// SIMATIC STEP 7 (V5.x) project Saldatura
// CPU: CPU 315-2 DP
// station: P_ADR_BUS
// station: Hardware
// station: SIMATIC 300(1)
// program: Programma S7(1)
// program: Originale

SYMBOL_TABLE
"Z10"	C 10	COUNTER	// Counter
"Z11"	C 11	COUNTER	// Counter
"Z12"	C 12	COUNTER	// Counter
"Z13"	C 13	COUNTER	// Counter
"DI_Balluff1"	DB 5	FB 20	// DB Instance of FB20
"DatiOP170B"	DB 7	DB 7	// PLC<->OP170B interface
"Timer"	DB 20	DB 20
"DBWork"	DB 21	DB 21
"coordinate"	DB 22	DB 22
"DB180"	DB 180	FB 24	// DB instance FB24 AsseY
"DB181"	DB 181	FB 24	// DB instance FB24 AsseX
"DBWork2"	DB 200	DB 200
"Asse_611U"	FB 16	FB 16	// Axis 611U management
"BALLUFF"	FB 20	FB 20	// BALLUFF Reader/Writer management
"FB24 - Gestione Mov Assi"	FB 24	FB 24	// GESTIONE ASSI STAZIONE
"NormalizzazioneAnalogico"	FC 7	FC 7	// Normalization of a analog value
"FC11 - STATUS"	FC 11	FC 11	// Sensors and proximity state
"FC12 - GENERAL"	FC 12	FC 12	// General management
"FC13 - MANUAL"	FC 13	FC 13	// Manual commands
"FC14 - AUTOMATIC"	FC 14	FC 14	// Automatic cycle management
"FC16 - ALARMS"	FC 16	FC 16	// Alarms management
"FC17 - OPERATOR PANNEL"	FC 17	FC 17	// Operator pannel management
"FC18 - OUTPUTS"	FC 18	FC 18	// Outputs management
"FC19 - REPOSITIONING"	FC 19	FC 19	// Repositioning management
"FC - AUTOMATIC"	FC 24	FC 24
"FC50 - TEACH-IN"	FC 50	FC 50
"FC51 - TYPE TOOL"	FC 51	FC 51
"FC52 - SYSTEM VISION"	FC 52	FC 52
"FC53 - REWORK"	FC 53	FC 53
"FC81 - GEST AXIS"	FC 81	FC 81	// Management axis
"FC117 - ERROR TOOL"	FC 117	FC 117
"TimeOut"	FC 800	FC 800	// Management TimeOut movimenti
"E0.0"	I 0.0	BOOL	// THERMAL SWTCH_ASPIRATOR_MTR
"E0.1"	I 0.1	BOOL	// 230 Vac power supply circuit braker
"E0.2"	I 0.2	BOOL	// 230 VAC PS CKT BRAKER
"E0.3"	I 0.3	BOOL	// Welding Machine OK
"E0.4"	I 0.4	BOOL	// Reserve
"E0.5"	I 0.5	BOOL	// AUXILIXARY ON
"DOOR CLOSE"	I 0.6	BOOL	// Reserve
"E0.7"	I 0.7	BOOL	// SAFETY BARRIER
"E1.0"	I 1.0	BOOL	// CYCLE_START
"E1.1"	I 1.1	BOOL	// AUTO_MANUAL
"E1.2"	I 1.2	BOOL	// COMPRESSED AIR
"E1.3"	I 1.3	BOOL	// AXIS RESET_POS
"E1.4"	I 1.4	BOOL	// Rotary table motor thermal switch
"E1.5"	I 1.5	BOOL	// LCK_UNLCK_DOORS_PB
"E1.6"	I 1.6	BOOL	// Reserve
"E1.7"	I 1.7	BOOL	// DRIVE TEMP
"E2.0"	I 2.0	BOOL	// STOP_CYCLE_PB
"E2.1"	I 2.1	BOOL	// Doors Closed & Locked
"E2.2"	I 2.2	BOOL	// Safety Barrier OK
"E2.3"	I 2.3	BOOL	// WELDING_TORCH_DWN
"E2.4"	I 2.4	BOOL	// WELDING_TORCH_UP
"E2.5"	I 2.5	BOOL	// ROTARY_TABLE_ZERO
"E2.6"	I 2.6	BOOL	// ROTARY_TABLE_ZERO1
"E2.7"	I 2.7	BOOL	// Reserve
"E3.0"	I 3.0	BOOL	// VEN DETECTOR_FWD
"E3.1"	I 3.1	BOOL	// VEN DETECTOR_REV
"E3.2"	I 3.2	BOOL	// VEN DETECTOR_DWN
"E3.3"	I 3.3	BOOL	// VEN DETECTOR_UP
"E3.4"	I 3.4	BOOL	// ROTARY_TABLE_CAM
"E3.5"	I 3.5	BOOL	// Reserve
"E3.6"	I 3.6	BOOL	// Reserve
"E3.7"	I 3.7	BOOL	// Reserve
"e5.0"	I 5.0	BOOL	// Lever Detector System - bit 0
"e5.1"	I 5.1	BOOL	// Lever Detector System - bit 1
"e5.2"	I 5.2	BOOL	// Lever Detector System - bit 2
"e5.3"	I 5.3	BOOL	// Lever Detector System - bit 3
"e5.4"	I 5.4	BOOL	// Lever Detector System - bit 4
"e5.5"	I 5.5	BOOL	// Lever Detector System - bit 5
"e5.6"	I 5.6	BOOL	// Lever Detector System - bit 6
"e5.7"	I 5.7	BOOL	// Lever Detector System - bit 7
"e6.0"	I 6.0	BOOL	// Lever Detector System - bit 8
"e6.1"	I 6.1	BOOL	// Lever Detector System - bit 9
"e6.2"	I 6.2	BOOL	// Lever Detector System - bit 10
"e6.3"	I 6.3	BOOL	// Lever Detector System - bit 11 - 12è13
"e6.4"	I 6.4	BOOL	// Lever Detector System - bit 12
"e6.5"	I 6.5	BOOL	// Lever Detector System - bit 13
"e6.6"	I 6.6	BOOL	// Lever Detector System - bit 14
"e6.7"	I 6.7	BOOL	// Lever Detector System - Vane Assy Total Number
"EXSTRACTOR_HIGH"	I 7.2	BOOL
"EXSTRACTOR_LOW"	I 7.3	BOOL
"TABLE_LCK_CYCLINDER_UP"	I 7.4	BOOL
"TABLE_LCK_CYCLINDER_DWN"	I 7.5	BOOL
"E32.0"	I 32.0	BOOL	// Push-button start cycle (on load position)
"E32.1"	I 32.1	BOOL	// Push button stop cycle
"E32.2"	I 32.2	BOOL	// Aut/Man Selector
"E32.3"	I 32.3	BOOL	// Reserve
"E32.4"	I 32.4	BOOL	// Reserve
"E32.5"	I 32.5	BOOL	// Lock/Unlock doors Push Button
"E32.6"	I 32.6	BOOL	// Reserve
"E32.7"	I 32.7	BOOL	// Air Presence
"E34.0"	I 34.0	BOOL	// Cam Table
"E34.1"	I 34.1	BOOL	// Reserve
"E34.2"	I 34.2	BOOL	// Reserve
"E34.3"	I 34.3	BOOL	// Reserve
"E34.4"	I 34.4	BOOL	// Table locker cylinder  up
"E34.5"	I 34.5	BOOL	// Table locker cylinder down
"E34.6"	I 34.6	BOOL	// Exstractor High
"E34.7"	I 34.7	BOOL	// Extractor Low
"E35.0"	I 35.0	BOOL	// Torch Welding low
"E35.1"	I 35.1	BOOL	// Torch Welding high
"E35.2"	I 35.2	BOOL	// Home Assy
"E35.3"	I 35.3	BOOL	// 1 --> PP1 on welding ; 0 --> PP2 on welding
"E35.4"	I 35.4	BOOL	// Detect components Control group High
"E35.5"	I 35.5	BOOL	// Detect components Control group Low
"E35.6"	I 35.6	BOOL	// Detect components Control group forward
"E35.7"	I 35.7	BOOL	// Detect components Control group backward
"E36.0"	I 36.0	BOOL	// Reserve not mounted
"E36.1"	I 36.1	BOOL	// Reserve not mounted
"E36.2"	I 36.2	BOOL	// Reserve not mounted
"E36.3"	I 36.3	BOOL	// Reserve not mounted
"E36.4"	I 36.4	BOOL	// Reserve not mounted
"E36.5"	I 36.5	BOOL	// Reserve not mounted
"E36.6"	I 36.6	BOOL	// Reserve not mounted
"E36.7"	I 36.7	BOOL	// Reserve not mounted
"E52.0"	I 52.0	BOOL	// Lever Detector System - bit 0
"E52.1"	I 52.1	BOOL	// Lever Detector System - bit 1
"E52.2"	I 52.2	BOOL	// Lever Detector System - bit 2
"E52.3"	I 52.3	BOOL	// Lever Detector System - bit 3
"E52.4"	I 52.4	BOOL	// Lever Detector System - bit 4
"E52.5"	I 52.5	BOOL	// Lever Detector System - bit 5
"E52.6"	I 52.6	BOOL	// Lever Detector System - bit 6
"E52.7"	I 52.7	BOOL	// Lever Detector System - bit 7
"E53.0"	I 53.0	BOOL	// Lever Detector System - bit 8
"E53.1"	I 53.1	BOOL	// Lever Detector System - bit 9
"E53.2"	I 53.2	BOOL	// Lever Detector System - bit 10
"E53.3"	I 53.3	BOOL	// Lever Detector System - bit 11 - 12è13
"E53.4"	I 53.4	BOOL	// Lever Detector System - bit 12
"E53.5"	I 53.5	BOOL	// Lever Detector System - bit 13
"E53.6"	I 53.6	BOOL	// Lever Detector System - bit 14
"E53.7"	I 53.7	BOOL	// Lever Detector System - Vane Assy Total Number
"E64.0"	I 64.0	BOOL	// VOSION SYSTEM OK
"E64.1"	I 64.1	BOOL	// Busy
"E64.2"	I 64.2	BOOL	// Or
"E64.3"	I 64.3	BOOL	// Error
"E64.4"	I 64.4	BOOL	// Gate
"E64.5"	I 64.5	BOOL	// Strobe trigger 0 out
"E64.6"	I 64.6	BOOL	// Strobe trigger 1 out
"E64.7"	I 64.7	BOOL	// DO0
"E65.0"	I 65.0	BOOL	// DO1
"E65.1"	I 65.1	BOOL	// DO2
"E65.2"	I 65.2	BOOL	// DO3
"E65.3"	I 65.3	BOOL	// DO4
"E65.4"	I 65.4	BOOL	// DO5
"E65.5"	I 65.5	BOOL	// DO6
"E65.6"	I 65.6	BOOL	// DO7
"E65.7"	I 65.7	BOOL	// DO8
"M0.0"	M 0.0	BOOL	// Clock 0,1 s
"M0.1"	M 0.1	BOOL	// Clock 0,2 s
"M0.2"	M 0.2	BOOL	// Clock 0,4 s
"M0.3"	M 0.3	BOOL	// Clock 0,5 s
"M0.4"	M 0.4	BOOL	// Clock 0,8 s
"M0.5"	M 0.5	BOOL	// Clock 1 s
"M0.6"	M 0.6	BOOL	// Clock 1,6 s
"M0.7"	M 0.7	BOOL	// Clock 2 s
"Off"	M 1.0	BOOL	// Merker always OFF
"On"	M 1.1	BOOL	// Merker always ON
"ToDo"	M 1.2	BOOL
"Bypass"	M 1.3	BOOL	// Merker that indicates a bypass forced of the code
"BypassPC"	M 1.4	BOOL	// Merker for bypass control handshake with PC supervision
"Clock_P"	M 1.5	BOOL	// Positiv pulse of clock
"Clock_N"	M 1.6	BOOL	// Negativ pulse of code
"Clock_10s"	M 1.7	BOOL	// 10 seconds clock
"M2.0"	M 2.0	BOOL	// Occhio
"BPSupervisor"	M 3.0	BOOL	// By Pass del supervisore
"Auxiliary_ON"	M 10.0	BOOL	// Auxiliary ON
"COMPRESSED_AIR"	M 10.1	BOOL	// Compressed Air
"SHIELDS_OK"	M 10.2	BOOL	// Schermi Chiusi e bloccati
"MACHINE_ON"	M 10.3	BOOL	// Machine OK
"Occhio"	M 10.7	BOOL
"START_POS"	M 11.0	BOOL	// Machine in initial positon
"START_POS_MEM"	M 11.1	BOOL	// mem initial position
"M11.2"	M 11.2	BOOL	// Manual Mode Selected
"SEMI"	M 11.3	BOOL	// Selezione modo semi automatico
"AUT"	M 11.4	BOOL	// Automatic Mode Selected
"START"	M 12.0	BOOL	// Start machine
"START_PULSE"	M 12.1	BOOL	// Pulse of start push-button
"SINGLE_CYCLE"	M 12.2	BOOL	// 1=ciclo singolo 0=ciclo continuo
"ALARM"	M 12.3	BOOL	// Alarm
"END_CYCLE"	M 12.4	BOOL	// Automatic cycle finished
"CmdMan_Av"	M 12.5	BOOL	// Forward manual command
"CmdMan_Ind"	M 12.6	BOOL	// Backward manual command
"STOP_BUTTON"	M 12.7	BOOL	// STATUS - stop button
"M13.0"	M 13.0	BOOL	// STATUS - Lock/Unlock doors Push Button
"M14.0"	M 14.0	BOOL	// Mem Lever Detector System - bit 0
"M14.1"	M 14.1	BOOL	// Mem Lever Detector System - bit 1
"M14.2"	M 14.2	BOOL	// Mem Lever Detector System - bit 2
"M14.3"	M 14.3	BOOL	// Mem Lever Detector System - bit 3
"M14.4"	M 14.4	BOOL	// Mem Lever Detector System - bit 4
"M14.5"	M 14.5	BOOL	// Mem Lever Detector System - bit 5
"M14.6"	M 14.6	BOOL	// Mem Lever Detector System - bit 6
"M14.7"	M 14.7	BOOL	// Mem Lever Detector System - bit 7
"M15.0"	M 15.0	BOOL	// Mem Lever Detector System - bit 8
"M15.1"	M 15.1	BOOL	// Mem Lever Detector System - bit 9
"M15.2"	M 15.2	BOOL	// Mem Lever Detector System - bit 10
"M15.3"	M 15.3	BOOL	// Mem Lever Detector System - bit 11
"M15.4"	M 15.4	BOOL	// Mem Lever Detector System - bit 12
"M15.5"	M 15.5	BOOL	// Mem Lever Detector System - bit 13
"M15.6"	M 15.6	BOOL	// Mem Lever Detector System - bit 14 (Roller)
"M15.7"	M 15.7	BOOL	// Mem Lever Detector System - bit 15
"M16.0"	M 16.0	BOOL	// mem Reworked Parts
"M16.1"	M 16.1	BOOL	// Disable Extractor if Rework
"M16.2"	M 16.2	BOOL	// Part on table 1 welding
"M16.3"	M 16.3	BOOL	// Part on Table 2 Welding
"M16.4"	M 16.4	BOOL	// Table can ROTATE
"M16.5"	M 16.5	BOOL	// Extractor can MOVE
"M16.6"	M 16.6	BOOL	// OK Extract
"M16.7"	M 16.7	BOOL	// Manual PAge Active
"M17.2"	M 17.2	BOOL	// Rework
"M17.3"	M 17.3	BOOL	// Vane no welding
"M17.4"	M 17.4	BOOL	// PP2 - OUT
"M17.5"	M 17.5	BOOL	// PP1 - OUT
"M17.6"	M 17.6	BOOL	// AUX - F R E E
"M17.7"	M 17.7	BOOL	// AUX - F R E E
"M18.0"	M 18.0	BOOL	// AUX - F R E E
"M18.1"	M 18.1	BOOL	// AUX - F R E E
"M18.2"	M 18.2	BOOL	// AUX - F R E E
"M18.3"	M 18.3	BOOL	// AUX - F R E E
"M18.4"	M 18.4	BOOL	// AUX - F R E E
"M18.5"	M 18.5	BOOL	// AUX - F R E E
"M18.6"	M 18.6	BOOL	// AUX - F R E E
"M18.7"	M 18.7	BOOL	// AUX - F R E E
"M19.0"	M 19.0	BOOL	// AUX - F R E E
"M19.1"	M 19.1	BOOL	// AUX - F R E E
"M19.2"	M 19.2	BOOL	// AUX - F R E E
"M19.3"	M 19.3	BOOL	// AUX - F R E E
"M19.4"	M 19.4	BOOL	// AUX - F R E E
"M19.5"	M 19.5	BOOL	// AUX - F R E E
"M19.6"	M 19.6	BOOL	// AUX - F R E E
"M19.7"	M 19.7	BOOL	// AUX - F R E E
"M20.0"	M 20.0	BOOL	// AUX - F R E E
"M20.1"	M 20.1	BOOL	// AUX - F R E E
"M20.2"	M 20.2	BOOL	// Presence of tool to assembly nozzle
"M20.3"	M 20.3	BOOL	// AUX - F R E E
"M20.4"	M 20.4	BOOL	// Tension OK
"M20.5"	M 20.5	BOOL	// AUX - F R E E
"M20.6"	M 20.6	BOOL	// AUX - F R E E
"M20.7"	M 20.7	BOOL	// AUX-Man
"M21.0"	M 21.0	BOOL	// STATUS - Mem Component pinched on Workrest - FC1
"Mem E34.5"	M 21.1	BOOL	// Mem Component pinched on Workrest - FC2
"M21.2"	M 21.2	BOOL	// AUX - F R E E
"M21.3"	M 21.3	BOOL	// AUX - F R E E
"M21.4"	M 21.4	BOOL	// Aux Alarm
"Warning"	M 21.5	BOOL	// Warning
"ResetAlarm"	M 21.6	BOOL	// Reset alarm
"Repos"	M 21.7	BOOL	// Repositioning
"M22.0"	M 22.0	BOOL	// STATUS - Table locker up
"M22.1"	M 22.1	BOOL	// STATUS - Table locker Down
"CmdMan_Av_Pulse"	M 22.2	BOOL	// Pulse of forward manual command
"CmdMan_Ind_Pulse"	M 22.3	BOOL	// Pulse of backward manual command
"M22.4"	M 22.4	BOOL	// Forward command
"M22.5"	M 22.5	BOOL	// Backward command
"CmdMan_Esg"	M 22.6	BOOL	// Memory of manual command executed
"CicloInCorso"	M 22.7	BOOL	// Automatic cycle in course
"M23.0"	M 23.0	BOOL	// Mem Start
"StopAEndCycle"	M 23.1	BOOL
"ChangeFunc"	M 23.2	BOOL	// Pulse change operation mode
"PresencePz"	M 23.3	BOOL
"SafetyBarrier_KO"	M 23.5	BOOL	// STATUS - Security bar KO
"M24.0"	M 24.0	BOOL	// STATUS - Torch Welding low
"M24.1"	M 24.1	BOOL	// STATUS - Torch Welding high
"M24.2"	M 24.2	BOOL	// STATUS -
"M24.3"	M 24.3	BOOL	// STATUS -
"M24.4"	M 24.4	BOOL	// STATUS - Cam table
"M24.5"	M 24.5	BOOL	// 1 --> PP1 on welding ;0 --> PP2 on welding
"M25.0"	M 25.0	BOOL	// Position Rotation 0°
"M25.1"	M 25.1	BOOL	// Position Rotation 180°
"M25.2"	M 25.2	BOOL	// Pos 0° e camma OK
"M25.3"	M 25.3	BOOL	// Pos 180° e camma OK
"M25.7"	M 25.7	BOOL	// Pulse Cam
"M26.1"	M 26.1	BOOL	// Table is FREE
"M26.2"	M 26.2	BOOL	// STATUS - System Detector Up
"M26.3"	M 26.3	BOOL	// STATUS - System Detector Lower
"M26.4"	M 26.4	BOOL	// STATUS - Detector work position
"M26.5"	M 26.5	BOOL	// STATUS - Detector park position
"M26.6"	M 26.6	BOOL	// STATUS - Exstractor High
"M26.7"	M 26.7	BOOL	// STATUS - Extractor low
"M28.0"	M 28.0	BOOL	// STATUS - DO1SYSTEM VISION
"M28.1"	M 28.1	BOOL	// STATUS - DO2 SYSTEM VISION
"M28.2"	M 28.2	BOOL	// STATUS - DO3 SYSTEM VISION
"M28.3"	M 28.3	BOOL	// STATUS - DO4 SYSTEM VISION
"M29.0"	M 29.0	BOOL	// STATUS - Run System Vision
"M29.1"	M 29.1	BOOL	// STATUS - Busy System Vision
"M29.2"	M 29.2	BOOL	// STATUS - OK System Vision
"M29.3"	M 29.3	BOOL	// STATUS - Error System Vision
"M29.4"	M 29.4	BOOL	// STATUS - Gate System Vision
"M29.6"	M 29.6	BOOL	// STATUS - DO1 SYSTEM VISION
"M29.7"	M 29.7	BOOL	// STATUS - DO0 SYSTEM VISION
"M30.0"	M 30.0	BOOL	// MAN - Table Rotation Forward
"M30.1"	M 30.1	BOOL	// MAN - Table Rotation Backward
"M30.2"	M 30.2	BOOL	// MAN - Jog + AsseY
"M30.3"	M 30.3	BOOL	// MAN - Jog - AsseY
"M30.4"	M 30.4	BOOL	// MAN - Jog + AsseX
"M30.5"	M 30.5	BOOL	// MAN - Jog - AsseX
"M30.6"	M 30.6	BOOL	// MAN - Forward SD
"M30.7"	M 30.7	BOOL	// MAN - Backward SD
"M31.0"	M 31.0	BOOL	// MAN - High SD
"M31.1"	M 31.1	BOOL	// MAN - Low SD
"M31.2"	M 31.2	BOOL	// MAN - High TW
"M31.3"	M 31.3	BOOL	// MAN - Low TW
"M31.4"	M 31.4	BOOL	// MAN - Extractor High
"M31.5"	M 31.5	BOOL	// MAN - Extractor down
"M31.6"	M 31.6	BOOL	// MAN - ON\OFF TW
"M31.7"	M 31.7	BOOL	// MAN - START/STOP WM
"M32.0"	M 32.0	BOOL	// Man  -  Start Torch W"elding
"M32.1"	M 32.1	BOOL	// MAN - Test Arco Gas Ok
"M32.2"	M 32.2	BOOL	// MAN - Test Arco Gas
"M32.3"	M 32.3	BOOL	// MAN - Torch Welding Temp Ok
"M32.4"	M 32.4	BOOL	// MAN - low table locker cylinder
"M32.5"	M 32.5	BOOL	// MAN - up table locker cylinder
"M32.6"	M 32.6	BOOL	// MAN - Welding
"M32.7"	M 32.7	BOOL	// MAN - Free
"M33.0"	M 33.0	BOOL	// MAN - Free
"M33.1"	M 33.1	BOOL	// MAN - Free
"M33.2"	M 33.2	BOOL	// MAN - Free
"M33.3"	M 33.3	BOOL	// MAN - Free
"M33.4"	M 33.4	BOOL	// MAN - Free
"M33.5"	M 33.5	BOOL	// MAN - Free
"M33.6"	M 33.6	BOOL	// MAN - Free
"M33.7"	M 33.7	BOOL	// MAN - Free
"M34.0"	M 34.0	BOOL	// MAN - Memory for rotation table
"M34.1"	M 34.1	BOOL	// MAN - Memory back rotation table
"M34.2"	M 34.2	BOOL	// MAN - Free
"M34.3"	M 34.3	BOOL	// MAN - Free
"M34.4"	M 34.4	BOOL	// MAN - Free
"M34.5"	M 34.5	BOOL	// MAN - Free
"M34.6"	M 34.6	BOOL	// MAN - Free
"M34.7"	M 34.7	BOOL	// MAN - Free
"M40.0"	M 40.0	BOOL	// RIP - Start repositioning
"M40.1"	M 40.1	BOOL	// RIP - Start reposit CamTable
"M40.2"	M 40.2	BOOL	// RIP - Cam Table
"M40.3"	M 40.3	BOOL	// RIP - System Detector vertical
"M40.4"	M 40.4	BOOL	// RIP - System Detector horizontal
"M40.5"	M 40.5	BOOL	// RIP - torch welding
"M40.6"	M 40.6	BOOL	// RIP - estractor
"M40.7"	M 40.7	BOOL	// RIP - Axis X and Y
"M41.0"	M 41.0	BOOL	// RIP - low table locker cylinder
"M41.1"	M 41.1	BOOL	// RIP - up table locker cylinder
"M41.2"	M 41.2	BOOL	// RIP - Free
"M41.3"	M 41.3	BOOL	// RIP - Free
"M41.4"	M 41.4	BOOL	// RIP - Free
"M41.5"	M 41.5	BOOL	// RIP - Free
"M41.6"	M 41.6	BOOL	// RIP - Free
"M41.7"	M 41.7	BOOL	// RIP - Free
"M42.0"	M 42.0	BOOL	// RIP - Free
"M42.1"	M 42.1	BOOL	// RIP - Table locker
"M42.2"	M 42.2	BOOL	// RIP - Free
"M42.3"	M 42.3	BOOL	// RIP - Free
"M42.4"	M 42.4	BOOL	// RIP - Free
"M42.5"	M 42.5	BOOL	// RIP - Free
"M42.6"	M 42.6	BOOL	// RIP - Free
"M42.7"	M 42.7	BOOL	// RIP - Free
"M50.0"	M 50.0	BOOL	// AUT - Table forward Side A
"M50.1"	M 50.1	BOOL	// AUT - Table backward Side B
"M50.2"	M 50.2	BOOL	// AUT - System Detector Forward
"M50.3"	M 50.3	BOOL	// AUT - System Detector Backward
"M50.4"	M 50.4	BOOL	// AUT - System Detector Low
"M50.5"	M 50.5	BOOL	// AUT - System Detector High
"M50.6"	M 50.6	BOOL	// AUT - welding down
"M50.7"	M 50.7	BOOL	// AUT - welding up
"M51.0"	M 51.0	BOOL	// AUT - Free
"M51.1"	M 51.1	BOOL	// AUT - Free
"M51.2"	M 51.2	BOOL	// AUT - Free
"M51.3"	M 51.3	BOOL	// AUT - Estractor High
"M51.4"	M 51.4	BOOL	// AUT - Estractor Low
"M51.5"	M 51.5	BOOL	// AUT - Free
"M51.6"	M 51.6	BOOL	// AUT - Free
"M51.7"	M 51.7	BOOL	// AUT - Free
"M52.0"	M 52.0	BOOL	// AUT -Temp  welding OK
"M52.1"	M 52.1	BOOL	// AUT - welding now
"M52.2"	M 52.2	BOOL	// AUT - Trigger System Vision
"M52.3"	M 52.3	BOOL	// AUT - ligth up
"M52.4"	M 52.4	BOOL	// AUT - Test Arc
"M52.5"	M 52.5	BOOL	// AUT - Test Arc Gas Ok
"M52.6"	M 52.6	BOOL	// AUT - low table locker cylinder
"M52.7"	M 52.7	BOOL	// AUT - up table locker cylinder
"M53.0"	M 53.0	BOOL	// AUT - Table locker Up
"M53.1"	M 53.1	BOOL	// AUT - Table locker Down
"M60.0"	M 60.0	BOOL	// STEP - 1:Table Forward
"M60.1"	M 60.1	BOOL	// STEP - 2:System Detector Forward
"M60.2"	M 60.2	BOOL	// STEP 3- System Detector Low
"M60.3"	M 60.3	BOOL	// STEP - 3 Check Nozzle Component
"M60.4"	M 60.4	BOOL	// STEP - 5 System detector High
"M60.5"	M 60.5	BOOL	// STEP 6 - System Detector Bacward
"M60.6"	M 60.6	BOOL	// STEP -7 welding down on point
"M60.7"	M 60.7	BOOL	// STEP - welding OK
"M61.0"	M 61.0	BOOL	// STEP - All welding is effectuated
"M61.1"	M 61.1	BOOL	// STEP - Photo Executed
"M61.2"	M 61.2	BOOL	// STEP - Axis in position 0
"M61.3"	M 61.3	BOOL	// STEP - point for welding receive
"M61.4"	M 61.4	BOOL	// STEP - welding up after work
"M61.5"	M 61.5	BOOL	// STEP - Welding in progress
"M61.6"	M 61.6	BOOL	// STEP - Start Rotation Table
"M61.7"	M 61.7	BOOL	// STEP - Photo without error
"M62.0"	M 62.0	BOOL	// STEP - Mem Reset Table
"M62.1"	M 62.1	BOOL	// STEP - Free
"M62.2"	M 62.2	BOOL	// STEP - Table cylinder up
"M62.3"	M 62.3	BOOL	// STEP - Free
"M62.4"	M 62.4	BOOL	// STEP - Free
"M62.5"	M 62.5	BOOL	// STEP - Free
"M62.6"	M 62.6	BOOL	// STEP - Free
"M62.7"	M 62.7	BOOL	// STEP - Photo Executed
"M63.0"	M 63.0	BOOL	// STEP - Nozzle Extracted
"M63.1"	M 63.1	BOOL	// STEP - Table Cylinder Low
"M63.6"	M 63.6	BOOL	// STEP - receive point photo
"M66.0"	M 66.0	BOOL	// STEP - photo 1 is NO good
"M66.1"	M 66.1	BOOL	// STEP - photo 2 is NO good
"M66.4"	M 66.4	BOOL	// STEP - Axis in position
"M66.6"	M 66.6	BOOL	// STEP - Execute 2th photo
"M66.7"	M 66.7	BOOL	// STEP - All photo is NO Good
"M67.0"	M 67.0	BOOL	// STEP - Axis Y in position
"M67.1"	M 67.1	BOOL	// STEP - Axis X in position
"M70.0"	M 70.0	BOOL	// Nozzle components Ok
"M70.1"	M 70.1	BOOL	// memNozzle-components Ok
"M70.2"	M 70.2	BOOL	// Component of Nozzle KO
"M70.3"	M 70.3	BOOL	// error assembling su PP1
"M70.4"	M 70.4	BOOL	// error assembling su PP2
"M71.0"	M 71.0	BOOL	// System Detector in Pos initial
"M72.0"	M 72.0	BOOL	// ready for welding
"M73.0"	M 73.0	BOOL	// Enable velocity for repositioning
"M74.0"	M 74.0	BOOL	// Output SV enable
"M74.1"	M 74.1	BOOL	// piece good
"M74.2"	M 74.2	BOOL	// piece reject
"M75.0"	M 75.0	BOOL	// Enable movement axis for teach in
"M75.1"	M 75.1	BOOL	// TeachIn OK
"M76.0"	M 76.0	BOOL	// position welding receive
"MEM Welding Machine OK"	M 80.0	BOOL
"Type_PP1_10_vane"	M 90.0	BOOL	// PP1-10 presence
"Type_PP2_9_vane"	M 90.1	BOOL	// presence PP2 -11 welding
"Type_PP3_9_vane"	M 90.2	BOOL	// presence PP3 - 9welding
"Type_PP4_13_vane"	M 90.3	BOOL	// presence PP4 - 13 Welding
"AUT STEP 1"	M 160.0	BOOL
"AUT STEP 2"	M 160.1	BOOL
"AUT STEP 3"	M 160.2	BOOL
"AUT STEP 4"	M 160.3	BOOL
"AUT STEP 5"	M 160.4	BOOL
"AUT STEP 6"	M 160.5	BOOL
"AUT STEP 7"	M 160.6	BOOL
"AUT STEP 8"	M 160.7	BOOL
"AUT STEP 9"	M 161.0	BOOL
"AUT STEP10"	M 161.1	BOOL
"AUT STEP11"	M 161.2	BOOL
"AUT STEP12"	M 161.3	BOOL
"AUT STEP13"	M 161.4	BOOL
"AUT STEP14"	M 161.5	BOOL
"AUT STEP15"	M 161.6	BOOL
"AUT STEP16"	M 161.7	BOOL
"AUT STEP17"	M 162.0	BOOL
"AUT STEP18"	M 162.1	BOOL
"AUT STEP19"	M 162.2	BOOL
"AUT STEP20"	M 162.3	BOOL
"AUT STEP21"	M 162.4	BOOL
"AUT STEP22"	M 162.5	BOOL
"AUT STEP23"	M 162.6	BOOL
"AUT STEP24"	M 162.7	BOOL
"AUT STEP25"	M 163.0	BOOL
"AUT STEP26"	M 163.1	BOOL
"AUT STEP27"	M 163.2	BOOL
"AUT STEP28"	M 163.3	BOOL
"AUT STEP29"	M 163.4	BOOL
"AUT STEP30"	M 163.5	BOOL
"Clock 0.5 S"	M 200.3	BOOL
"Clock 1s"	M 200.5	BOOL
"M254.0"	M 254.0	BOOL	// Front Command HOME
"M254.1"	M 254.1	BOOL	// Front Command END
"M256.0"	M 256.0	BOOL	// Pulse
"M256.2"	M 256.2	BOOL	// Pulse
"M256.6"	M 256.6	BOOL	// Pulse
"M256.7"	M 256.7	BOOL	// Pulse
"M340.0"	M 340.0	BOOL	// AXIS Y:STOP MOVE
"M340.1"	M 340.1	BOOL	// AXIS Y:START POSITIONING
"M340.2"	M 340.2	BOOL	// AXIS Y:START SEARCH HOME
"M340.3"	M 340.3	BOOL	// AXIS Y:START POSITIONING ON HOME
"M340.4"	M 340.4	BOOL	// AXIS X:COMMAND JOG PLUS
"M340.5"	M 340.5	BOOL	// AXIS X:COMANDO JOG LESS
"M341.0"	M 341.0	BOOL	// AXIS Y:ACHIEVED LOCATION
"M341.1"	M 341.1	BOOL	// AXIS Y:REFERED AXIS
"M341.2"	M 341.2	BOOL	// AXIS Y:AXIS LOCATION ON HOME
"M341.3"	M 341.3	BOOL	// AXIS Y:AXIS STOP NONE COMMAND PROGRESS
"M341.4"	M 341.4	BOOL	// AXIS Y:SETTING SETTING IN MOTION OK
"M341.5"	M 341.5	BOOL	// AXIS Y:ALLRM SETTING IN MOTION
"M342.0"	M 342.0	BOOL	// AXIS Y:AXIS ON CAM OF  REFERENCE
"M342.1"	M 342.1	BOOL	// AXIS Y:AXIS ON OVER RACE NEGATIVE HARDWARE
"M342.2"	M 342.2	BOOL	// AXIS Y:AXIS ON OVER RACE POSITIVE HARDWARE
"M342.3"	M 342.3	BOOL	// AXIS Y:COMMAND BRAKE PARKING
"M342.4"	M 342.4	BOOL	// AXIS Y:AXIS ON OVER RACE NEGATIVE SOFTWARE
"M342.5"	M 342.5	BOOL	// AXIS Y:AXIS ON OVER RACE POSITIVE SOFTWARE
"M342.6"	M 342.6	BOOL	// AXIS Y:POSSIBLE MOVE AXIS
"M342.7"	M 342.7	BOOL	// AXIS Y:INITIAL LOCATION AXIS
"M343.0"	M 343.0	BOOL	// AXIS Y:START POSITIONING INCREMENTAL
"M346.0"	M 346.0	BOOL	// AXIS X:STOP MOVE
"M346.1"	M 346.1	BOOL	// AXIS X:START POSITIONING
"M346.2"	M 346.2	BOOL	// AXIS X:START SEARCH HOME
"M346.3"	M 346.3	BOOL	// AXIS X:START POSITIONING ON HOME
"M346.4"	M 346.4	BOOL	// AXIS Y:COMMAND JOG PLUS
"M346.5"	M 346.5	BOOL	// AXIS Y:COMANDO JOG LESS
"M347.0"	M 347.0	BOOL	// AXIS X:ACHIEVED LOCATION
"M347.1"	M 347.1	BOOL	// AXIS X:REFERED AXIS
"M347.2"	M 347.2	BOOL	// AXIS X:AXIS LOCATION ON HOME
"M347.3"	M 347.3	BOOL	// AXIS X:AXIS STOP NONE COMMAND PROGRESS
"M347.4"	M 347.4	BOOL	// AXIS X:SETTING SETTING IN MOTION OK
"M347.5"	M 347.5	BOOL	// AXIS X:ALLRM SETTING IN MOTION
"M348.0"	M 348.0	BOOL	// AXIS X:AXIS ON CAM OF  REFERENCE
"M348.1"	M 348.1	BOOL	// AXIS X:AXIS ON OVER RACE NEGATIVE HARDWARE
"M348.2"	M 348.2	BOOL	// AXIS X:AXIS ON OVER RACE POSITIVE HARDWARE
"M348.3"	M 348.3	BOOL	// AXIS X:COMMAND BRAKE PARKING
"M348.4"	M 348.4	BOOL	// AXIS X:AXIS ON OVER RACE NEGATIVE SOFTWARE
"M348.5"	M 348.5	BOOL	// AXIS X:AXIS ON OVER RACE POSITIVE SOFTWARE
"M348.6"	M 348.6	BOOL	// AXIS X:POSSIBLE MOVE AXIS
"M348.7"	M 348.7	BOOL	// AXIS X:INITIAL LOCATION AXIS
"M349.0"	M 349.0	BOOL	// AXIS X:START POSITIONING INCREMENTAL
"Photo 2 executed"	M 500.0	BOOL	// m61.1
"TriggerVisSystem2"	M 500.1	BOOL
"ErroreCamera"	M 500.7	BOOL
"M1000.0"	M 1000.0	BOOL	// AUX
"M1000.1"	M 1000.1	BOOL	// AUX
"M1000.2"	M 1000.2	BOOL	// AUX
"M1000.3"	M 1000.3	BOOL	// AUX
"M1000.4"	M 1000.4	BOOL	// AUX
"M1000.5"	M 1000.5	BOOL	// AUX
"M1000.6"	M 1000.6	BOOL	// AUX
"M1000.7"	M 1000.7	BOOL	// AUX
"M1001.0"	M 1001.0	BOOL	// AUX
"M1001.1"	M 1001.1	BOOL	// AUX
"M1001.2"	M 1001.2	BOOL	// AUX
"M1001.3"	M 1001.3	BOOL	// AUX
"M1001.4"	M 1001.4	BOOL	// AUX
"M1001.5"	M 1001.5	BOOL	// AUX
"M1001.6"	M 1001.6	BOOL	// AUX
"M1001.7"	M 1001.7	BOOL	// AUX
"M1002.0"	M 1002.0	BOOL	// AUX
"M1002.1"	M 1002.1	BOOL	// AUX
"M1002.2"	M 1002.2	BOOL	// AUX
"M1002.3"	M 1002.3	BOOL	// AUX
"M1002.4"	M 1002.4	BOOL	// AUX
"M1002.5"	M 1002.5	BOOL	// AUX
"M1002.6"	M 1002.6	BOOL	// AUX
"M1002.7"	M 1002.7	BOOL	// AUX
"M1003.0"	M 1003.0	BOOL	// AUX
"M1003.1"	M 1003.1	BOOL	// AUX
"M1003.2"	M 1003.2	BOOL	// AUX
"M1003.3"	M 1003.3	BOOL	// AUX
"M1003.4"	M 1003.4	BOOL	// AUX
"M1003.5"	M 1003.5	BOOL	// AUX
"M1003.6"	M 1003.6	BOOL	// AUX
"M1003.7"	M 1003.7	BOOL	// AUX
"M1004.0"	M 1004.0	BOOL	// AUX
"M1004.1"	M 1004.1	BOOL	// AUX
"M1004.2"	M 1004.2	BOOL	// AUX
"M1004.3"	M 1004.3	BOOL	// AUX
"M1004.4"	M 1004.4	BOOL	// AUX
"M1004.5"	M 1004.5	BOOL	// AUX
"M1004.6"	M 1004.6	BOOL	// AUX
"M1004.7"	M 1004.7	BOOL	// AUX
"M1005.0"	M 1005.0	BOOL	// AUX
"M1005.1"	M 1005.1	BOOL	// AUX
"M1005.2"	M 1005.2	BOOL	// AUX
"M1005.3"	M 1005.3	BOOL	// AUX
"M1005.4"	M 1005.4	BOOL	// AUX
"M1005.5"	M 1005.5	BOOL	// AUX
"M1005.6"	M 1005.6	BOOL	// AUX
"M1005.7"	M 1005.7	BOOL	// AUX
"M1006.0"	M 1006.0	BOOL	// AUX
"M1006.1"	M 1006.1	BOOL	// AUX
"M1006.2"	M 1006.2	BOOL	// AUX
"M1006.3"	M 1006.3	BOOL	// AUX
"M1006.4"	M 1006.4	BOOL	// AUX
"M1006.5"	M 1006.5	BOOL	// AUX
"M1006.6"	M 1006.6	BOOL	// AUX
"M1006.7"	M 1006.7	BOOL	// AUX
"M1007.0"	M 1007.0	BOOL	// AUX
"M1007.1"	M 1007.1	BOOL	// AUX
"M1007.2"	M 1007.2	BOOL	// AUX
"M1007.3"	M 1007.3	BOOL	// AUX
"M1007.4"	M 1007.4	BOOL	// AUX
"M1007.5"	M 1007.5	BOOL	// AUX
"M1007.6"	M 1007.6	BOOL	// AUX
"M1007.7"	M 1007.7	BOOL	// AUX
"M1008.0"	M 1008.0	BOOL	// AUX
"M1008.1"	M 1008.1	BOOL	// AUX
"M1008.2"	M 1008.2	BOOL	// AUX
"M1008.3"	M 1008.3	BOOL	// AUX
"M1008.4"	M 1008.4	BOOL	// AUX
"M1008.5"	M 1008.5	BOOL	// AUX
"M1008.6"	M 1008.6	BOOL	// AUX
"M1008.7"	M 1008.7	BOOL	// AUX
"M1009.0"	M 1009.0	BOOL	// AUX
"M1009.1"	M 1009.1	BOOL	// AUX
"M1009.2"	M 1009.2	BOOL	// AUX
"M1009.3"	M 1009.3	BOOL	// AUX
"M1009.4"	M 1009.4	BOOL	// AUX
"M1009.5"	M 1009.5	BOOL	// AUX
"M1009.6"	M 1009.6	BOOL	// AUX
"M1009.7"	M 1009.7	BOOL	// AUX
"FPAuxON_force_Axis_reset"	M 1900.0	BOOL
"Luce telecamera"	M 1900.2	BOOL
"AppoFP_M1900.3"	M 1900.3	BOOL
"Soffio Camera"	M 1900.4	BOOL
"Manual_cameralight_on"	M 1900.5	BOOL
"M2034.0"	M 2034.0	BOOL	// Key Start from pannell
"M2034.1"	M 2034.1	BOOL	// Key Finish from pannell
"M2034.2"	M 2034.2	BOOL	// Key Teach In from Pannell
"M2034.5"	M 2034.5	BOOL	// Key Enter teach from pannel
"M2034.6"	M 2034.6	BOOL	// Key Exit teach from pannel
"M2034.7"	M 2034.7	BOOL	// Key Rite from pannell
"M2035.0"	M 2035.0	BOOL	// Key Start from Teach In page
"M2035.1"	M 2035.1	BOOL	// Key Welding Run from pannel
"M2035.2"	M 2035.2	BOOL	// Key ACK on page 21 from pannell
"MB2046"	MB 2046	BYTE	// white byte
"MD30"	MD 30	DWORD	// DWORD Manual Commands
"MD100"	MD 100	DWORD	// temp
"MD588"	MD 588	DINT	// temporary for X point
"MD592"	MD 592	DINT	// temporary for X point
"MD596"	MD 596	DINT	// target X
"MD600"	MD 600	DINT	// target Y
"MD620"	MD 620	DWORD	// InsertPointX
"MD624"	MD 624	DWORD	// InsertPointY
"MD650"	MD 650	DINT	// axis X actual position
"MD654"	MD 654	DINT	// axis Y actual posiion
"SaldEffet"	MW 110	WORD	// number welding make
"MW120"	MW 120	INT	// number welding make
"MW300"	MW 300	INT	// number point to want go
"MW2042"	MW 2042	INT	// temp for clock
"MAIN PROGRAM"	OB 1	OB 1	// Main Program
"I/O_FLT1"	OB 82	OB 82	// I/O Point Fault 1
"RACK_FLT"	OB 86	OB 86	// Loss of Rack Fault
"COMPLETE RESTART"	OB 100	OB 100	// Complete Restart
"MOD_ERR"	OB 122	OB 122	// Module Access Error
"A0.0"	Q 0.0	BOOL	// Red Lamp
"A0.1"	Q 0.1	BOOL	// Yellow Lamp
"A0.2"	Q 0.2	BOOL	// Green Lamp
"A0.3"	Q 0.3	BOOL	// Lock doors relay
"A0.4"	Q 0.4	BOOL	// Simodrive Reset realy
"A0.5"	Q 0.5	BOOL	// Reserve
"A0.6"	Q 0.6	BOOL	// Reserve
"A0.7"	Q 0.7	BOOL	// Reserve
"A1.0"	Q 1.0	BOOL	// Enable Coral Vacuum
"A1.1"	Q 1.1	BOOL	// Test Gas Arco Pilota
"A1.2"	Q 1.2	BOOL	// Forward table rotation
"A1.3"	Q 1.3	BOOL	// Backward table rotation
"A1.4"	Q 1.4	BOOL	// Enable Axis X
"A1.5"	Q 1.5	BOOL	// Enable Axis Y
"A1.6"	Q 1.6	BOOL	// Start Welding
"A1.7"	Q 1.7	BOOL	// Ignition torch
"A2.0"	Q 2.0	BOOL	// Reserve
"A2.1"	Q 2.1	BOOL	// Reserve
"A2.2"	Q 2.2	BOOL	// Reserve
"A2.3"	Q 2.3	BOOL	// Reserve
"A2.4"	Q 2.4	BOOL	// Reserve
"A2.5"	Q 2.5	BOOL	// Reserve
"A2.6"	Q 2.6	BOOL	// Reserve
"A2.7"	Q 2.7	BOOL	// Reserve
"A3.0"	Q 3.0	BOOL	// Reserve
"A3.1"	Q 3.1	BOOL	// Reserve
"A3.2"	Q 3.2	BOOL	// Reserve
"A3.3"	Q 3.3	BOOL	// Reserve
"A3.4"	Q 3.4	BOOL	// Reserve
"A3.5"	Q 3.5	BOOL	// Reserve
"A3.6"	Q 3.6	BOOL	// Reserve
"A3.7"	Q 3.7	BOOL	// Reserve
"SIMODRIVE_RESET"	Q 12.0	BOOL
"BUZZER"	Q 12.1	BOOL
"Torch Welding Machin"	Q 12.2	BOOL	// Down
"Torch Welding MachinE"	Q 12.3	BOOL	// UP
"TABLE_LCKER_DWN"	Q 12.4	BOOL
"Table locker cylinder up"	Q 12.5	BOOL
"FWD_LEVER_DETECT_SYS"	Q 12.6	BOOL
"REV_LEVER_DETECT_SYS"	Q 12.7	BOOL
"UP_lever detector system"	Q 13.0	BOOL
"DW_lever detector sys"	Q 13.1	BOOL
"UP_Down _Extractor"	Q 13.2	BOOL
"_soffio_telecamera"	Q 13.3	BOOL
"DRIVE_ENABLE"	Q 13.5	BOOL
"ENABLE_Y_AXIS"	Q 13.6	BOOL
"ENABLE_X_AXIS"	Q 13.7	BOOL
"STOP_CYCLE_LAMP"	Q 14.3	BOOL
"START_CYCLE_LAMP"	Q 14.4	BOOL
"a14.5"	Q 14.5	BOOL
"ACCESES_BARRIER_LAMP"	Q 14.6	BOOL
"Enable Coral Vacuum"	Q 17.0	BOOL
"FWD_TABLE_ROTATION"	Q 17.1	BOOL
"REVERSE_TABLE_ROTATION"	Q 17.2	BOOL
"IGNITION_TORCH"	Q 17.5	BOOL
"START_WELDING"	Q 17.6	BOOL
"Test Gas Arc Pilota"	Q 17.7	BOOL
"PLC READY"	Q 18.0	BOOL	// ADDITION
"_Illumin_telecamera"	Q 18.1	BOOL
"PIECE_REFUSE"	Q 18.3	BOOL
"RED_LAMP"	Q 18.4	BOOL
"PIECE_GOOD"	Q 18.5	BOOL
"Lamp_Door_Locked"	Q 18.6	BOOL
"LOCK_DOORS_RELAY"	Q 18.7	BOOL
"A32.0"	Q 32.0	BOOL	// Lamp Start cycle
"A32.1"	Q 32.1	BOOL	// Lamp Stop cycle
"A32.2"	Q 32.2	BOOL	// Piece Good
"A32.3"	Q 32.3	BOOL	// Piece Refuse
"A32.4"	Q 32.4	BOOL	// Unlocked doors
"A32.5"	Q 32.5	BOOL	// Emergency Lamp
"A32.6"	Q 32.6	BOOL	// Access barrier Lamp
"A32.7"	Q 32.7	BOOL	// Buzzer
"A33.0"	Q 33.0	BOOL	// Reserve
"A33.1"	Q 33.1	BOOL	// Reserve
"A33.2"	Q 33.2	BOOL	// Reserve
"A33.3"	Q 33.3	BOOL	// Reserve
"A33.4"	Q 33.4	BOOL	// Reserve not mounted
"A33.5"	Q 33.5	BOOL	// Reserve not mounted
"A33.6"	Q 33.6	BOOL	// Reserve not mounted
"A33.7"	Q 33.7	BOOL	// Reserve not mounted
"A34.0"	Q 34.0	BOOL	// Forward lever detector System
"A34.1"	Q 34.1	BOOL	// Backward lever detector System
"A34.2"	Q 34.2	BOOL	// Down lever detector system
"A34.3"	Q 34.3	BOOL	// Up lever detector system
"A34.4"	Q 34.4	BOOL	// Down Torch Welding Machine
"A34.5"	Q 34.5	BOOL	// Up Torch Welding Machine
"A34.6"	Q 34.6	BOOL	// Down Extractor
"A34.7"	Q 34.7	BOOL	// Up Extractor
"A35.0"	Q 35.0	BOOL	// Table locker down
"A35.1"	Q 35.1	BOOL	// Table locker up
"A35.2"	Q 35.2	BOOL	// Reserve
"A35.3"	Q 35.3	BOOL	// Reserve
"A35.4"	Q 35.4	BOOL	// Reserve
"A35.5"	Q 35.5	BOOL	// Reserve
"A35.6"	Q 35.6	BOOL	// Reserve
"A35.7"	Q 35.7	BOOL	// Reserve
"A64.0"	Q 64.0	BOOL	// Reset
"A64.1"	Q 64.1	BOOL	// Trigger
"A64.2"	Q 64.2	BOOL	// Data Send Request
"A64.3"	Q 64.3	BOOL	// DI0
"A64.4"	Q 64.4	BOOL	// DI1
"A64.5"	Q 64.5	BOOL	// DI2
"A64.6"	Q 64.6	BOOL	// DI3
"A64.7"	Q 64.7	BOOL	// DI4
"A65.0"	Q 65.0	BOOL	// DI5
"A65.1"	Q 65.1	BOOL	// DI6
"A65.2"	Q 65.2	BOOL	// DI7
"A65.3"	Q 65.3	BOOL	// DI8
"A65.4"	Q 65.4	BOOL	// DI9
"A65.5"	Q 65.5	BOOL	// Reserve
"A65.6"	Q 65.6	BOOL	// Reserve
"A65.7"	Q 65.7	BOOL	// Reserve
"TON"	SFB 4	SFB 4	// Generate an On Delay
"READ_CLK"	SFC 1	SFC 1	// Read System Clock
"DPRD_DAT"	SFC 14	SFC 14	// Read Consistent Data of a Standard DP Slave
"DPWR_DAT"	SFC 15	SFC 15	// Write Consistent Data to a Standard DP Slave
"BLKMOV"	SFC 20	SFC 20	// Copy Variables
"FILL"	SFC 21	SFC 21	// Initialize a Memory Area
"CREAT_DB"	SFC 22	SFC 22	// Create Data Block
"DIS_AIRT"	SFC 41	SFC 41	// Delay the Higher Priority Interrupts and Asynchronous Errors
"EN_AIRT"	SFC 42	SFC 42	// Enable Higher Priority Interrupts and Asynchronous Errors
"STP"	SFC 46	SFC 46	// Change the CPU to STOP
"LGC_GADR"	SFC 49	SFC 49	// Query the Module Slot Belonging to a Logical Address
"RDSYSST"	SFC 51	SFC 51	// Read a System Status List or Partial List
"WR_REC"	SFC 58	SFC 58	// Write Data Record
"RD_REC"	SFC 59	SFC 59	// Read a Data Record
"T2"	T 2	TIMER
"T3"	T 3	TIMER	// Time for Component Start UP
"T10"	T 10	TIMER	// Delay
"T11"	T 11	TIMER
"T12"	T 12	TIMER	// delay next step
"T13"	T 13	TIMER	// Delay
"T14"	T 14	TIMER	// timer for delay KO
"T15"	T 15	TIMER	// Delay
"T16"	T 16	TIMER	// Delay
"T17"	T 17	TIMER	// timer delay
"T18"	T 18	TIMER	// Delay
"T19"	T 19	TIMER	// delay
"T20"	T 20	TIMER	// timer delay
"T21"	T 21	TIMER	// Time Test Arc
"T22"	T 22	TIMER	// Delay
"T23"	T 23	TIMER	// Timer for repositioning
"T24"	T 24	TIMER	// Delay make 2th photo
"T25"	T 25	TIMER	// delay
"T26"	T 26	TIMER	// time for reset output rotation table
"T27"	T 27	TIMER	// Timer for Executed Photo
"T28"	T 28	TIMER	// Delay for entry in teach in mode
"T29"	T 29	TIMER	// delay for reset both axis
"T30"	T 30	TIMER	// timer dealy
"T31"	T 31	TIMER	// MAN - time for welding
"T32"	T 32	TIMER	// MAN - time for welding UP
"T33"	T 33	TIMER	// Delay
"T34"	T 34	TIMER	// Time Test Arco
"T35"	T 35	TIMER	// Delay
"T36"	T 36	TIMER	// delay for cam not present
"T37"	T 37	TIMER	// Time Torch Welding Ok
"T38"	T 38	TIMER	// timer reset alarms axis X
"T39"	T 39	TIMER	// timer reset alarms axis Y
"T40"	T 40	TIMER	// Time Torch Welding Ok
"T41"	T 41	TIMER	// delay alarm air pressure
"T42"	T 42	TIMER	// Timer stop welding
"T43"	T 43	TIMER	// Timer welding Manual
"T44"	T 44	TIMER	// Delay
"T45"	T 45	TIMER	// timer for upgrade value
"T46"	T 46	TIMER	// delay enable axis Ytimer reset alarms axis X
"T47"	T 47	TIMER	// delay
"T48"	T 48	TIMER	// delay enable axis Ytimer reset alarms axis Y
"T50"	T 50	TIMER	// Delay
"T51"	T 51	TIMER
"T52"	T 52	TIMER	// wait after rotation table
"T53"	T 53	TIMER	// delay for chek camera point
"T54"	T 54	TIMER	// delay turn OFF Buzzer
"T60"	T 60	TIMER	// Delay for entry in teach in mode
"T61"	T 61	TIMER	// delay go in position for 2th photo
"T62"	T 62	TIMER	// delay for axis in position
"T63"	T 63	TIMER	// Delay
"T_SystemDetectorDW"	T 70	TIMER
"T_SystemDetector_UP"	T 71	TIMER
"T90"	T 90	TIMER	// delay allarm for Simodrive
"VAT_1"	VAT 1	
"Coordinate_saldatura"	VAT 2	
"I/O System Vision"	VAT 3	
"Saldatrice"	VAT 4	
"VAT_12"	VAT 5	
"VAT_PUNTI_AVV"	VAT 6	
"VAT_PUNTI_AVV_2"	VAT 7	
"DB22_SaldaturaSilv"	VAT 8	
"DB22_Sald_PP1"	VAT 9	
"VAT_tool check"	VAT 10	
"VAT_Balluff"	VAT 11	
"ASSE_P"	VAT 12	
"DB22_Sald_PP3"	VAT 13	
"VAT_Point"	VAT 14	
"VAT_Point 16"	VAT 15	
"DB22_Sald_PP16"	VAT 16	
"VAT_17"	VAT 17	
"Tipo portapezzo"	VAT 18	
"VAT_Daniele"	VAT 19	
END_SYMBOL_TABLE

FUNCTION_BLOCK "Asse_611U"	// FB 16
AUTHOR : Cellini
VERSION : 0.1
BEGIN
// (block stored without names or comments; labels and parameter names are numbered)
NETWORK
TITLE =
      L     DIW [AR2,P#0.0];
      SLD   3;
      T     LD 28;
      L     P#DIX 2.0;
      T     LD 36;
      L     11;
M001: T     LW 34;
      L     PIW [LD 28];
      T     DIW [LD 36];
      L     LD 28;
      L     P#2.0;
      +D;
      T     LD 28;
      L     LD 36;
      L     P#2.0;
      +D;
      T     LD 36;
      L     LW 34;
      LOOP  M001;
NETWORK
TITLE =
      A     DIX [AR2,P#10.5];
      AN    DIX [AR2,P#10.4];
      =     DIX [AR2,P#45.1];
      A     DIX [AR2,P#11.0];
      A     DIX [AR2,P#11.1];
      A     DIX [AR2,P#11.2];
      AN    DIX [AR2,P#11.3];
      A     DIX [AR2,P#11.4];
      A     DIX [AR2,P#11.5];
      A     DIX [AR2,P#10.0];
      =     DIX [AR2,P#45.2];
      A     DIX [AR2,P#17.5];
      =     DIX [AR2,P#45.3];
      A     DIX [AR2,P#23.0];
      =     DIX [AR2,P#45.4];
      A     DIX [AR2,P#23.1];
      =     DIX [AR2,P#45.5];
      A     DIX [AR2,P#23.2];
      =     DIX [AR2,P#45.6];
      A     DIX [AR2,P#15.6];
      =     DIX [AR2,P#45.7];
      A     DIX [AR2,P#15.7];
      =     DIX [AR2,P#46.0];
      L     DID [AR2,P#18.0];
      T     DID [AR2,P#62.0];
NETWORK
TITLE =
      A     DIX [AR2,P#42.0];
      =     DIX [AR2,P#33.0];
      =     DIX [AR2,P#33.1];
      =     DIX [AR2,P#33.2];
      A     "On";
      =     DIX [AR2,P#33.3];
      O     DIX [AR2,P#42.2];
      O     DIX [AR2,P#11.3];
      ON    DIX [AR2,P#10.0];
      R     DIX [AR2,P#42.3];
      R     DIX [AR2,P#44.0];
      R     DIX [AR2,P#44.1];
      R     DIX [AR2,P#42.4];
      R     DIX [AR2,P#44.2];
      R     DIX [AR2,P#44.3];
      R     DIX [AR2,P#42.5];
      R     DIX [AR2,P#42.6];
      R     DIX [AR2,P#32.3];
      R     DIX [AR2,P#33.6];
      AN    DIX [AR2,P#42.2];
      =     DIX [AR2,P#33.4];
      AN    DIX [AR2,P#42.7];
      =     DIX [AR2,P#33.5];
      A     DIX [AR2,P#42.1];
      =     DIX [AR2,P#33.7];
      A     DIX [AR2,P#10.1];
      =     DIX [AR2,P#32.2];
      L     DIW [AR2,P#60.0];
      T     DIW [AR2,P#40.0];
NETWORK
TITLE =
      A     DIX [AR2,P#42.3];
      A(;
      L     DID [AR2,P#48.0];
      L     50;
      <D;
      );
      A(;
      L     DID [AR2,P#48.0];
      L     -50;
      >D;
      );
      R     DIX [AR2,P#42.3];
      A     DIX [AR2,P#42.3];
      R     DIX [AR2,P#35.0];
      S     DIX [AR2,P#35.1];
      R     DIX [AR2,P#35.2];
      R     DIX [AR2,P#35.3];
      R     DIX [AR2,P#35.4];
      R     DIX [AR2,P#35.5];
      A     DIX [AR2,P#42.3];
      AN    DIX [AR2,P#44.0];
      AN    DIX [AR2,P#44.1];
      S     DIX [AR2,P#44.0];
      JCN   M002;
      L     DID [AR2,P#48.0];
      T     DID [AR2,P#28.0];
      L     W#16#8051;
      T     DIW [AR2,P#24.0];
      L     2;
      T     DIW [AR2,P#26.0];
M002: NOP   0;
      A     DIX [AR2,P#42.3];
      A     DIX [AR2,P#44.0];
      AN    DIX [AR2,P#44.1];
      A(;
      L     DID [AR2,P#28.0];
      L     DID [AR2,P#6.0];
      ==D;
      );
      A(;
      L     W#16#5051;
      L     DIW [AR2,P#2.0];
      ==I;
      );
      A(;
      L     DIW [AR2,P#26.0];
      L     DIW [AR2,P#4.0];
      ==I;
      );
      S     DIX [AR2,P#44.1];
      A     DIX [AR2,P#42.3];
      A     DIX [AR2,P#44.0];
      A     DIX [AR2,P#44.1];
      A(;
      L     DID [AR2,P#48.0];
      L     DID [AR2,P#6.0];
      ==D;
      );
      AN    DIX [AR2,P#33.6];
      S     DIX [AR2,P#33.6];
      JCN   M003;
      L     0;
      T     DIW [AR2,P#24.0];
      T     DIW [AR2,P#26.0];
      T     DID [AR2,P#28.0];
M003: NOP   0;
      A     DIX [AR2,P#10.2];
      FP    DIX [AR2,P#47.0];
      A     DIX [AR2,P#42.3];
      A     DIX [AR2,P#44.0];
      A     DIX [AR2,P#44.1];
      A     DIX [AR2,P#33.6];
      R     DIX [AR2,P#33.6];
      R     DIX [AR2,P#42.3];
      R     DIX [AR2,P#44.0];
      R     DIX [AR2,P#44.1];
NETWORK
TITLE =
      A     DIX [AR2,P#42.4];
      AN    DIX [AR2,P#44.2];
      AN    DIX [AR2,P#44.3];
      JCN   M005;
      L     DID [AR2,P#52.0];
      L     DID [AR2,P#18.0];
      -D;
      T     DID [AR2,P#56.0];
      L     0;
      <D;
      JCN   M004;
      L     DID [AR2,P#56.0];
      NEGD;
      T     DID [AR2,P#56.0];
M004: NOP   0;
      A(;
      L     DID [AR2,P#56.0];
      L     99;
      <=D;
      );
      R     DIX [AR2,P#42.4];
M005: NOP   0;
      A     DIX [AR2,P#42.4];
      R     DIX [AR2,P#35.0];
      R     DIX [AR2,P#35.1];
      R     DIX [AR2,P#35.2];
      R     DIX [AR2,P#35.3];
      R     DIX [AR2,P#35.4];
      R     DIX [AR2,P#35.5];
      A     DIX [AR2,P#42.4];
      AN    DIX [AR2,P#44.2];
      AN    DIX [AR2,P#44.3];
      S     DIX [AR2,P#44.2];
      JCN   M006;
      L     DID [AR2,P#52.0];
      T     DID [AR2,P#28.0];
      L     W#16#8051;
      T     DIW [AR2,P#24.0];
      L     0;
      T     DIW [AR2,P#26.0];
M006: NOP   0;
      A     DIX [AR2,P#42.4];
      A     DIX [AR2,P#44.2];
      AN    DIX [AR2,P#44.3];
      A(;
      L     DID [AR2,P#28.0];
      L     DID [AR2,P#6.0];
      ==D;
      );
      A(;
      L     W#16#5051;
      L     DIW [AR2,P#2.0];
      ==I;
      );
      A(;
      L     DIW [AR2,P#26.0];
      L     DIW [AR2,P#4.0];
      ==I;
      );
      S     DIX [AR2,P#44.3];
      A     DIX [AR2,P#42.4];
      A     DIX [AR2,P#44.2];
      A     DIX [AR2,P#44.3];
      A(;
      L     DID [AR2,P#52.0];
      L     DID [AR2,P#6.0];
      ==D;
      );
      AN    DIX [AR2,P#13.0];
      AN    DIX [AR2,P#13.1];
      AN    DIX [AR2,P#13.2];
      AN    DIX [AR2,P#13.3];
      AN    DIX [AR2,P#13.4];
      AN    DIX [AR2,P#13.5];
      AN    DIX [AR2,P#33.6];
      S     DIX [AR2,P#33.6];
      JCN   M007;
      L     0;
      T     DIW [AR2,P#24.0];
      T     DIW [AR2,P#26.0];
      T     DID [AR2,P#28.0];
M007: NOP   0;
      A     DIX [AR2,P#10.2];
      FP    DIX [AR2,P#47.1];
      A     DIX [AR2,P#42.4];
      A     DIX [AR2,P#44.2];
      A     DIX [AR2,P#44.3];
      A     DIX [AR2,P#33.6];
      R     DIX [AR2,P#33.6];
      R     DIX [AR2,P#42.4];
      R     DIX [AR2,P#44.2];
      R     DIX [AR2,P#44.3];
NETWORK
TITLE =
      A     DIX [AR2,P#42.5];
      FP    DIX [AR2,P#47.2];
      A     DIX [AR2,P#45.0];
      R     DIX [AR2,P#42.5];
      A     DIX [AR2,P#42.5];
      S     DIX [AR2,P#35.0];
      R     DIX [AR2,P#35.1];
      R     DIX [AR2,P#35.2];
      R     DIX [AR2,P#35.3];
      R     DIX [AR2,P#35.4];
      R     DIX [AR2,P#35.5];
      A     DIX [AR2,P#42.5];
      A     DIX [AR2,P#13.0];
      AN    DIX [AR2,P#13.1];
      AN    DIX [AR2,P#13.2];
      AN    DIX [AR2,P#13.3];
      AN    DIX [AR2,P#13.4];
      AN    DIX [AR2,P#13.5];
      AN    DIX [AR2,P#33.6];
      S     DIX [AR2,P#33.6];
      A     DIX [AR2,P#10.2];
      FP    DIX [AR2,P#47.3];
      A     DIX [AR2,P#42.5];
      A     DIX [AR2,P#33.6];
      R     DIX [AR2,P#33.6];
      R     DIX [AR2,P#42.5];
NETWORK
TITLE =
      A     DIX [AR2,P#43.0];
      A     DIX [AR2,P#10.3];
      AN    DIX [AR2,P#15.7];
      =     DIX [AR2,P#32.1];
      A     DIX [AR2,P#43.1];
      A     DIX [AR2,P#10.3];
      AN    DIX [AR2,P#15.6];
      =     DIX [AR2,P#32.0];
NETWORK
TITLE =
      A     DIX [AR2,P#42.6];
      FP    DIX [AR2,P#47.4];
      S     DIX [AR2,P#32.3];
      A     DIX [AR2,P#10.3];
      FP    DIX [AR2,P#47.5];
      R     DIX [AR2,P#32.3];
      R     DIX [AR2,P#42.6];
NETWORK
TITLE =
      L     DIW [AR2,P#0.0];
      SLD   3;
      T     LD 28;
      L     P#DIX 24.0;
      T     LD 36;
      L     9;
M008: T     LW 34;
      L     DIW [LD 36];
      T     PQW [LD 28];
      L     LD 28;
      L     P#2.0;
      +D;
      T     LD 28;
      L     LD 36;
      L     P#2.0;
      +D;
      T     LD 36;
      L     LW 34;
      LOOP  M008;
END_FUNCTION_BLOCK

FUNCTION_BLOCK "BALLUFF"	// FB 20
AUTHOR : Salvati
VERSION : 0.1
BEGIN
// (block stored without names or comments; labels and parameter names are numbered)
NETWORK
TITLE =
      TAR1  LD 0;
      TAR2  LD 4;
      LAR1  P#L 8.0;
      L     B#16#10;
      T     LB [AR1,P#0.0];
      L     B#16#2;
      T     LB [AR1,P#1.0];
      L     6;
      T     LW [AR1,P#2.0];
      L     0;
      T     LW [AR1,P#4.0];
      L     DIW 0;
      SLD   3;
      L     P#I 0.0;
      +D;
      T     LD [AR1,P#6.0];
      LAR1  P#L 18.0;
      L     B#16#10;
      T     LB [AR1,P#0.0];
      L     B#16#2;
      T     LB [AR1,P#1.0];
      L     6;
      T     LW [AR1,P#2.0];
      L     0;
      T     LW [AR1,P#4.0];
      L     P#DIX 2.0;
      T     LD [AR1,P#6.0];
      BLD   7;
      UC    "BLKMOV";
      {     P#L 8.0, P#L 34.0, P#L 18.0 };
      BLD   8;
      LAR1  LD 0;
      LAR2  LD 4;
NETWORK
TITLE =
      TAR1  LD 0;
      TAR2  LD 4;
      LAR1  P#L 8.0;
      L     B#16#10;
      T     LB [AR1,P#0.0];
      L     B#16#2;
      T     LB [AR1,P#1.0];
      L     6;
      T     LW [AR1,P#2.0];
      L     0;
      T     LW [AR1,P#4.0];
      L     DIW 0;
      SLD   3;
      L     P#Q 0.0;
      +D;
      T     LD [AR1,P#6.0];
      LAR1  P#L 18.0;
      L     B#16#10;
      T     LB [AR1,P#0.0];
      L     B#16#2;
      T     LB [AR1,P#1.0];
      L     6;
      T     LW [AR1,P#2.0];
      L     0;
      T     LW [AR1,P#4.0];
      L     P#DIX 8.0;
      T     LD [AR1,P#6.0];
      BLD   7;
      UC    "BLKMOV";
      {     P#L 8.0, P#L 34.0, P#L 18.0 };
      BLD   8;
      LAR1  LD 0;
      LAR2  LD 4;
NETWORK
TITLE =
      A     DIX 14.3;
      A     "Clock_P";
      JCN   M001;
      L     DIB 18;
      L     1;
      +I;
      T     DIB 18;
M001: NOP   0;
      A     DIX 14.0;
      AN    DIX 15.0;
      AN    DIX 14.3;
      S     DIX 14.3;
      R     DIX 8.4;
      JCN   M002;
      L     0;
      T     DIB 18;
M002: NOP   0;
      A     DIX 14.0;
      A     DIX 14.3;
      AN    DIX 2.4;
      AN    DIX 14.4;
      S     DIX 14.4;
      A     DIX 14.0;
      A     DIX 14.4;
      A     DIX 2.7;
      A     DIX 2.0;
      AN    DIX 14.5;
      S     DIX 14.5;
      R     DIX 14.1;
      R     DIX 14.2;
      S     DIX 8.0;
      R     DIX 8.7;
      JC    M003;
      JU    M004;
M003: NOP   0;
      L     0;
      T     DIB 10;
      T     DIB 11;
      T     DIB 13;
      L     1;
      T     DIB 12;
      L     1;
      T     DIB 9;
M004: NOP   0;
      A     DIX 14.0;
      A     DIX 14.5;
      A     DIX 2.1;
      A     DIX 2.3;
      O;
      A(;
      L     DIB 18;
      L     10;
      >=I;
      );
      R     DIX 14.3;
      R     DIX 14.4;
      R     DIX 14.5;
      R     DIX 8.0;
      R     DIX 14.0;
      S     DIX 14.2;
      JCN   M005;
      L     0;
      T     DIB 18;
M005: NOP   0;
      A     DIX 14.0;
      A     DIX 14.5;
      A     DIX 2.1;
      A     DIX 2.2;
      R     DIX 14.3;
      R     DIX 14.4;
      R     DIX 14.5;
      R     DIX 8.0;
      R     DIX 14.0;
      S     DIX 14.1;
      JC    M006;
      JU    M007;
M006: L     DIB 3;
      T     DIB 16;
M007: NOP   0;
NETWORK
TITLE =
      A     DIX 15.3;
      A     "Clock_P";
      JCN   M008;
      L     DIB 18;
      L     1;
      +I;
      T     DIB 18;
M008: NOP   0;
      A     DIX 15.0;
      AN    DIX 14.0;
      AN    DIX 15.3;
      S     DIX 15.3;
      R     DIX 8.4;
      JCN   M009;
      L     0;
      T     DIB 18;
M009: NOP   0;
      A     DIX 15.0;
      A     DIX 15.3;
      AN    DIX 2.4;
      AN    DIX 15.4;
      S     DIX 15.4;
      A     DIX 15.0;
      A     DIX 15.4;
      A     DIX 2.7;
      A     DIX 2.0;
      AN    DIX 15.5;
      S     DIX 15.5;
      R     DIX 15.1;
      R     DIX 15.2;
      S     DIX 8.0;
      R     DIX 8.7;
      JC    M010;
      JU    M011;
M010: NOP   0;
      L     0;
      T     DIB 10;
      T     DIB 11;
      T     DIB 13;
      L     1;
      T     DIB 12;
      L     2;
      T     DIB 9;
M011: NOP   0;
      A     DIX 15.0;
      A     DIX 15.5;
      A     DIX 2.1;
      A     DIX 2.5;
      AN    DIX 15.6;
      S     DIX 15.6;
      S     DIX 8.6;
      JC    M012;
      JU    M013;
M012: NOP   0;
      L     DIB 17;
      T     DIB 9;
M013: NOP   0;
      A     DIX 15.0;
      A     DIX 15.6;
      A     DIX 2.1;
      A     DIX 2.3;
      O;
      A(;
      L     DIB 18;
      L     10;
      >=I;
      );
      R     DIX 15.3;
      R     DIX 15.4;
      R     DIX 15.5;
      R     DIX 15.6;
      R     DIX 8.0;
      R     DIX 8.6;
      R     DIX 15.0;
      S     DIX 15.2;
      JCN   M014;
      L     0;
      T     DIB 18;
M014: NOP   0;
      A     DIX 15.0;
      A     DIX 15.6;
      A     DIX 2.1;
      A     DIX 2.2;
      R     DIX 15.3;
      R     DIX 15.4;
      R     DIX 15.5;
      R     DIX 15.6;
      R     DIX 8.0;
      R     DIX 8.6;
      R     DIX 15.0;
      S     DIX 15.1;
NETWORK
TITLE =
      A     DIX 20.3;
      A     "Clock_P";
      JCN   M015;
      L     DIB 24;
      L     1;
      +I;
      T     DIB 24;
M015: NOP   0;
      A     DIX 20.0;
      AN    DIX 21.0;
      AN    DIX 14.0;
      AN    DIX 15.0;
      AN    DIX 20.3;
      S     DIX 20.3;
      S     DIX 8.4;
      JCN   M016;
      L     0;
      T     DIB 24;
M016: NOP   0;
      A     DIX 20.0;
      A     DIX 20.3;
      A     DIX 2.4;
      AN    DIX 20.4;
      S     DIX 20.4;
      A     DIX 20.0;
      A     DIX 20.4;
      A     DIX 2.7;
      A     DIX 2.0;
      AN    DIX 20.5;
      S     DIX 20.5;
      R     DIX 20.1;
      R     DIX 20.2;
      S     DIX 8.0;
      R     DIX 8.7;
      JC    M017;
      JU    M018;
M017: NOP   0;
      L     0;
      T     DIB 10;
      T     DIB 11;
      T     DIB 13;
      L     1;
      T     DIB 12;
      L     1;
      T     DIB 9;
M018: NOP   0;
      A     DIX 20.0;
      A     DIX 20.5;
      A     DIX 2.1;
      A     DIX 2.3;
      O;
      A(;
      L     DIB 24;
      L     10;
      >=I;
      );
      R     DIX 20.3;
      R     DIX 20.4;
      R     DIX 20.5;
      R     DIX 8.0;
      R     DIX 20.0;
      S     DIX 20.2;
      JCN   M019;
      L     0;
      T     DIB 24;
M019: NOP   0;
      A     DIX 20.0;
      A     DIX 20.5;
      A     DIX 2.1;
      A     DIX 2.2;
      R     DIX 20.3;
      R     DIX 20.4;
      R     DIX 20.5;
      R     DIX 8.0;
      R     DIX 20.0;
      S     DIX 20.1;
      JC    M020;
      JU    M021;
M020: L     DIB 3;
      T     DIB 22;
M021: NOP   0;
NETWORK
TITLE =
      A     DIX 21.3;
      A     "Clock_P";
      JCN   M022;
      L     DIB 24;
      L     1;
      +I;
      T     DIB 24;
M022: NOP   0;
      A     DIX 21.0;
      AN    DIX 20.0;
      AN    DIX 14.0;
      AN    DIX 15.0;
      AN    DIX 21.3;
      S     DIX 21.3;
      S     DIX 8.4;
      JCN   M023;
      L     0;
      T     DIB 24;
M023: NOP   0;
      A     DIX 21.0;
      A     DIX 21.3;
      A     DIX 2.4;
      AN    DIX 21.4;
      S     DIX 21.4;
      A     DIX 21.0;
      A     DIX 21.4;
      A     DIX 2.7;
      A     DIX 2.0;
      AN    DIX 21.5;
      S     DIX 21.5;
      R     DIX 21.1;
      R     DIX 21.2;
      S     DIX 8.0;
      R     DIX 8.7;
      JC    M024;
      JU    M025;
M024: NOP   0;
      L     0;
      T     DIB 10;
      T     DIB 11;
      T     DIB 13;
      L     1;
      T     DIB 12;
      L     2;
      T     DIB 9;
M025: NOP   0;
      A     DIX 21.0;
      A     DIX 21.5;
      A     DIX 2.1;
      A     DIX 2.5;
      AN    DIX 21.6;
      S     DIX 21.6;
      S     DIX 8.6;
      JC    M026;
      JU    M027;
M026: NOP   0;
      L     DIB 23;
      T     DIB 9;
M027: NOP   0;
      A     DIX 21.0;
      A     DIX 21.6;
      A     DIX 2.1;
      A     DIX 2.3;
      O;
      A(;
      L     DIB 24;
      L     10;
      >=I;
      );
      R     DIX 21.3;
      R     DIX 21.4;
      R     DIX 21.5;
      R     DIX 21.6;
      R     DIX 8.0;
      R     DIX 8.6;
      R     DIX 21.0;
      S     DIX 21.2;
      JCN   M028;
      L     0;
      T     DIB 24;
M028: NOP   0;
      A     DIX 21.0;
      A     DIX 21.6;
      A     DIX 2.1;
      A     DIX 2.2;
      R     DIX 21.3;
      R     DIX 21.4;
      R     DIX 21.5;
      R     DIX 21.6;
      R     DIX 8.0;
      R     DIX 8.6;
      R     DIX 21.0;
      S     DIX 21.1;
NETWORK
TITLE =
      TAR1  LD 0;
      TAR2  LD 4;
      LAR1  P#L 8.0;
      L     B#16#10;
      T     LB [AR1,P#0.0];
      L     B#16#2;
      T     LB [AR1,P#1.0];
      L     6;
      T     LW [AR1,P#2.0];
      L     0;
      T     LW [AR1,P#4.0];
      L     P#DIX 8.0;
      T     LD [AR1,P#6.0];
      LAR1  P#L 18.0;
      L     B#16#10;
      T     LB [AR1,P#0.0];
      L     B#16#2;
      T     LB [AR1,P#1.0];
      L     6;
      T     LW [AR1,P#2.0];
      L     0;
      T     LW [AR1,P#4.0];
      L     DIW 0;
      SLD   3;
      L     P#Q 0.0;
      +D;
      T     LD [AR1,P#6.0];
      BLD   7;
      UC    "BLKMOV";
      {     P#L 8.0, P#L 34.0, P#L 18.0 };
      BLD   8;
      LAR1  LD 0;
      LAR2  LD 4;
END_FUNCTION_BLOCK

FUNCTION_BLOCK "FB24 - Gestione Mov Assi"	// FB 24
VERSION : 0.1
VAR_INPUT
  INDIRIZZO_INIZIALE_E_A : DINT ;
  OK_FOR_COMMANDS : BOOL ;
  RESET_ALLARMI : BOOL ;
  STOP : BOOL ;
  TARGET_POSIZIONE : DINT ;
  TARGET_INCREMENTALE : DINT ;
  OVERRIDE : INT ;
  JOG_PIU : BOOL ;
  JOG_MENO : BOOL ;
  IN_PKE : WORD ;
  IN_IND : WORD ;
  IN_PWE : DINT ;
  ASSE_SU_HOME : BOOL ;
END_VAR
VAR_OUTPUT
  OUT_PKE : WORD ;
  OUT_IND : WORD ;
  OUT_PWE : DINT ;
  POSIZIONE_ATTUALE : DINT ;
  POSIZIONE_RAGGIUNTA : BOOL ;
  HOME_OK : BOOL ;
  RIPOSIZIONAMENTO_OK : BOOL ;
  ASSE_FERMO_NO_JOB : BOOL ;
  AZIONAMENTO_OK : BOOL ;
  AZIONAMENTO_FAULT : BOOL ;
  CAMMA_DI_RIFERIMENTO : BOOL ;
  OLTRECORSA_NEGATIVO : BOOL ;
  OLTRECORSA_POSITIVO : BOOL ;
  FINECORSA_SOFTWARE_NEG : BOOL ;
  FINECORSA_SOFTWARE_POS : BOOL ;
  FRENO : BOOL ;
END_VAR
VAR_IN_OUT
  START_ASSOLUTO : BOOL ;
  START_INCREMENTALE : BOOL ;
  START_HOME : BOOL ;
  START_RIPOSIZIONAMENTO : BOOL ;
END_VAR
VAR
  SCELTA_BLOCCO : WORD ;
  BLOCCO_ATTUALE : WORD ;
  INVIA_JOB1 : BOOL ;
  JOB1_ULTIMATO : BOOL ;
  INVIA_JOB2 : BOOL ;
  JOB2_ULTIMATO : BOOL ;
  GIA_IN_POSIZIONE : BOOL ;
  PACO1 : STRUCT
   STAT41 : BOOL ;
   STAT42 : BOOL ;
   STAT43 : BOOL ;
   STAT44 : BOOL ;
   STAT45 : BOOL ;
   STAT46 : BOOL ;
   STAT47 : BOOL ;
   STAT48 : BOOL ;
   STAT49 : BOOL ;
   STAT50 : BOOL ;
   STAT51 : BOOL ;
   STAT52 : BOOL ;
   STAT53 : BOOL ;
   STAT54 : BOOL ;
   STAT55 : BOOL ;
   STAT56 : BOOL ;
  END_STRUCT ;
  PAST1 : STRUCT
   STAT58 : BOOL ;
   STAT59 : BOOL ;
   STAT60 : BOOL ;
   STAT61 : BOOL ;
   STAT62 : BOOL ;
   STAT63 : BOOL ;
   STAT64 : BOOL ;
   STAT65 : BOOL ;
   STAT66 : BOOL ;
   STAT67 : BOOL ;
   STAT68 : BOOL ;
   STAT69 : BOOL ;
   STAT70 : BOOL ;
   STAT71 : BOOL ;
   STAT72 : BOOL ;
   STAT73 : BOOL ;
  END_STRUCT ;
  DIGin : STRUCT
   STAT75 : BOOL ;
   STAT76 : BOOL ;
   STAT77 : BOOL ;
   STAT78 : BOOL ;
   STAT79 : BOOL ;
   STAT80 : BOOL ;
   STAT81 : BOOL ;
   STAT82 : BOOL ;
   STAT83 : BOOL ;
   STAT84 : BOOL ;
   STAT85 : BOOL ;
   STAT86 : BOOL ;
   STAT87 : BOOL ;
   STAT88 : BOOL ;
   STAT89 : BOOL ;
   STAT90 : BOOL ;
  END_STRUCT ;
  AUX1 : BOOL ;
  AUX2 : BOOL ;
  AUX3 : BOOL ;
  AUX4 : BOOL ;
  AUX5 : BOOL ;
  AUX6 : BOOL ;
  AUX7 : BOOL ;
  VERIFICA_SPOSTAMENTO : DINT ;
  PAST2 : STRUCT
   STAT100 : BOOL ;
   STAT101 : BOOL ;
   STAT102 : BOOL ;
   STAT103 : BOOL ;
   STAT104 : BOOL ;
   STAT105 : BOOL ;
   STAT106 : BOOL ;
   STAT107 : BOOL ;
   STAT108 : BOOL ;
   STAT109 : BOOL ;
   STAT110 : BOOL ;
   STAT111 : BOOL ;
   STAT112 : BOOL ;
   STAT113 : BOOL ;
   STAT114 : BOOL ;
   STAT115 : BOOL ;
  END_STRUCT ;
  POS_PAST : STRUCT
   STAT117 : BOOL ;
   STAT118 : BOOL ;
   STAT119 : BOOL ;
   STAT120 : BOOL ;
   STAT121 : BOOL ;
   STAT122 : BOOL ;
   STAT123 : BOOL ;
   STAT124 : BOOL ;
   STAT125 : BOOL ;
   STAT126 : BOOL ;
   STAT127 : BOOL ;
   STAT128 : BOOL ;
   STAT129 : BOOL ;
   STAT130 : BOOL ;
   STAT131 : BOOL ;
   STAT132 : BOOL ;
  END_STRUCT ;
END_VAR
BEGIN
NETWORK
TITLE =
      L     #INDIRIZZO_INIZIALE_E_A;
      L     8;
      +I;
      SLD   3;
      T     "MD100";
      L     PIW ["MD100"];
      T     DIW 52;
      L     "MD100";
      SRW   3;
      L     2;
      +D;
      SLW   3;
      T     "MD100";
      L     PIW ["MD100"];
      T     #BLOCCO_ATTUALE;
      L     "MD100";
      SRW   3;
      L     2;
      +D;
      SLW   3;
      T     "MD100";
      L     PIW ["MD100"];
      T     DIW 64;
      L     "MD100";
      SRW   3;
      L     2;
      +D;
      SLW   3;
      T     "MD100";
      L     PIW ["MD100"];
      T     DIW 62;
      L     "MD100";
      SRW   3;
      L     2;
      +D;
      SLW   3;
      T     "MD100";
      L     PID ["MD100"];
      T     #POSIZIONE_ATTUALE;
      L     "MD100";
      SRW   3;
      L     4;
      +D;
      SLW   3;
      T     "MD100";
      L     PIW ["MD100"];
      T     DIW 54;
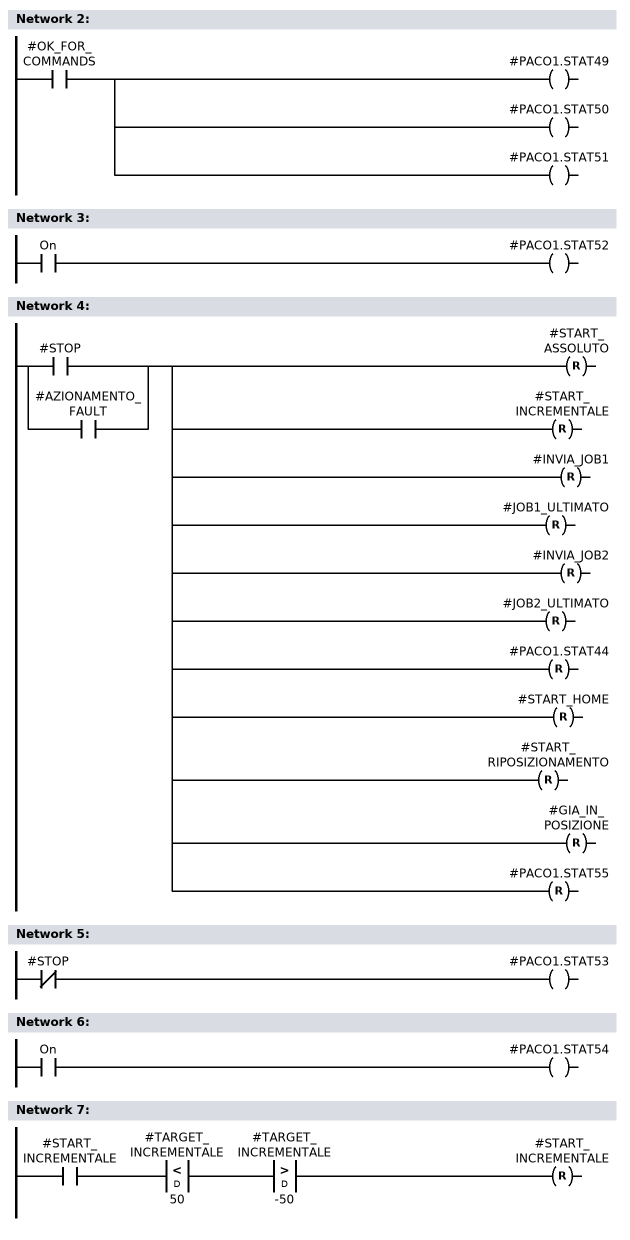
NETWORK
TITLE =
      A     #OK_FOR_COMMANDS;
      =     #PACO1.STAT49;
      =     #PACO1.STAT50;
      =     #PACO1.STAT51;
NETWORK
TITLE =
      A     "On";
      =     #PACO1.STAT52;
NETWORK
TITLE =
      O     #STOP;
      O     #AZIONAMENTO_FAULT;
      R     #START_ASSOLUTO;
      R     #START_INCREMENTALE;
      R     #INVIA_JOB1;
      R     #JOB1_ULTIMATO;
      R     #INVIA_JOB2;
      R     #JOB2_ULTIMATO;
      R     #PACO1.STAT44;
      R     #START_HOME;
      R     #START_RIPOSIZIONAMENTO;
      R     #GIA_IN_POSIZIONE;
      R     #PACO1.STAT55;
NETWORK
TITLE =
      AN    #STOP;
      =     #PACO1.STAT53;
NETWORK
TITLE =
      A     "On";
      =     #PACO1.STAT54;
NETWORK
TITLE =
      A     #START_INCREMENTALE;
      A(;
      L     #TARGET_INCREMENTALE;
      L     50;
      <D;
      );
      A(;
      L     #TARGET_INCREMENTALE;
      L     -50;
      >D;
      );
      R     #START_INCREMENTALE;
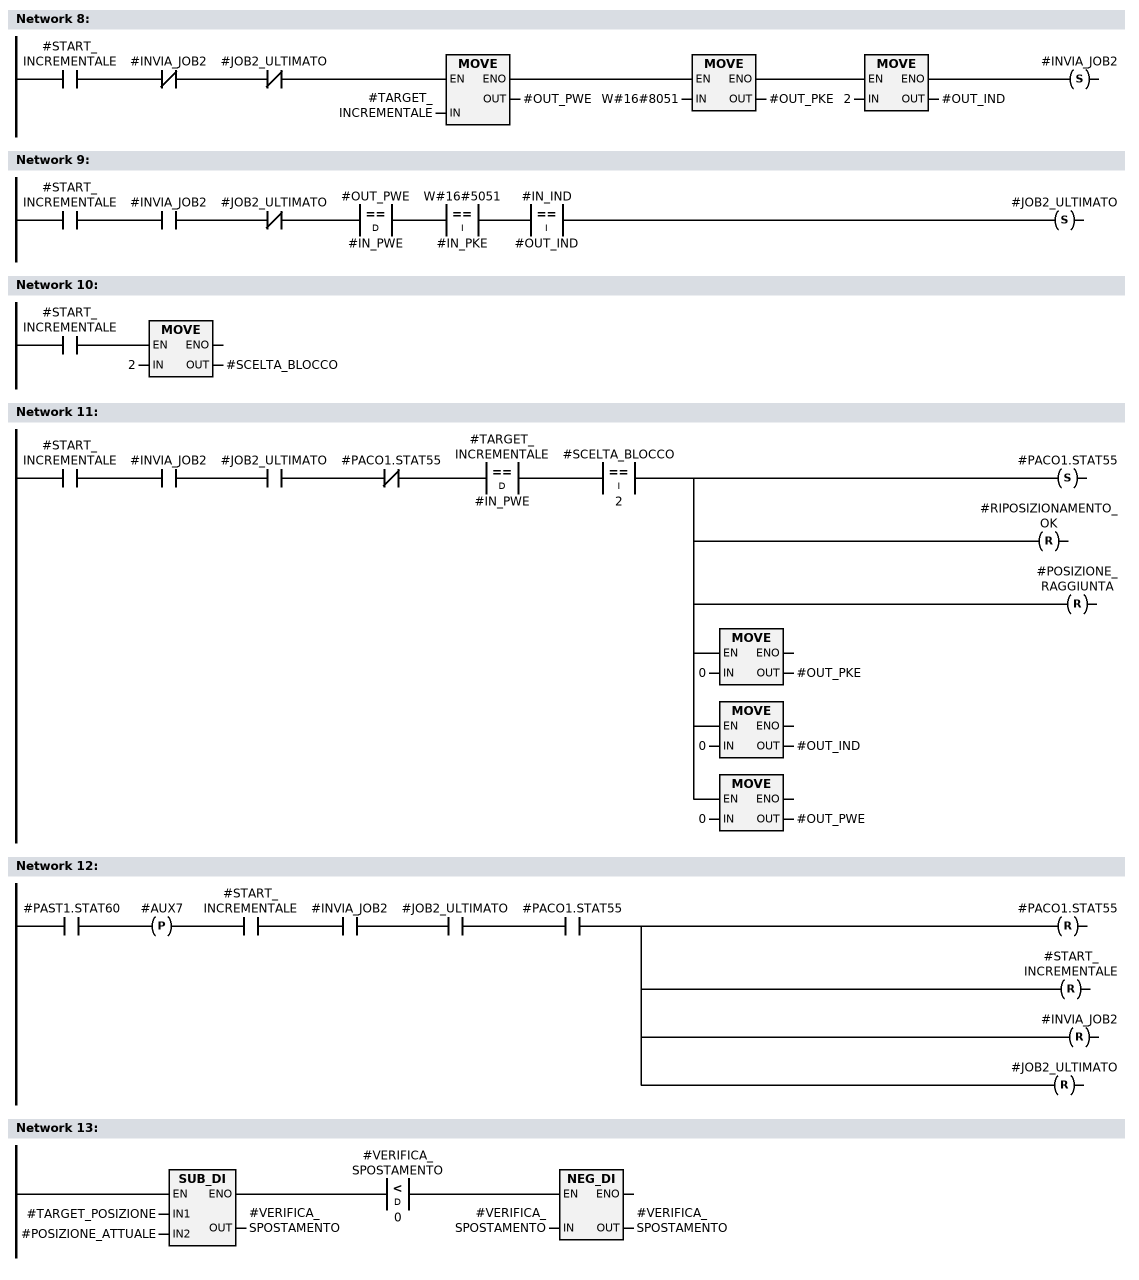
NETWORK
TITLE =
      A(;
      A(;
      A     #START_INCREMENTALE;
      AN    #INVIA_JOB2;
      AN    #JOB2_ULTIMATO;
      JNB   _001;
      L     #TARGET_INCREMENTALE;
      T     #OUT_PWE;
      SET;
      SAVE;
      CLR;
_001: A     BR;
      );
      JNB   _002;
      L     W#16#8051;
      T     #OUT_PKE;
      SET;
      SAVE;
      CLR;
_002: A     BR;
      );
      JNB   _003;
      L     2;
      T     #OUT_IND;
      SET;
      SAVE;
      CLR;
_003: A     BR;
      S     #INVIA_JOB2;
NETWORK
TITLE =
      A     #START_INCREMENTALE;
      A     #INVIA_JOB2;
      AN    #JOB2_ULTIMATO;
      A(;
      L     #OUT_PWE;
      L     #IN_PWE;
      ==D;
      );
      A(;
      L     W#16#5051;
      L     #IN_PKE;
      ==I;
      );
      A(;
      L     #IN_IND;
      L     #OUT_IND;
      ==I;
      );
      S     #JOB2_ULTIMATO;
NETWORK
TITLE =
      A     #START_INCREMENTALE;
      JNB   _004;
      L     2;
      T     #SCELTA_BLOCCO;
_004: NOP   0;
NETWORK
TITLE =
      A     #START_INCREMENTALE;
      A     #INVIA_JOB2;
      A     #JOB2_ULTIMATO;
      AN    #PACO1.STAT55;
      A(;
      L     #TARGET_INCREMENTALE;
      L     #IN_PWE;
      ==D;
      );
      A(;
      L     #SCELTA_BLOCCO;
      L     2;
      ==I;
      );
      =     L 0.0;
      A     L 0.0;
      BLD   102;
      S     #PACO1.STAT55;
      A     L 0.0;
      BLD   102;
      R     #RIPOSIZIONAMENTO_OK;
      A     L 0.0;
      BLD   102;
      R     #POSIZIONE_RAGGIUNTA;
      A     L 0.0;
      JNB   _005;
      L     0;
      T     #OUT_PKE;
_005: NOP   0;
      A     L 0.0;
      JNB   _006;
      L     0;
      T     #OUT_IND;
_006: NOP   0;
      A     L 0.0;
      JNB   _007;
      L     0;
      T     #OUT_PWE;
_007: NOP   0;
NETWORK
TITLE =
      A     #PAST1.STAT60;
      FP    #AUX7;
      A     #START_INCREMENTALE;
      A     #INVIA_JOB2;
      A     #JOB2_ULTIMATO;
      A     #PACO1.STAT55;
      R     #PACO1.STAT55;
      R     #START_INCREMENTALE;
      R     #INVIA_JOB2;
      R     #JOB2_ULTIMATO;
NETWORK
TITLE =
      A(;
      L     #TARGET_POSIZIONE;
      L     #POSIZIONE_ATTUALE;
      -D;
      T     #VERIFICA_SPOSTAMENTO;
      AN    OV;
      SAVE;
      CLR;
      A     BR;
      );
      A(;
      L     #VERIFICA_SPOSTAMENTO;
      L     0;
      <D;
      );
      JNB   _008;
      L     #VERIFICA_SPOSTAMENTO;
      NEGD;
      T     #VERIFICA_SPOSTAMENTO;
_008: NOP   0;
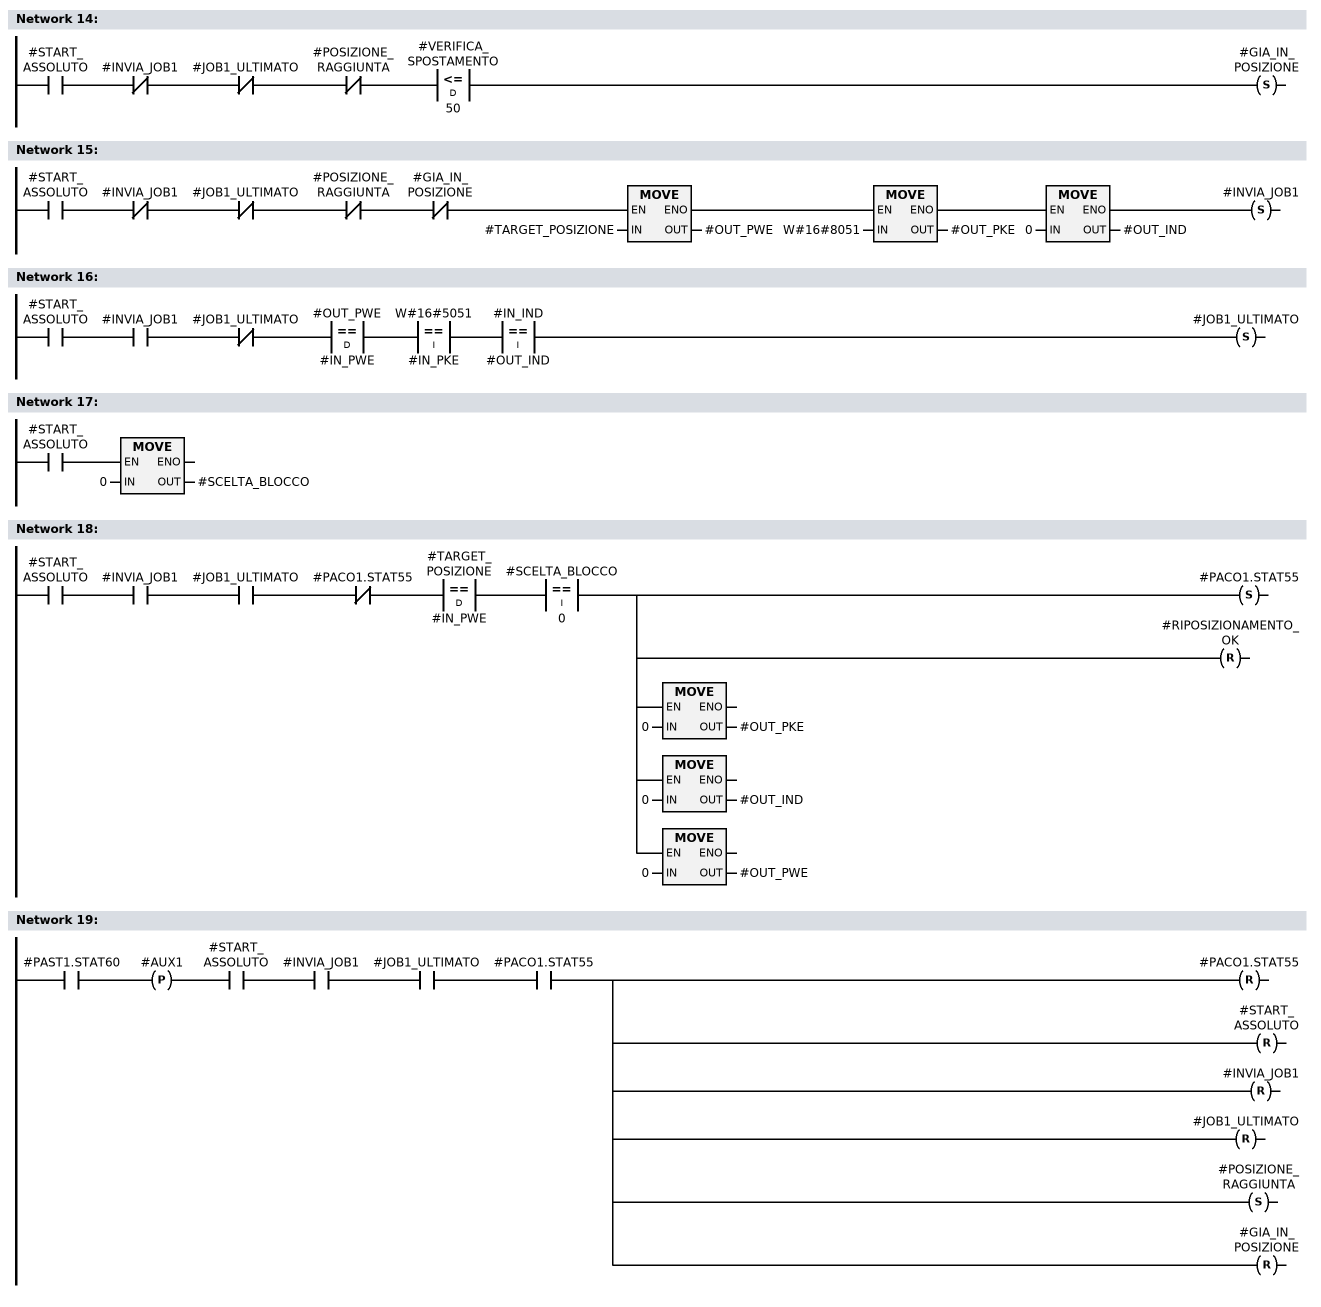
NETWORK
TITLE =
      A     #START_ASSOLUTO;
      AN    #INVIA_JOB1;
      AN    #JOB1_ULTIMATO;
      AN    #POSIZIONE_RAGGIUNTA;
      A(;
      L     #VERIFICA_SPOSTAMENTO;
      L     50;
      <=D;
      );
      S     #GIA_IN_POSIZIONE;
NETWORK
TITLE =
      A(;
      A(;
      A     #START_ASSOLUTO;
      AN    #INVIA_JOB1;
      AN    #JOB1_ULTIMATO;
      AN    #POSIZIONE_RAGGIUNTA;
      AN    #GIA_IN_POSIZIONE;
      JNB   _009;
      L     #TARGET_POSIZIONE;
      T     #OUT_PWE;
      SET;
      SAVE;
      CLR;
_009: A     BR;
      );
      JNB   _00a;
      L     W#16#8051;
      T     #OUT_PKE;
      SET;
      SAVE;
      CLR;
_00a: A     BR;
      );
      JNB   _00b;
      L     0;
      T     #OUT_IND;
      SET;
      SAVE;
      CLR;
_00b: A     BR;
      S     #INVIA_JOB1;
NETWORK
TITLE =
      A     #START_ASSOLUTO;
      A     #INVIA_JOB1;
      AN    #JOB1_ULTIMATO;
      A(;
      L     #OUT_PWE;
      L     #IN_PWE;
      ==D;
      );
      A(;
      L     W#16#5051;
      L     #IN_PKE;
      ==I;
      );
      A(;
      L     #IN_IND;
      L     #OUT_IND;
      ==I;
      );
      S     #JOB1_ULTIMATO;
NETWORK
TITLE =
      A     #START_ASSOLUTO;
      JNB   _00c;
      L     0;
      T     #SCELTA_BLOCCO;
_00c: NOP   0;
NETWORK
TITLE =
      A     #START_ASSOLUTO;
      A     #INVIA_JOB1;
      A     #JOB1_ULTIMATO;
      AN    #PACO1.STAT55;
      A(;
      L     #TARGET_POSIZIONE;
      L     #IN_PWE;
      ==D;
      );
      A(;
      L     #SCELTA_BLOCCO;
      L     0;
      ==I;
      );
      =     L 0.0;
      A     L 0.0;
      BLD   102;
      S     #PACO1.STAT55;
      A     L 0.0;
      BLD   102;
      R     #RIPOSIZIONAMENTO_OK;
      A     L 0.0;
      JNB   _00d;
      L     0;
      T     #OUT_PKE;
_00d: NOP   0;
      A     L 0.0;
      JNB   _00e;
      L     0;
      T     #OUT_IND;
_00e: NOP   0;
      A     L 0.0;
      JNB   _00f;
      L     0;
      T     #OUT_PWE;
_00f: NOP   0;
NETWORK
TITLE =
      A     #PAST1.STAT60;
      FP    #AUX1;
      A     #START_ASSOLUTO;
      A     #INVIA_JOB1;
      A     #JOB1_ULTIMATO;
      A     #PACO1.STAT55;
      R     #PACO1.STAT55;
      R     #START_ASSOLUTO;
      R     #INVIA_JOB1;
      R     #JOB1_ULTIMATO;
      S     #POSIZIONE_RAGGIUNTA;
      R     #GIA_IN_POSIZIONE;
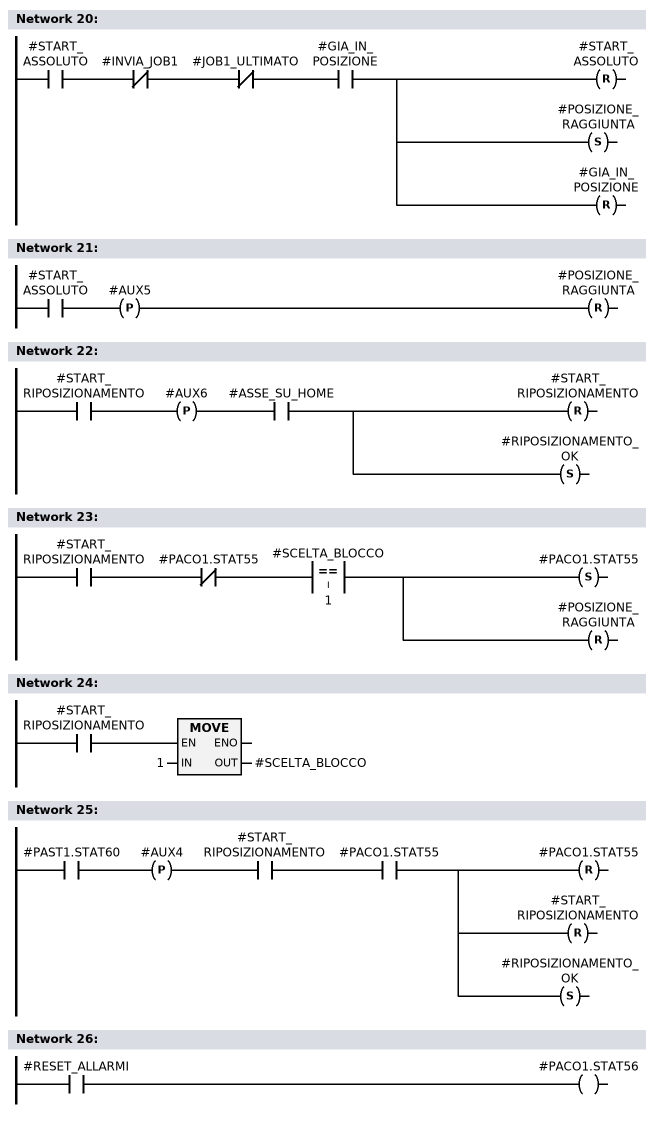
NETWORK
TITLE =
      A     #START_ASSOLUTO;
      AN    #INVIA_JOB1;
      AN    #JOB1_ULTIMATO;
      A     #GIA_IN_POSIZIONE;
      R     #START_ASSOLUTO;
      S     #POSIZIONE_RAGGIUNTA;
      R     #GIA_IN_POSIZIONE;
NETWORK
TITLE =
      A     #START_ASSOLUTO;
      FP    #AUX5;
      R     #POSIZIONE_RAGGIUNTA;
NETWORK
TITLE =
      A     #START_RIPOSIZIONAMENTO;
      FP    #AUX6;
      A     #ASSE_SU_HOME;
      R     #START_RIPOSIZIONAMENTO;
      S     #RIPOSIZIONAMENTO_OK;
NETWORK
TITLE =
      A     #START_RIPOSIZIONAMENTO;
      AN    #PACO1.STAT55;
      A(;
      L     #SCELTA_BLOCCO;
      L     1;
      ==I;
      );
      S     #PACO1.STAT55;
      R     #POSIZIONE_RAGGIUNTA;
NETWORK
TITLE =
      A     #START_RIPOSIZIONAMENTO;
      JNB   _010;
      L     1;
      T     #SCELTA_BLOCCO;
_010: NOP   0;
NETWORK
TITLE =
      A     #PAST1.STAT60;
      FP    #AUX4;
      A     #START_RIPOSIZIONAMENTO;
      A     #PACO1.STAT55;
      R     #PACO1.STAT55;
      R     #START_RIPOSIZIONAMENTO;
      S     #RIPOSIZIONAMENTO_OK;
NETWORK
TITLE =
      A     #RESET_ALLARMI;
      =     #PACO1.STAT56;
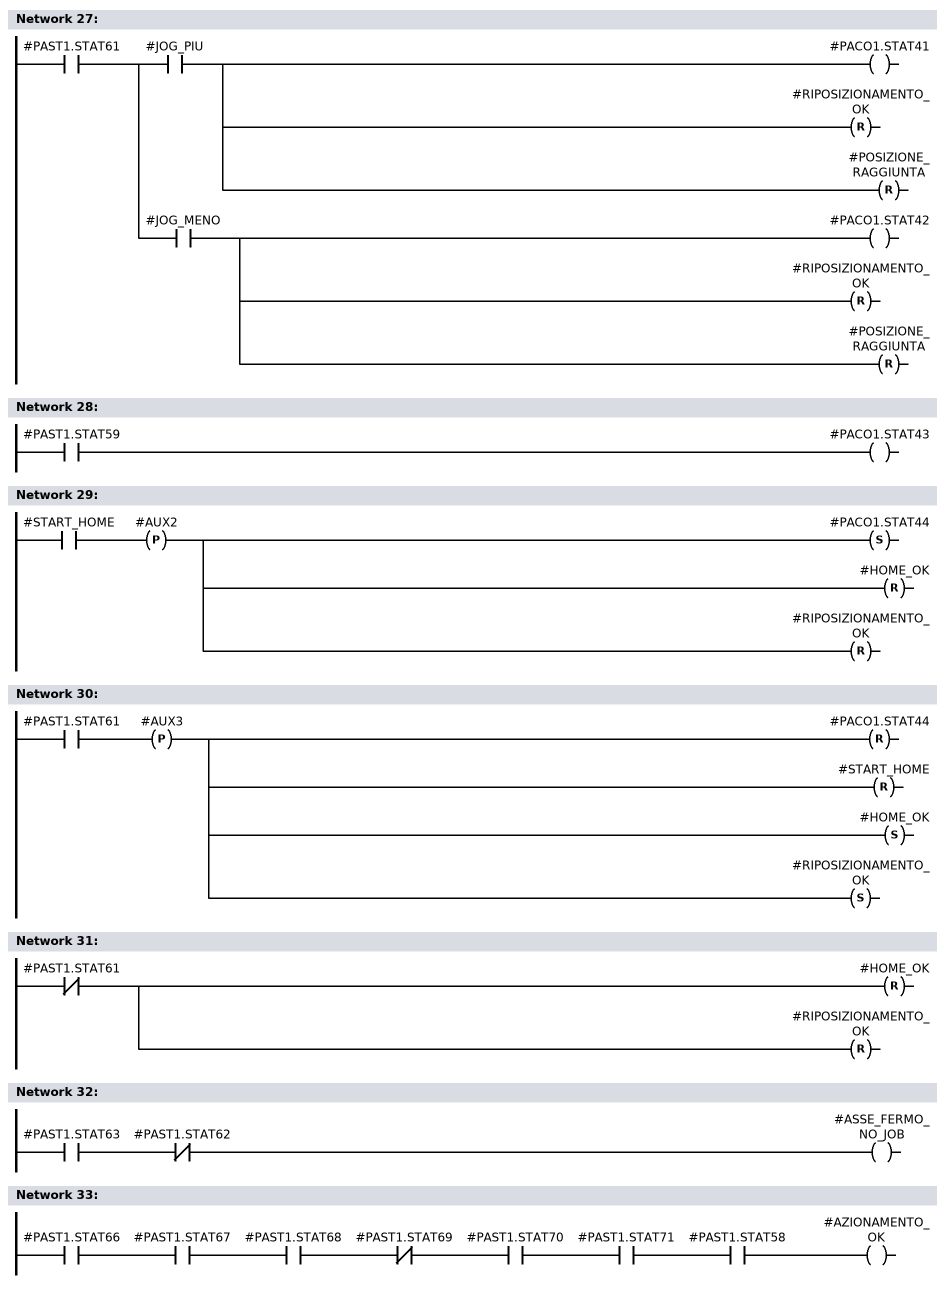
NETWORK
TITLE =
      A     #PAST1.STAT61;
      =     L 0.0;
      A     L 0.0;
      A     #JOG_PIU;
      =     #PACO1.STAT41;
      R     #RIPOSIZIONAMENTO_OK;
      R     #POSIZIONE_RAGGIUNTA;
      A     L 0.0;
      A     #JOG_MENO;
      =     #PACO1.STAT42;
      R     #RIPOSIZIONAMENTO_OK;
      R     #POSIZIONE_RAGGIUNTA;
NETWORK
TITLE =
      A     #PAST1.STAT59;
      =     #PACO1.STAT43;
NETWORK
TITLE =
      A     #START_HOME;
      FP    #AUX2;
      S     #PACO1.STAT44;
      R     #HOME_OK;
      R     #RIPOSIZIONAMENTO_OK;
NETWORK
TITLE =
      A     #PAST1.STAT61;
      FP    #AUX3;
      R     #PACO1.STAT44;
      R     #START_HOME;
      S     #HOME_OK;
      S     #RIPOSIZIONAMENTO_OK;
NETWORK
TITLE =
      AN    #PAST1.STAT61;
      R     #HOME_OK;
      R     #RIPOSIZIONAMENTO_OK;
NETWORK
TITLE =
      A     #PAST1.STAT63;
      AN    #PAST1.STAT62;
      =     #ASSE_FERMO_NO_JOB;
NETWORK
TITLE =
      A     #PAST1.STAT66;
      A     #PAST1.STAT67;
      A     #PAST1.STAT68;
      AN    #PAST1.STAT69;
      A     #PAST1.STAT70;
      A     #PAST1.STAT71;
      A     #PAST1.STAT58;
      =     #AZIONAMENTO_OK;
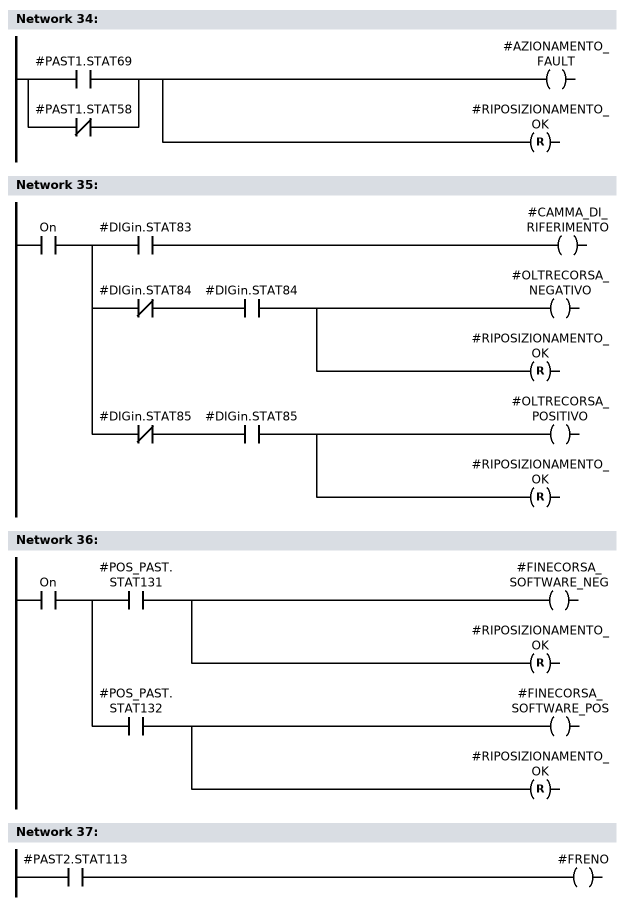
NETWORK
TITLE =
      O     #PAST1.STAT69;
      ON    #PAST1.STAT58;
      =     #AZIONAMENTO_FAULT;
      R     #RIPOSIZIONAMENTO_OK;
NETWORK
TITLE =
      A     "On";
      =     L 0.0;
      A     L 0.0;
      A     #DIGin.STAT83;
      =     #CAMMA_DI_RIFERIMENTO;
      A     L 0.0;
      AN    #DIGin.STAT84;
      A     #DIGin.STAT84;
      =     #OLTRECORSA_NEGATIVO;
      R     #RIPOSIZIONAMENTO_OK;
      A     L 0.0;
      AN    #DIGin.STAT85;
      A     #DIGin.STAT85;
      =     #OLTRECORSA_POSITIVO;
      R     #RIPOSIZIONAMENTO_OK;
NETWORK
TITLE =
      A     "On";
      =     L 0.0;
      A     L 0.0;
      A     #POS_PAST.STAT131;
      =     #FINECORSA_SOFTWARE_NEG;
      R     #RIPOSIZIONAMENTO_OK;
      A     L 0.0;
      A     #POS_PAST.STAT132;
      =     #FINECORSA_SOFTWARE_POS;
      R     #RIPOSIZIONAMENTO_OK;
NETWORK
TITLE =
      A     #PAST2.STAT113;
      =     #FRENO;
NETWORK
TITLE =
      L     #INDIRIZZO_INIZIALE_E_A;
      L     8;
      +I;
      SLD   3;
      T     "MD100";
      L     DIW 50;
      T     PQW ["MD100"];
      L     "MD100";
      SRW   3;
      L     2;
      +D;
      SLW   3;
      T     "MD100";
      L     #SCELTA_BLOCCO;
      T     PQW ["MD100"];
      L     "MD100";
      SRW   3;
      L     6;
      +D;
      SLW   3;
      T     "MD100";
      L     #OVERRIDE;
      T     PQW ["MD100"];
END_FUNCTION_BLOCK

// FC 7: know-how protected block, not included

FUNCTION "FC11 - STATUS" : VOID	// FC 11
VERSION : 0.1
VAR_TEMP
  TEMP0 : INT ;
END_VAR
BEGIN
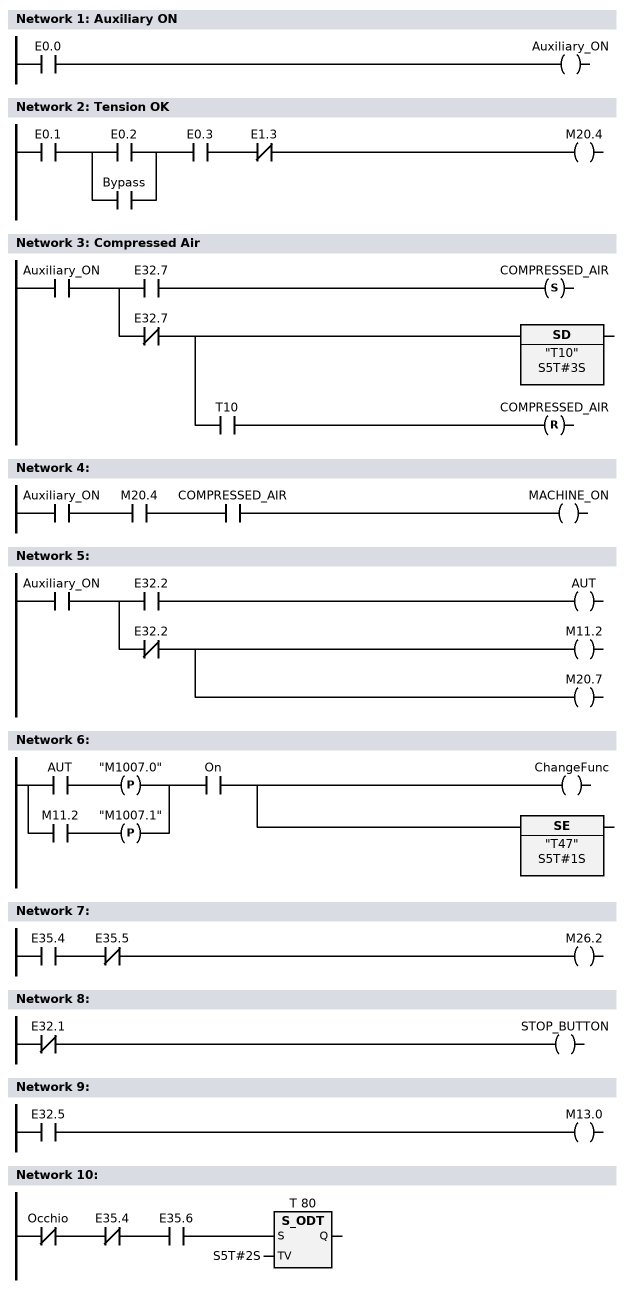
NETWORK
TITLE = Auxiliary ON
      A     "E0.0";
      =     "Auxiliary_ON";
NETWORK
TITLE = Tension OK
      A     "E0.1";
      A(;
      O     "E0.2";
      O     "Bypass";
      );
      A     "E0.3";
      AN    "E1.3";
      =     "M20.4";
NETWORK
TITLE = Compressed Air
      A     "Auxiliary_ON";
      =     L 2.0;
      A     L 2.0;
      A     "E32.7";
      S     "COMPRESSED_AIR";
      A     L 2.0;
      AN    "E32.7";
      =     L 2.1;
      A     L 2.1;
      BLD   102;
      L     S5T#3S;
      SD    "T10";
      A     L 2.1;
      A     "T10";
      R     "COMPRESSED_AIR";
NETWORK
TITLE =
      A     "Auxiliary_ON";
      A     "M20.4";
      A     "COMPRESSED_AIR";
      =     "MACHINE_ON";
NETWORK
TITLE =
      A     "Auxiliary_ON";
      =     L 2.0;
      A     L 2.0;
      A     "E32.2";
      =     "AUT";
      A     L 2.0;
      AN    "E32.2";
      =     "M11.2";
      =     "M20.7";
NETWORK
TITLE =
      A(;
      A     "AUT";
      FP    "M1007.0";
      O(;
      A     "M11.2";
      FP    "M1007.1";
      );
      );
      A     "On";
      =     "ChangeFunc";
      L     S5T#1S;
      SE    "T47";
NETWORK
TITLE =
      A     "E35.4";
      AN    "E35.5";
      =     "M26.2";
NETWORK
TITLE =
      AN    "E32.1";
      =     "STOP_BUTTON";
NETWORK
TITLE =
      A     "E32.5";
      =     "M13.0";
NETWORK
TITLE =
      AN    "Occhio";
      AN    "E35.4";
      A     "E35.6";
      L     S5T#2S;
      SD    T 80;
      NOP   0;
      NOP   0;
      NOP   0;
      NOP   0;
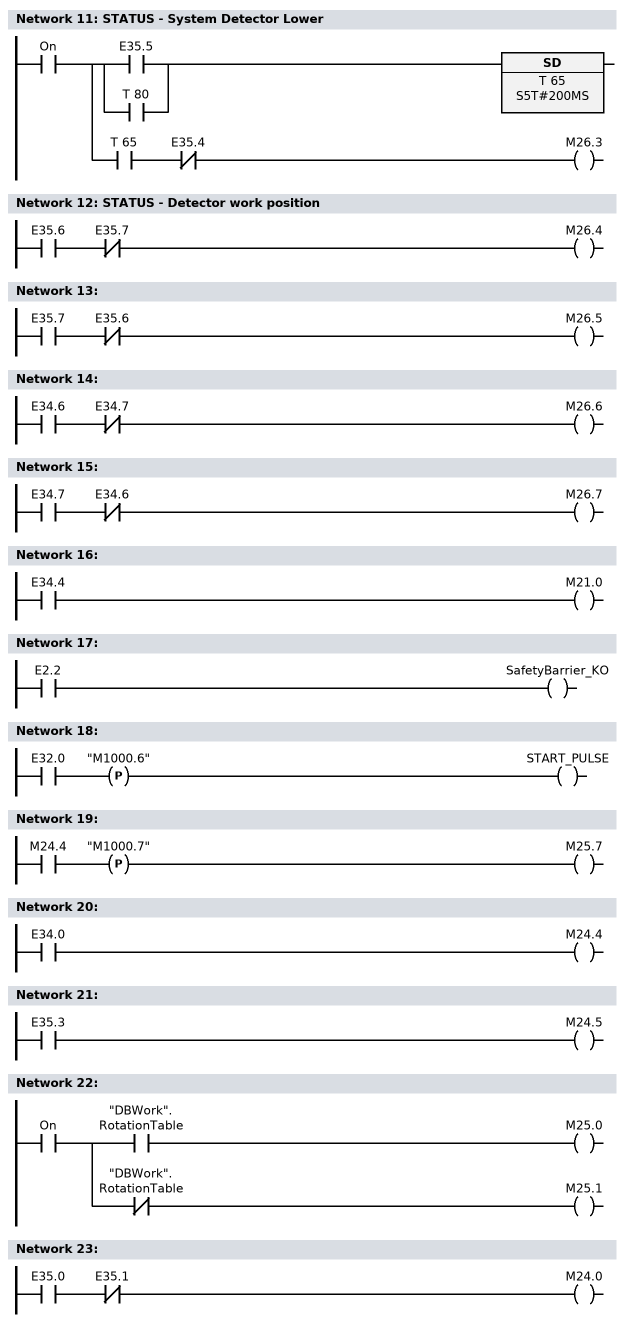
NETWORK
TITLE = STATUS - System Detector Lower
      A     "On";
      =     L 2.0;
      A     L 2.0;
      A(;
      O     "E35.5";
      O     T 80;
      );
      L     S5T#200MS;
      SD    T 65;
      A     L 2.0;
      A     T 65;
      AN    "E35.4";
      =     "M26.3";
NETWORK
TITLE = STATUS - Detector work position
      A     "E35.6";
      AN    "E35.7";
      =     "M26.4";
NETWORK
TITLE =
      A     "E35.7";
      AN    "E35.6";
      =     "M26.5";
NETWORK
TITLE =
      A     "E34.6";
      AN    "E34.7";
      =     "M26.6";
NETWORK
TITLE =
      A     "E34.7";
      AN    "E34.6";
      =     "M26.7";
NETWORK
TITLE =
      A     "E34.4";
      =     "M21.0";
NETWORK
TITLE =
      A     "E2.2";
      =     "SafetyBarrier_KO";
NETWORK
TITLE =
      A     "E32.0";
      FP    "M1000.6";
      =     "START_PULSE";
NETWORK
TITLE =
      A     "M24.4";
      FP    "M1000.7";
      =     "M25.7";
NETWORK
TITLE =
      A     "E34.0";
      =     "M24.4";
NETWORK
TITLE =
      A     "E35.3";
      =     "M24.5";
NETWORK
TITLE =
      A     "On";
      =     L 2.0;
      A     L 2.0;
      A     "DBWork".RotationTable;
      =     "M25.0";
      A     L 2.0;
      AN    "DBWork".RotationTable;
      =     "M25.1";
NETWORK
TITLE =
      A     "E35.0";
      AN    "E35.1";
      =     "M24.0";
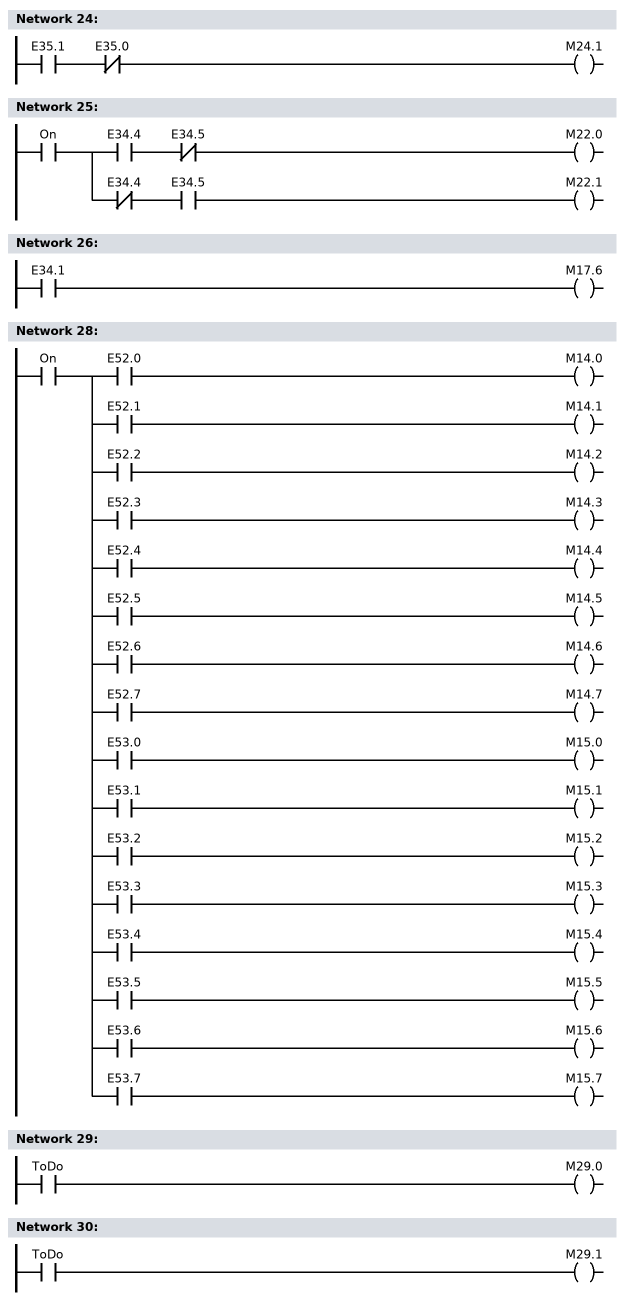
NETWORK
TITLE =
      A     "E35.1";
      AN    "E35.0";
      =     "M24.1";
NETWORK
TITLE =
      A     "On";
      =     L 2.0;
      A     L 2.0;
      A     "E34.4";
      AN    "E34.5";
      =     "M22.0";
      A     L 2.0;
      AN    "E34.4";
      A     "E34.5";
      =     "M22.1";
NETWORK
TITLE =
      A     "E34.1";
      =     "M17.6";
NETWORK
TITLE =
NETWORK
TITLE =
      A     "On";
      =     L 2.0;
      A     L 2.0;
      A     "E52.0";
      =     "M14.0";
      A     L 2.0;
      A     "E52.1";
      =     "M14.1";
      A     L 2.0;
      A     "E52.2";
      =     "M14.2";
      A     L 2.0;
      A     "E52.3";
      =     "M14.3";
      A     L 2.0;
      A     "E52.4";
      =     "M14.4";
      A     L 2.0;
      A     "E52.5";
      =     "M14.5";
      A     L 2.0;
      A     "E52.6";
      =     "M14.6";
      A     L 2.0;
      A     "E52.7";
      =     "M14.7";
      A     L 2.0;
      A     "E53.0";
      =     "M15.0";
      A     L 2.0;
      A     "E53.1";
      =     "M15.1";
      A     L 2.0;
      A     "E53.2";
      =     "M15.2";
      A     L 2.0;
      A     "E53.3";
      =     "M15.3";
      A     L 2.0;
      A     "E53.4";
      =     "M15.4";
      A     L 2.0;
      A     "E53.5";
      =     "M15.5";
      A     L 2.0;
      A     "E53.6";
      =     "M15.6";
      A     L 2.0;
      A     "E53.7";
      =     "M15.7";
NETWORK
TITLE =
      A     "ToDo";
      =     "M29.0";
NETWORK
TITLE =
      A     "ToDo";
      =     "M29.1";
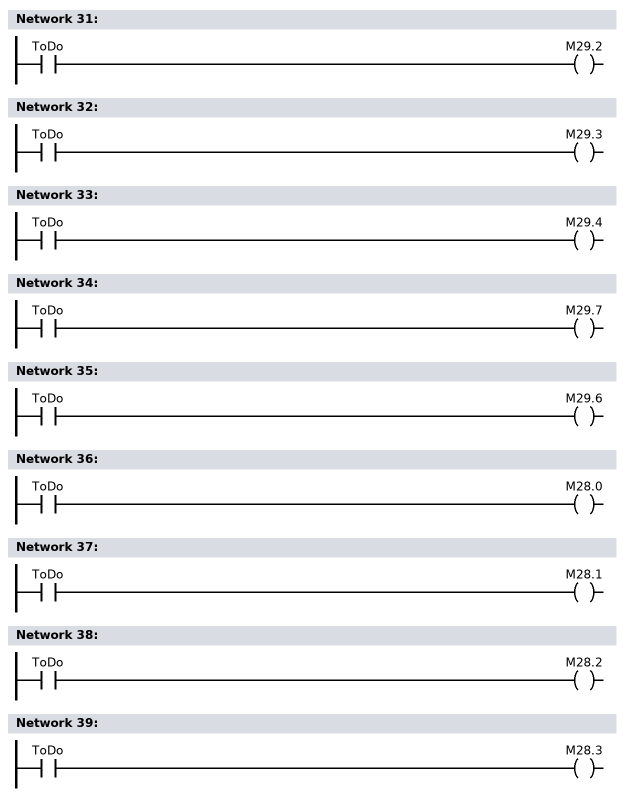
NETWORK
TITLE =
      A     "ToDo";
      =     "M29.2";
NETWORK
TITLE =
      A     "ToDo";
      =     "M29.3";
NETWORK
TITLE =
      A     "ToDo";
      =     "M29.4";
NETWORK
TITLE =
      A     "ToDo";
      =     "M29.7";
NETWORK
TITLE =
      A     "ToDo";
      =     "M29.6";
NETWORK
TITLE =
      A     "ToDo";
      =     "M28.0";
NETWORK
TITLE =
      A     "ToDo";
      =     "M28.1";
NETWORK
TITLE =
      A     "ToDo";
      =     "M28.2";
NETWORK
TITLE =
      A     "ToDo";
      =     "M28.3";
END_FUNCTION

FUNCTION "FC12 - GENERAL" : VOID	// FC 12
VERSION : 0.1
BEGIN
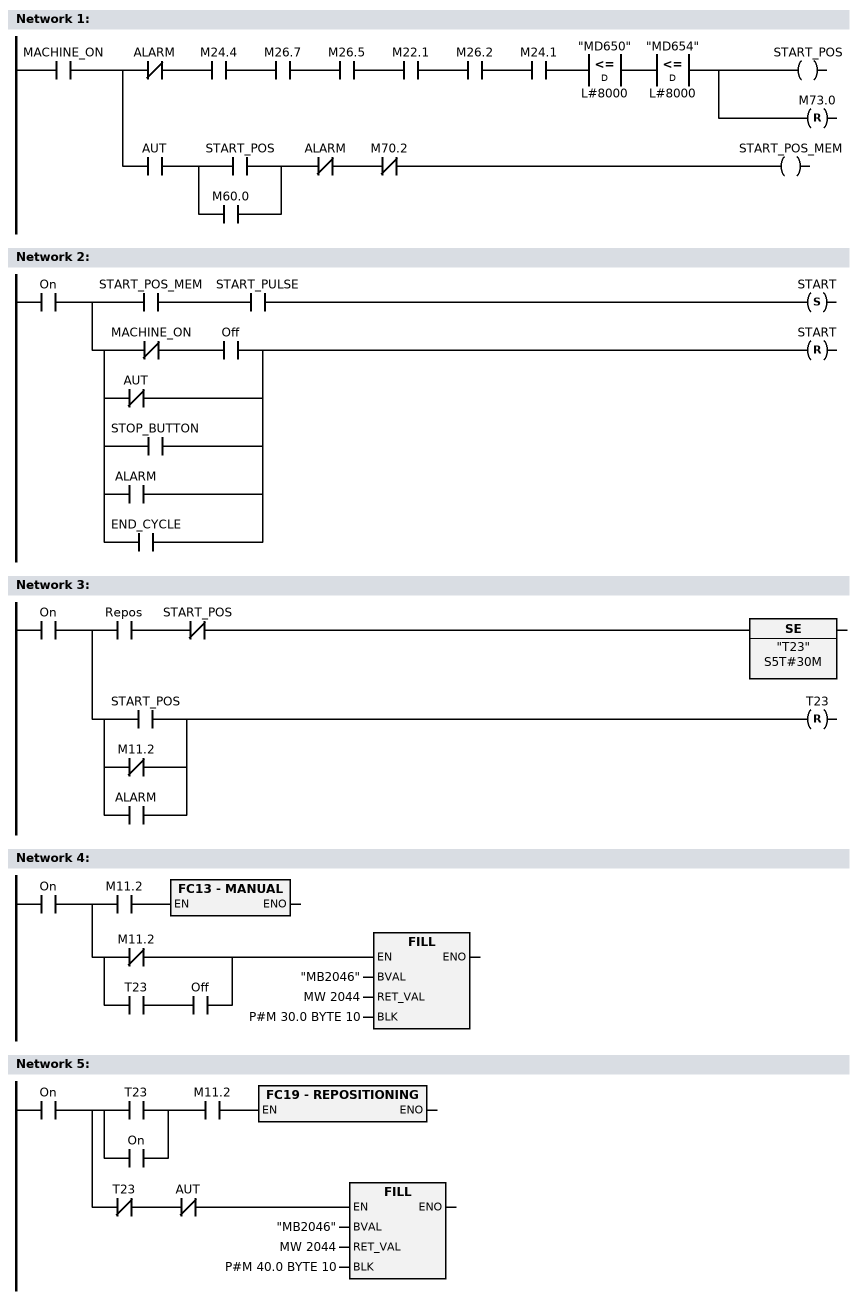
NETWORK
TITLE =
      A     "MACHINE_ON";
      =     L 0.0;
      A     L 0.0;
      AN    "ALARM";
      A     "M24.4";
      A     "M26.7";
      A     "M26.5";
      A     "M22.1";
      A     "M26.2";
      A     "M24.1";
      A(;
      L     "MD650";
      L     L#8000;
      <=D;
      );
      A(;
      L     "MD654";
      L     L#8000;
      <=D;
      );
      =     "START_POS";
      R     "M73.0";
      A     L 0.0;
      A     "AUT";
      A(;
      O     "START_POS";
      O     "M60.0";
      );
      AN    "ALARM";
      AN    "M70.2";
      =     "START_POS_MEM";
NETWORK
TITLE =
      A     "On";
      =     L 0.0;
      A     L 0.0;
      A     "START_POS_MEM";
      A     "START_PULSE";
      S     "START";
      A     L 0.0;
      A(;
      AN    "MACHINE_ON";
      A     "Off";
      ON    "AUT";
      O     "STOP_BUTTON";
      O     "ALARM";
      O     "END_CYCLE";
      );
      R     "START";
NETWORK
TITLE =
      A     "On";
      =     L 0.0;
      A     L 0.0;
      A     "Repos";
      AN    "START_POS";
      L     S5T#30M;
      SE    "T23";
      A     L 0.0;
      A(;
      O     "START_POS";
      ON    "M11.2";
      O     "ALARM";
      );
      R     "T23";
NETWORK
TITLE =
      A     "On";
      =     L 0.0;
      A     L 0.0;
      A     "M11.2";
      JNB   _001;
      CALL  "FC13 - MANUAL";
_001: NOP   0;
      A     L 0.0;
      A(;
      ON    "M11.2";
      O;
      A     "T23";
      A     "Off";
      );
      JNB   _002;
      CALL  "FILL" (
           BVAL                     := "MB2046",
           RET_VAL                  := MW 2044,
           BLK                      := P#M 30.0 BYTE 10);
_002: NOP   0;
NETWORK
TITLE =
      A     "On";
      =     L 0.0;
      A     L 0.0;
      A(;
      O     "T23";
      O     "On";
      );
      A     "M11.2";
      JNB   _003;
      CALL  "FC19 - REPOSITIONING";
_003: NOP   0;
      A     L 0.0;
      AN    "T23";
      AN    "AUT";
      JNB   _004;
      CALL  "FILL" (
           BVAL                     := "MB2046",
           RET_VAL                  := MW 2044,
           BLK                      := P#M 40.0 BYTE 10);
_004: NOP   0;
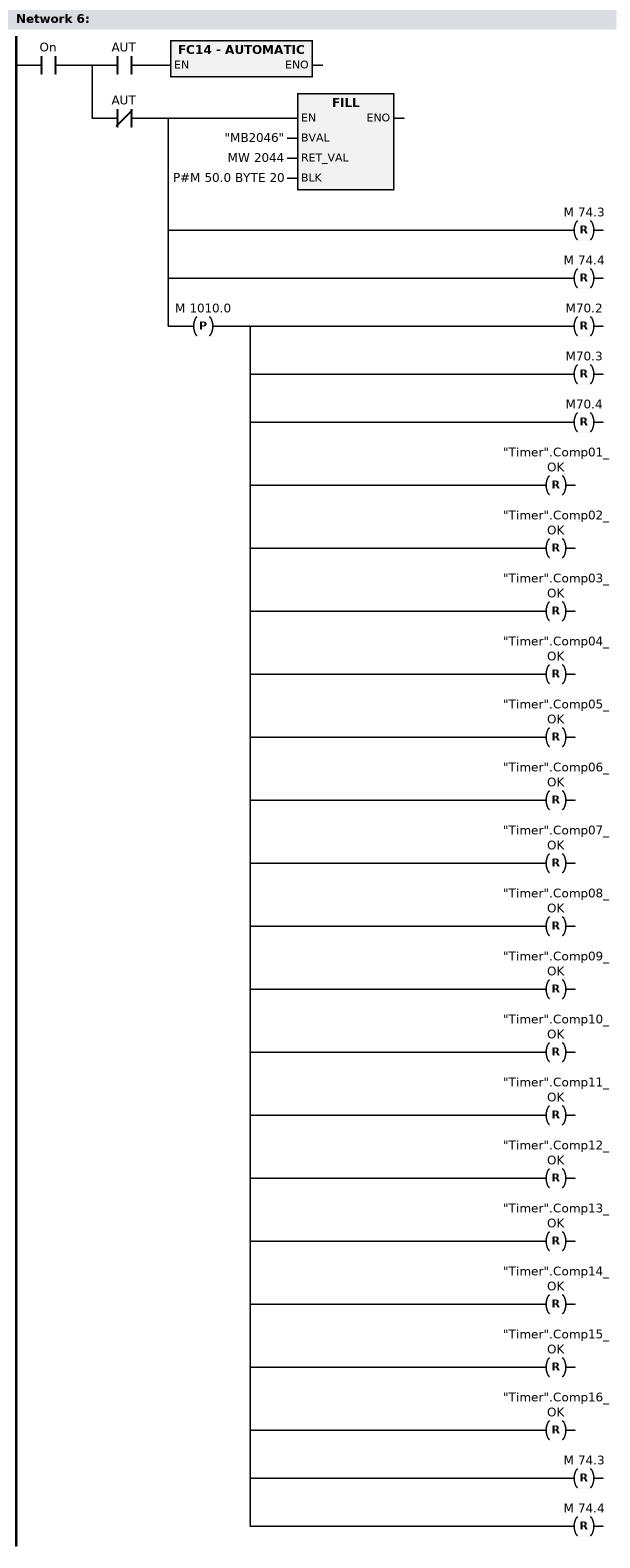
NETWORK
TITLE =
      A     "On";
      =     L 0.0;
      A     L 0.0;
      A     "AUT";
      JNB   _005;
      CALL  "FC14 - AUTOMATIC";
_005: NOP   0;
      A     L 0.0;
      AN    "AUT";
      =     L 0.1;
      A     L 0.1;
      JNB   _006;
      CALL  "FILL" (
           BVAL                     := "MB2046",
           RET_VAL                  := MW 2044,
           BLK                      := P#M 50.0 BYTE 20);
_006: NOP   0;
      A     L 0.1;
      BLD   102;
      R     M 74.3;
      A     L 0.1;
      BLD   102;
      R     M 74.4;
      A     L 0.1;
      FP    M 1010.0;
      R     "M70.2";
      R     "M70.3";
      R     "M70.4";
      R     "Timer".Comp01_OK;
      R     "Timer".Comp02_OK;
      R     "Timer".Comp03_OK;
      R     "Timer".Comp04_OK;
      R     "Timer".Comp05_OK;
      R     "Timer".Comp06_OK;
      R     "Timer".Comp07_OK;
      R     "Timer".Comp08_OK;
      R     "Timer".Comp09_OK;
      R     "Timer".Comp10_OK;
      R     "Timer".Comp11_OK;
      R     "Timer".Comp12_OK;
      R     "Timer".Comp13_OK;
      R     "Timer".Comp14_OK;
      R     "Timer".Comp15_OK;
      R     "Timer".Comp16_OK;
      R     M 74.3;
      R     M 74.4;
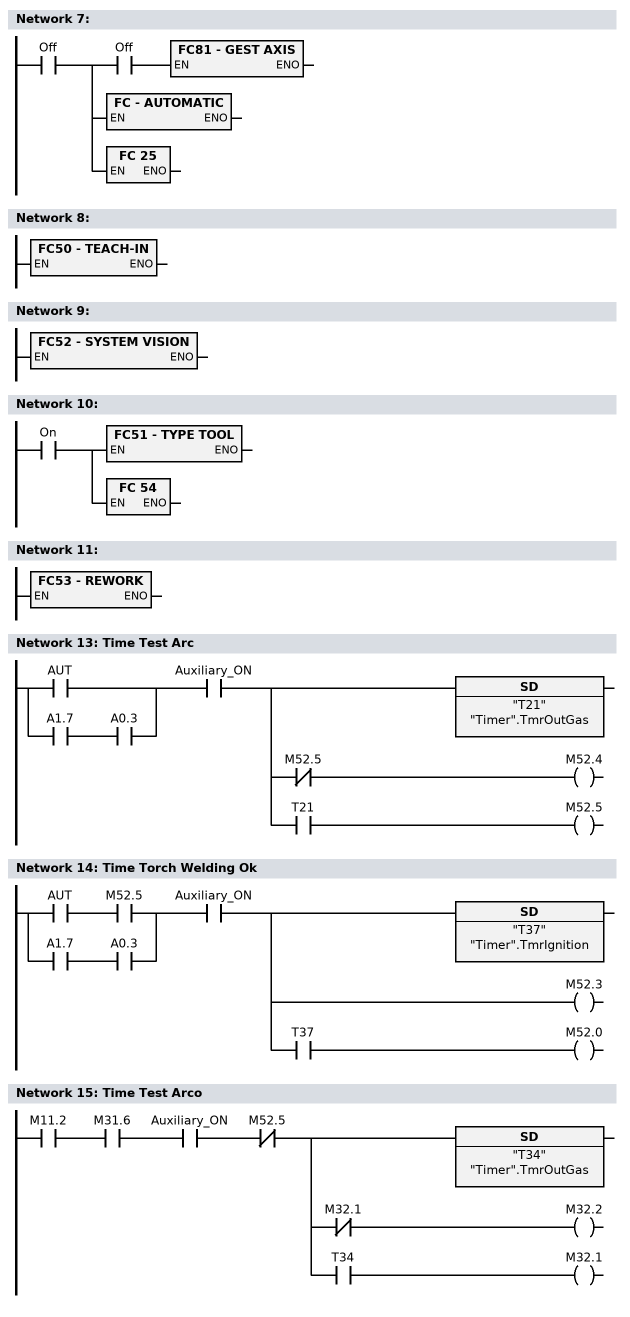
NETWORK
TITLE =
      A     "Off";
      =     L 0.0;
      A     L 0.0;
      A     "Off";
      JNB   _007;
      CALL  "FC81 - GEST AXIS";
_007: NOP   0;
      A     L 0.0;
      JNB   _008;
      CALL  "FC - AUTOMATIC";
_008: NOP   0;
      A     L 0.0;
      JNB   _009;
      CALL  FC 25;
_009: NOP   0;
NETWORK
TITLE =
      CALL  "FC50 - TEACH-IN";
      NOP   0;
NETWORK
TITLE =
      CALL  "FC52 - SYSTEM VISION";
      NOP   0;
NETWORK
TITLE =
      A     "On";
      =     L 0.0;
      A     L 0.0;
      JNB   _00a;
      CALL  "FC51 - TYPE TOOL";
_00a: NOP   0;
      A     L 0.0;
      JNB   _00b;
      CALL  FC 54;
_00b: NOP   0;
NETWORK
TITLE =
      CALL  "FC53 - REWORK";
      NOP   0;
NETWORK
TITLE =
NETWORK
TITLE = Time Test Arc
      A(;
      O     "AUT";
      O;
      A     "A1.7";
      A     "A0.3";
      );
      A     "Auxiliary_ON";
      =     L 0.0;
      A     L 0.0;
      BLD   102;
      L     "Timer".TmrOutGas;
      SD    "T21";
      A     L 0.0;
      AN    "M52.5";
      =     "M52.4";
      A     L 0.0;
      A     "T21";
      =     "M52.5";
NETWORK
TITLE = Time Torch Welding Ok
      A(;
      A     "AUT";
      A     "M52.5";
      O;
      A     "A1.7";
      A     "A0.3";
      );
      A     "Auxiliary_ON";
      =     L 0.0;
      A     L 0.0;
      BLD   102;
      L     "Timer".TmrIgnition;
      SD    "T37";
      A     L 0.0;
      BLD   102;
      =     "M52.3";
      A     L 0.0;
      A     "T37";
      =     "M52.0";
NETWORK
TITLE = Time Test Arco
      A     "M11.2";
      A     "M31.6";
      A     "Auxiliary_ON";
      AN    "M52.5";
      =     L 0.0;
      A     L 0.0;
      BLD   102;
      L     "Timer".TmrOutGas;
      SD    "T34";
      A     L 0.0;
      AN    "M32.1";
      =     "M32.2";
      A     L 0.0;
      A     "T34";
      =     "M32.1";
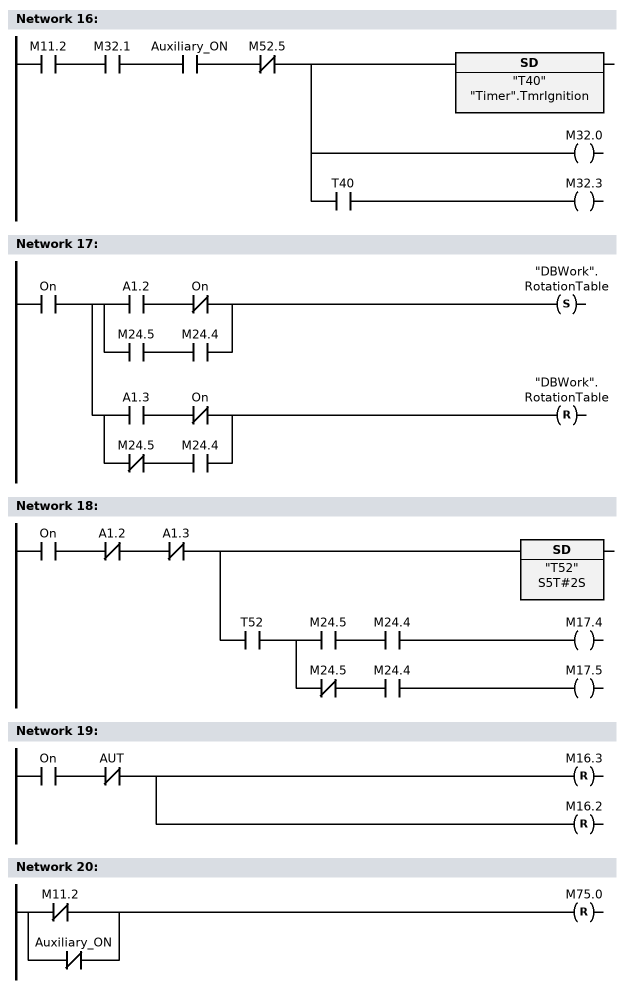
NETWORK
TITLE =
      A     "M11.2";
      A     "M32.1";
      A     "Auxiliary_ON";
      AN    "M52.5";
      =     L 0.0;
      A     L 0.0;
      BLD   102;
      L     "Timer".TmrIgnition;
      SD    "T40";
      A     L 0.0;
      BLD   102;
      =     "M32.0";
      A     L 0.0;
      A     "T40";
      =     "M32.3";
NETWORK
TITLE =
      A     "On";
      =     L 0.0;
      A     L 0.0;
      A(;
      A     "A1.2";
      AN    "On";
      O;
      A     "M24.5";
      A     "M24.4";
      );
      S     "DBWork".RotationTable;
      A     L 0.0;
      A(;
      A     "A1.3";
      AN    "On";
      O;
      AN    "M24.5";
      A     "M24.4";
      );
      R     "DBWork".RotationTable;
NETWORK
TITLE =
      A     "On";
      AN    "A1.2";
      AN    "A1.3";
      =     L 0.0;
      A     L 0.0;
      BLD   102;
      L     S5T#2S;
      SD    "T52";
      A     L 0.0;
      A     "T52";
      =     L 0.1;
      A     L 0.1;
      A     "M24.5";
      A     "M24.4";
      =     "M17.4";
      A     L 0.1;
      AN    "M24.5";
      A     "M24.4";
      =     "M17.5";
NETWORK
TITLE =
      A     "On";
      AN    "AUT";
      R     "M16.3";
      R     "M16.2";
NETWORK
TITLE =
      ON    "M11.2";
      ON    "Auxiliary_ON";
      R     "M75.0";
END_FUNCTION

FUNCTION "FC13 - MANUAL" : VOID	// FC 13
VERSION : 0.1
BEGIN
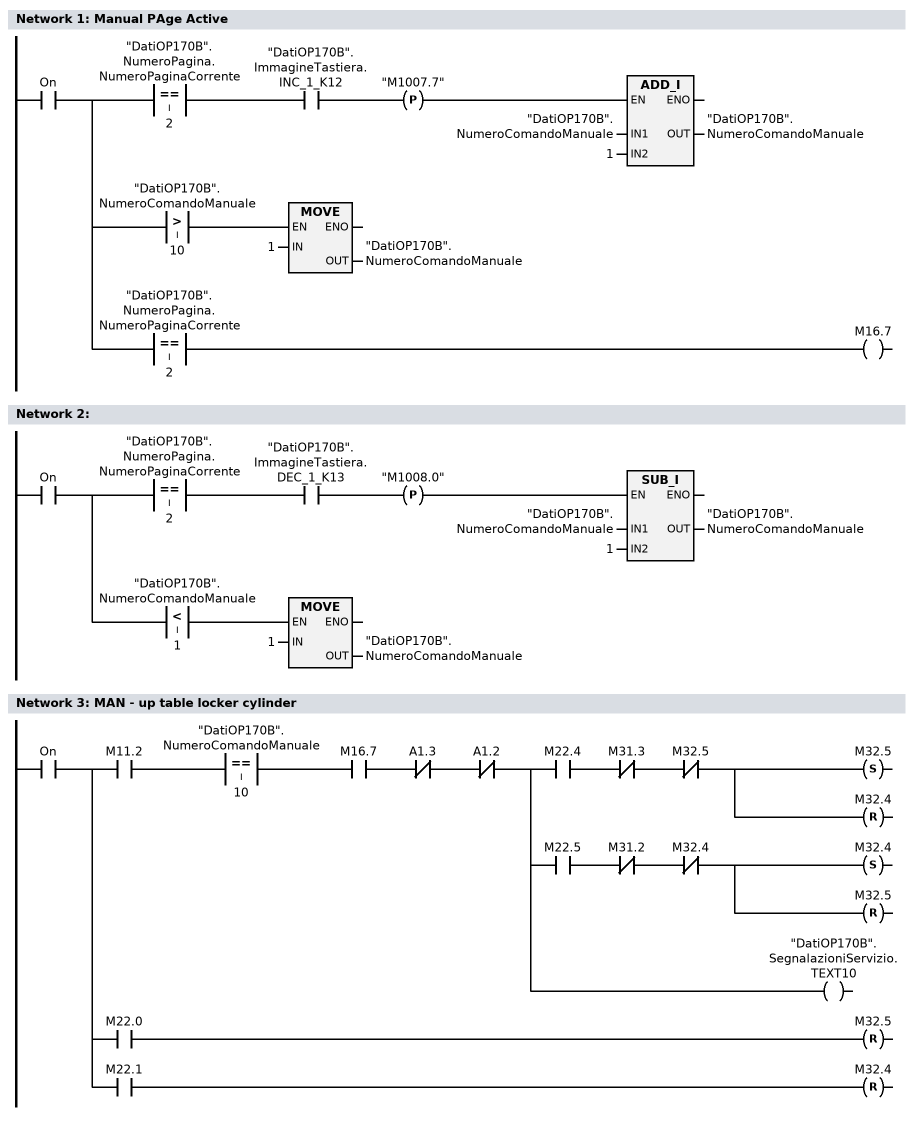
NETWORK
TITLE = Manual PAge Active
      A     "On";
      =     L 0.0;
      A     L 0.0;
      A(;
      L     "DatiOP170B".NumeroPagina.NumeroPaginaCorrente;
      L     2;
      ==I;
      );
      A     "DatiOP170B".ImmagineTastiera.INC_1_K12;
      FP    "M1007.7";
      JNB   _001;
      L     "DatiOP170B".NumeroComandoManuale;
      L     1;
      +I;
      T     "DatiOP170B".NumeroComandoManuale;
_001: NOP   0;
      A     L 0.0;
      A(;
      L     "DatiOP170B".NumeroComandoManuale;
      L     10;
      >I;
      );
      JNB   _002;
      L     1;
      T     "DatiOP170B".NumeroComandoManuale;
_002: NOP   0;
      A     L 0.0;
      A(;
      L     "DatiOP170B".NumeroPagina.NumeroPaginaCorrente;
      L     2;
      ==I;
      );
      =     "M16.7";
NETWORK
TITLE =
      A     "On";
      =     L 0.0;
      A     L 0.0;
      A(;
      L     "DatiOP170B".NumeroPagina.NumeroPaginaCorrente;
      L     2;
      ==I;
      );
      A     "DatiOP170B".ImmagineTastiera.DEC_1_K13;
      FP    "M1008.0";
      JNB   _003;
      L     "DatiOP170B".NumeroComandoManuale;
      L     1;
      -I;
      T     "DatiOP170B".NumeroComandoManuale;
_003: NOP   0;
      A     L 0.0;
      A(;
      L     "DatiOP170B".NumeroComandoManuale;
      L     1;
      <I;
      );
      JNB   _004;
      L     1;
      T     "DatiOP170B".NumeroComandoManuale;
_004: NOP   0;
NETWORK
TITLE = MAN - up table locker cylinder
      A     "On";
      =     L 0.0;
      A     L 0.0;
      A     "M11.2";
      A(;
      L     "DatiOP170B".NumeroComandoManuale;
      L     10;
      ==I;
      );
      A     "M16.7";
      AN    "A1.3";
      AN    "A1.2";
      =     L 0.1;
      A     L 0.1;
      A     "M22.4";
      AN    "M31.3";
      AN    "M32.5";
      S     "M32.5";
      R     "M32.4";
      A     L 0.1;
      A     "M22.5";
      AN    "M31.2";
      AN    "M32.4";
      S     "M32.4";
      R     "M32.5";
      A     L 0.1;
      BLD   102;
      =     "DatiOP170B".SegnalazioniServizio.TEXT10;
      A     L 0.0;
      A     "M22.0";
      R     "M32.5";
      A     L 0.0;
      A     "M22.1";
      R     "M32.4";
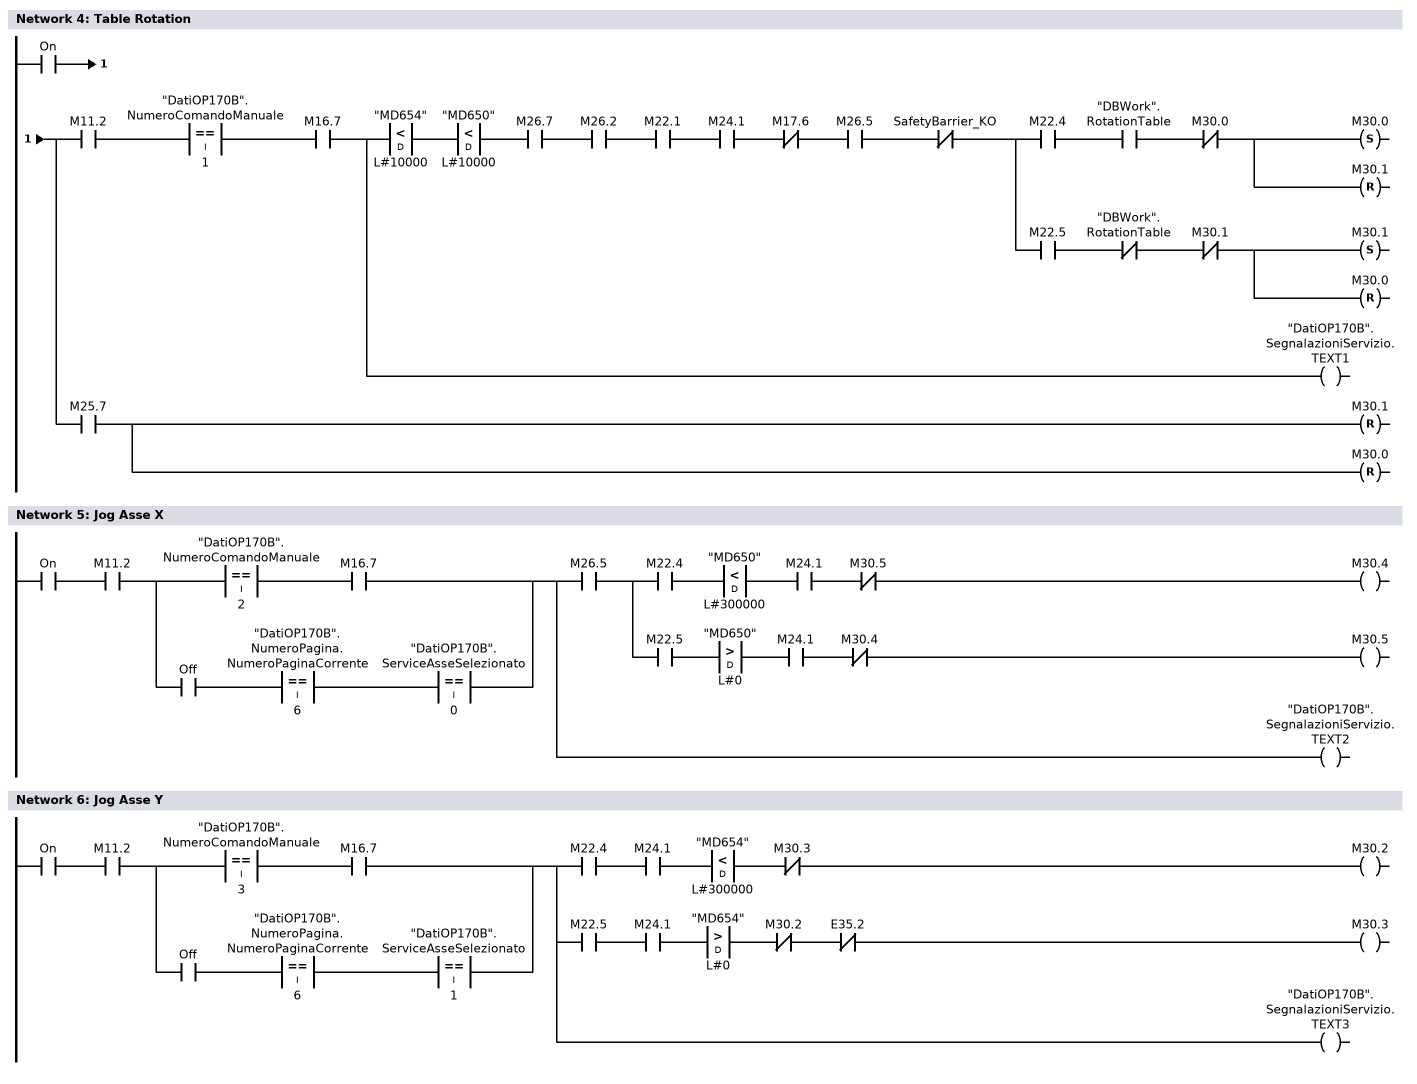
NETWORK
TITLE = Table Rotation
      A     "On";
      =     L 0.0;
      A     L 0.0;
      A     "M11.2";
      A(;
      L     "DatiOP170B".NumeroComandoManuale;
      L     1;
      ==I;
      );
      A     "M16.7";
      =     L 0.1;
      A     L 0.1;
      A(;
      L     "MD654";
      L     L#10000;
      <D;
      );
      A(;
      L     "MD650";
      L     L#10000;
      <D;
      );
      A     "M26.7";
      A     "M26.2";
      A     "M22.1";
      A     "M24.1";
      AN    "M17.6";
      A     "M26.5";
      AN    "SafetyBarrier_KO";
      =     L 0.2;
      A     L 0.2;
      A     "M22.4";
      A     "DBWork".RotationTable;
      AN    "M30.0";
      S     "M30.0";
      R     "M30.1";
      A     L 0.2;
      A     "M22.5";
      AN    "DBWork".RotationTable;
      AN    "M30.1";
      S     "M30.1";
      R     "M30.0";
      A     L 0.1;
      BLD   102;
      =     "DatiOP170B".SegnalazioniServizio.TEXT1;
      A     L 0.0;
      A     "M25.7";
      R     "M30.1";
      R     "M30.0";
NETWORK
TITLE = Jog Asse X
      A     "On";
      A     "M11.2";
      A(;
      A(;
      L     "DatiOP170B".NumeroComandoManuale;
      L     2;
      ==I;
      );
      A     "M16.7";
      O;
      A     "Off";
      A(;
      L     "DatiOP170B".NumeroPagina.NumeroPaginaCorrente;
      L     6;
      ==I;
      );
      A(;
      L     "DatiOP170B".ServiceAsseSelezionato;
      L     0;
      ==I;
      );
      );
      =     L 0.0;
      A     L 0.0;
      A     "M26.5";
      =     L 0.1;
      A     L 0.1;
      A     "M22.4";
      A(;
      L     "MD650";
      L     L#300000;
      <D;
      );
      A     "M24.1";
      AN    "M30.5";
      =     "M30.4";
      A     L 0.1;
      A     "M22.5";
      A(;
      L     "MD650";
      L     L#0;
      >D;
      );
      A     "M24.1";
      AN    "M30.4";
      =     "M30.5";
      A     L 0.0;
      BLD   102;
      =     "DatiOP170B".SegnalazioniServizio.TEXT2;
NETWORK
TITLE = Jog Asse Y
      A     "On";
      A     "M11.2";
      A(;
      A(;
      L     "DatiOP170B".NumeroComandoManuale;
      L     3;
      ==I;
      );
      A     "M16.7";
      O;
      A     "Off";
      A(;
      L     "DatiOP170B".NumeroPagina.NumeroPaginaCorrente;
      L     6;
      ==I;
      );
      A(;
      L     "DatiOP170B".ServiceAsseSelezionato;
      L     1;
      ==I;
      );
      );
      =     L 0.0;
      A     L 0.0;
      A     "M22.4";
      A     "M24.1";
      A(;
      L     "MD654";
      L     L#300000;
      <D;
      );
      AN    "M30.3";
      =     "M30.2";
      A     L 0.0;
      A     "M22.5";
      A     "M24.1";
      A(;
      L     "MD654";
      L     L#0;
      >D;
      );
      AN    "M30.2";
      AN    "E35.2";
      =     "M30.3";
      A     L 0.0;
      BLD   102;
      =     "DatiOP170B".SegnalazioniServizio.TEXT3;
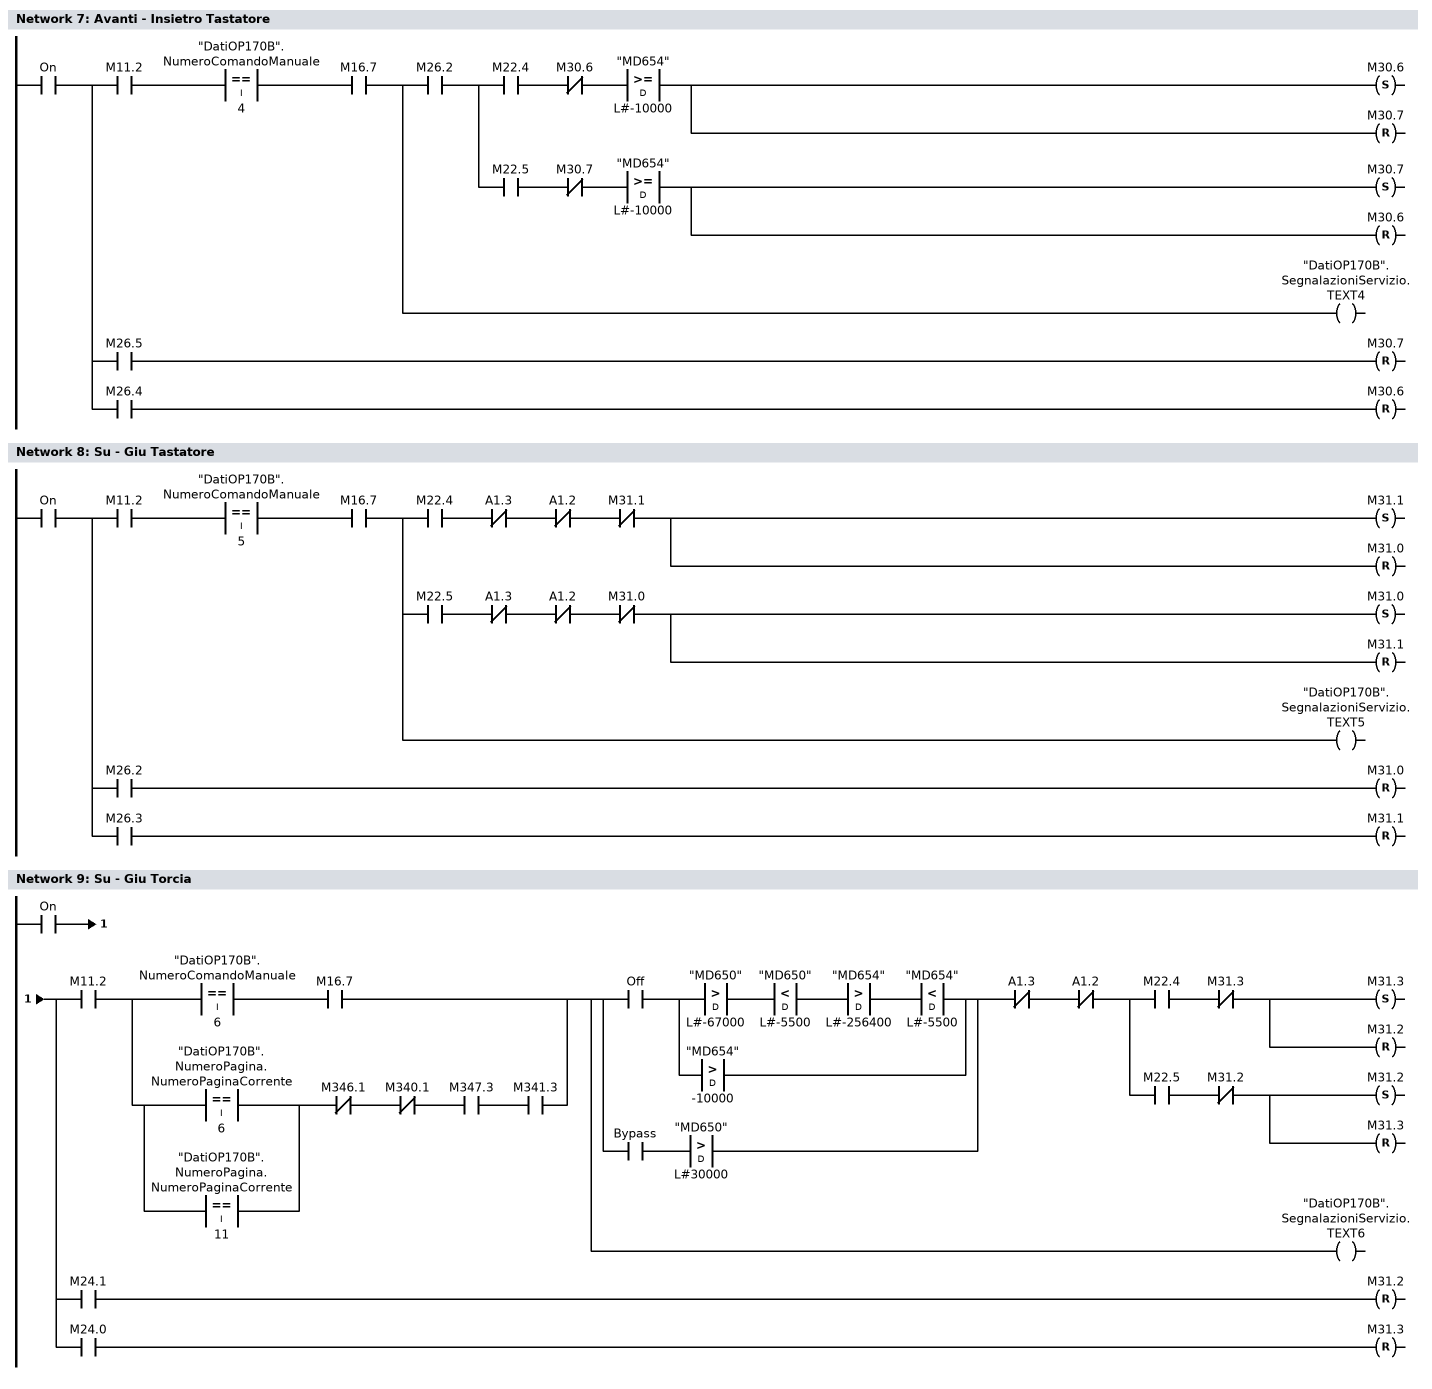
NETWORK
TITLE = Avanti - Insietro Tastatore
      A     "On";
      =     L 0.0;
      A     L 0.0;
      A     "M11.2";
      A(;
      L     "DatiOP170B".NumeroComandoManuale;
      L     4;
      ==I;
      );
      A     "M16.7";
      =     L 0.1;
      A     L 0.1;
      A     "M26.2";
      =     L 0.2;
      A     L 0.2;
      A     "M22.4";
      AN    "M30.6";
      A(;
      L     "MD654";
      L     L#-10000;
      >=D;
      );
      S     "M30.6";
      R     "M30.7";
      A     L 0.2;
      A     "M22.5";
      AN    "M30.7";
      A(;
      L     "MD654";
      L     L#-10000;
      >=D;
      );
      S     "M30.7";
      R     "M30.6";
      A     L 0.1;
      BLD   102;
      =     "DatiOP170B".SegnalazioniServizio.TEXT4;
      A     L 0.0;
      A     "M26.5";
      R     "M30.7";
      A     L 0.0;
      A     "M26.4";
      R     "M30.6";
NETWORK
TITLE = Su - Giu Tastatore
      A     "On";
      =     L 0.0;
      A     L 0.0;
      A     "M11.2";
      A(;
      L     "DatiOP170B".NumeroComandoManuale;
      L     5;
      ==I;
      );
      A     "M16.7";
      =     L 0.1;
      A     L 0.1;
      A     "M22.4";
      AN    "A1.3";
      AN    "A1.2";
      AN    "M31.1";
      S     "M31.1";
      R     "M31.0";
      A     L 0.1;
      A     "M22.5";
      AN    "A1.3";
      AN    "A1.2";
      AN    "M31.0";
      S     "M31.0";
      R     "M31.1";
      A     L 0.1;
      BLD   102;
      =     "DatiOP170B".SegnalazioniServizio.TEXT5;
      A     L 0.0;
      A     "M26.2";
      R     "M31.0";
      A     L 0.0;
      A     "M26.3";
      R     "M31.1";
NETWORK
TITLE = Su - Giu Torcia
      A     "On";
      =     L 0.0;
      A     L 0.0;
      A     "M11.2";
      A(;
      A(;
      L     "DatiOP170B".NumeroComandoManuale;
      L     6;
      ==I;
      );
      A     "M16.7";
      O;
      A(;
      O(;
      L     "DatiOP170B".NumeroPagina.NumeroPaginaCorrente;
      L     6;
      ==I;
      );
      O(;
      L     "DatiOP170B".NumeroPagina.NumeroPaginaCorrente;
      L     11;
      ==I;
      );
      );
      AN    "M346.1";
      AN    "M340.1";
      A     "M347.3";
      A     "M341.3";
      );
      =     L 0.1;
      A     L 0.1;
      A(;
      A     "Off";
      A(;
      A(;
      L     "MD650";
      L     L#-67000;
      >D;
      );
      A(;
      L     "MD650";
      L     L#-5500;
      <D;
      );
      A(;
      L     "MD654";
      L     L#-256400;
      >D;
      );
      A(;
      L     "MD654";
      L     L#-5500;
      <D;
      );
      O(;
      L     "MD654";
      L     -10000;
      >D;
      );
      );
      O;
      A     "Bypass";
      A(;
      L     "MD650";
      L     L#30000;
      >D;
      );
      );
      AN    "A1.3";
      AN    "A1.2";
      =     L 0.2;
      A     L 0.2;
      A     "M22.4";
      AN    "M31.3";
      S     "M31.3";
      R     "M31.2";
      A     L 0.2;
      A     "M22.5";
      AN    "M31.2";
      S     "M31.2";
      R     "M31.3";
      A     L 0.1;
      BLD   102;
      =     "DatiOP170B".SegnalazioniServizio.TEXT6;
      A     L 0.0;
      A     "M24.1";
      R     "M31.2";
      A     L 0.0;
      A     "M24.0";
      R     "M31.3";
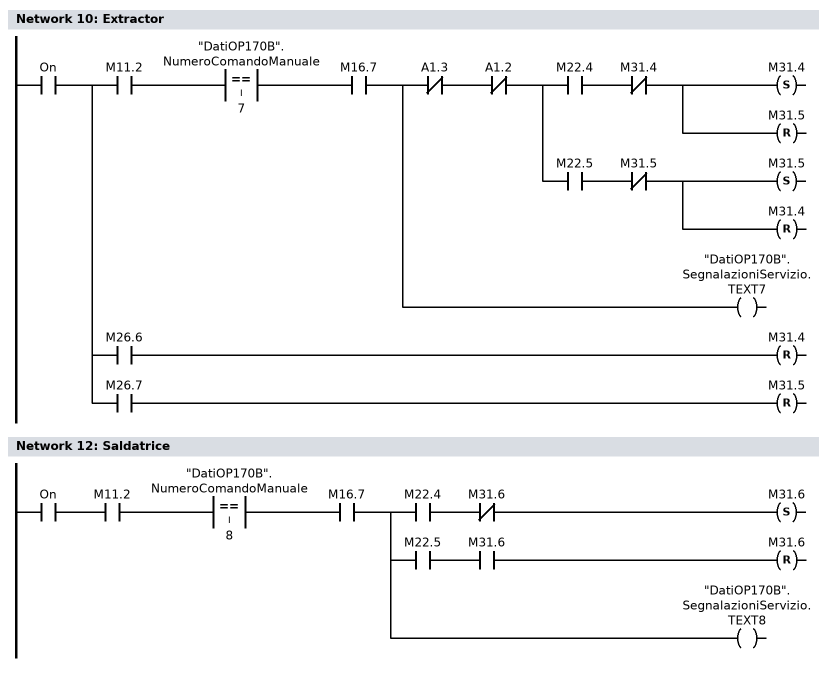
NETWORK
TITLE = Extractor
      A     "On";
      =     L 0.0;
      A     L 0.0;
      A     "M11.2";
      A(;
      L     "DatiOP170B".NumeroComandoManuale;
      L     7;
      ==I;
      );
      A     "M16.7";
      =     L 0.1;
      A     L 0.1;
      AN    "A1.3";
      AN    "A1.2";
      =     L 0.2;
      A     L 0.2;
      A     "M22.4";
      AN    "M31.4";
      S     "M31.4";
      R     "M31.5";
      A     L 0.2;
      A     "M22.5";
      AN    "M31.5";
      S     "M31.5";
      R     "M31.4";
      A     L 0.1;
      BLD   102;
      =     "DatiOP170B".SegnalazioniServizio.TEXT7;
      A     L 0.0;
      A     "M26.6";
      R     "M31.4";
      A     L 0.0;
      A     "M26.7";
      R     "M31.5";
NETWORK
TITLE =
NETWORK
TITLE = Saldatrice
      A     "On";
      A     "M11.2";
      A(;
      L     "DatiOP170B".NumeroComandoManuale;
      L     8;
      ==I;
      );
      A     "M16.7";
      =     L 0.0;
      A     L 0.0;
      A     "M22.4";
      AN    "M31.6";
      S     "M31.6";
      A     L 0.0;
      A     "M22.5";
      A     "M31.6";
      R     "M31.6";
      A     L 0.0;
      BLD   102;
      =     "DatiOP170B".SegnalazioniServizio.TEXT8;
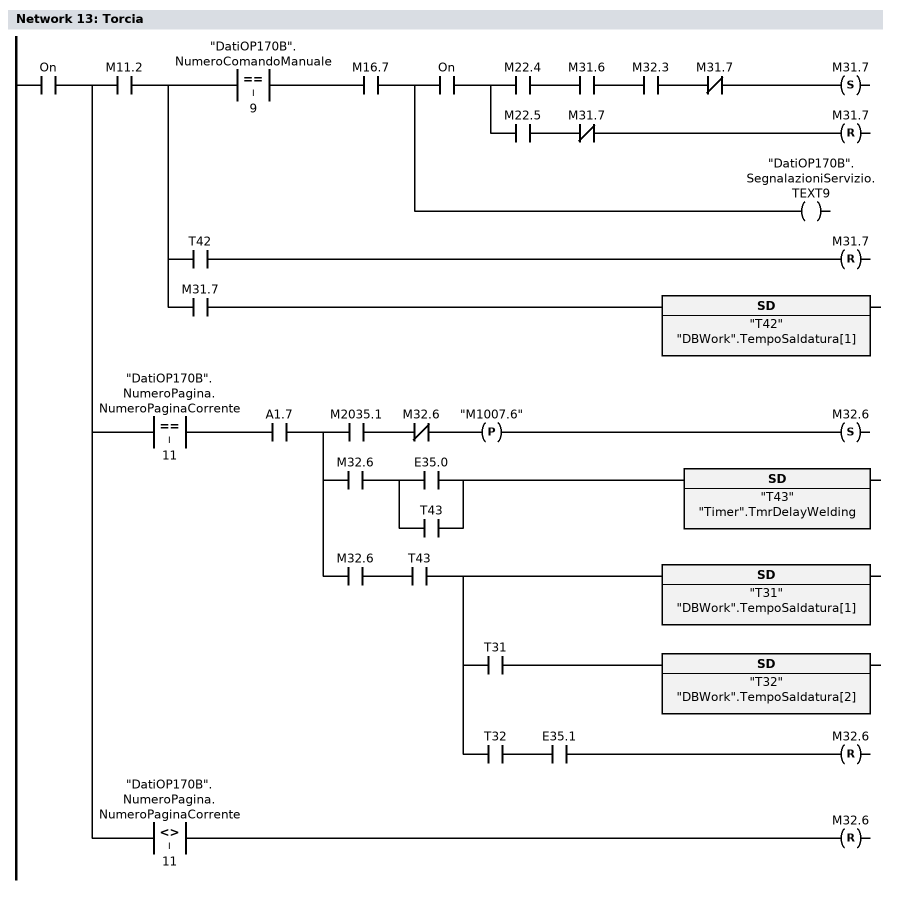
NETWORK
TITLE = Torcia
      A     "On";
      =     L 0.0;
      A     L 0.0;
      A     "M11.2";
      =     L 0.1;
      A     L 0.1;
      A(;
      L     "DatiOP170B".NumeroComandoManuale;
      L     9;
      ==I;
      );
      A     "M16.7";
      =     L 0.2;
      A     L 0.2;
      A     "On";
      =     L 0.3;
      A     L 0.3;
      A     "M22.4";
      A     "M31.6";
      A     "M32.3";
      AN    "M31.7";
      S     "M31.7";
      A     L 0.3;
      A     "M22.5";
      AN    "M31.7";
      R     "M31.7";
      A     L 0.2;
      BLD   102;
      =     "DatiOP170B".SegnalazioniServizio.TEXT9;
      A     L 0.1;
      A     "T42";
      R     "M31.7";
      A     L 0.1;
      A     "M31.7";
      L     "DBWork".TempoSaldatura[1];
      SD    "T42";
      A     L 0.0;
      A(;
      L     "DatiOP170B".NumeroPagina.NumeroPaginaCorrente;
      L     11;
      ==I;
      );
      A     "A1.7";
      =     L 0.1;
      A     L 0.1;
      A     "M2035.1";
      AN    "M32.6";
      FP    "M1007.6";
      S     "M32.6";
      A     L 0.1;
      A     "M32.6";
      A(;
      O     "E35.0";
      O     "T43";
      );
      L     "Timer".TmrDelayWelding;
      SD    "T43";
      A     L 0.1;
      A     "M32.6";
      A     "T43";
      =     L 0.2;
      A     L 0.2;
      BLD   102;
      L     "DBWork".TempoSaldatura[1];
      SD    "T31";
      A     L 0.2;
      A     "T31";
      L     "DBWork".TempoSaldatura[2];
      SD    "T32";
      A     L 0.2;
      A     "T32";
      A     "E35.1";
      R     "M32.6";
      A     L 0.0;
      A(;
      L     "DatiOP170B".NumeroPagina.NumeroPaginaCorrente;
      L     11;
      <>I;
      );
      R     "M32.6";
END_FUNCTION

FUNCTION "FC14 - AUTOMATIC" : VOID	// FC 14
VERSION : 0.1
VAR_TEMP
  TEMP0 : DINT ;
  TEMP1 : DINT ;
  TEMP2 : DINT ;
  TEMP3 : DINT ;
  TEMP4 : DINT ;
  TEMP5 : DINT ;
END_VAR
BEGIN
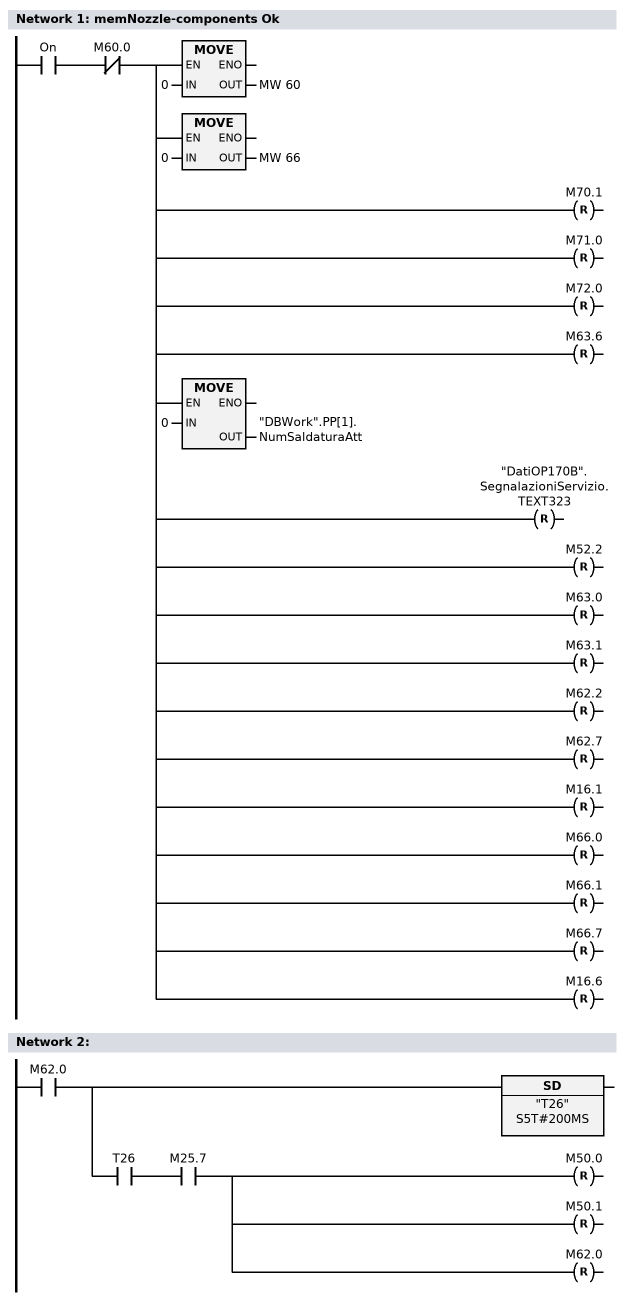
NETWORK
TITLE = memNozzle-components Ok
      A     "On";
      AN    "M60.0";
      =     L 24.0;
      A     L 24.0;
      JNB   _001;
      L     0;
      T     MW 60;
_001: NOP   0;
      A     L 24.0;
      JNB   _002;
      L     0;
      T     MW 66;
_002: NOP   0;
      A     L 24.0;
      BLD   102;
      R     "M70.1";
      A     L 24.0;
      BLD   102;
      R     "M71.0";
      A     L 24.0;
      BLD   102;
      R     "M72.0";
      A     L 24.0;
      BLD   102;
      R     "M63.6";
      A     L 24.0;
      JNB   _003;
      L     0;
      T     "DBWork".PP[1].NumSaldaturaAtt;
_003: NOP   0;
      A     L 24.0;
      BLD   102;
      R     "DatiOP170B".SegnalazioniServizio.TEXT323;
      A     L 24.0;
      BLD   102;
      R     "M52.2";
      A     L 24.0;
      BLD   102;
      R     "M63.0";
      A     L 24.0;
      BLD   102;
      R     "M63.1";
      A     L 24.0;
      BLD   102;
      R     "M62.2";
      A     L 24.0;
      BLD   102;
      R     "M62.7";
      A     L 24.0;
      BLD   102;
      R     "M16.1";
      A     L 24.0;
      BLD   102;
      R     "M66.0";
      A     L 24.0;
      BLD   102;
      R     "M66.1";
      A     L 24.0;
      BLD   102;
      R     "M66.7";
      A     L 24.0;
      BLD   102;
      R     "M16.6";
NETWORK
TITLE =
      A     "M62.0";
      =     L 24.0;
      A     L 24.0;
      BLD   102;
      L     S5T#200MS;
      SD    "T26";
      A     L 24.0;
      A     "T26";
      A     "M25.7";
      R     "M50.0";
      R     "M50.1";
      R     "M62.0";
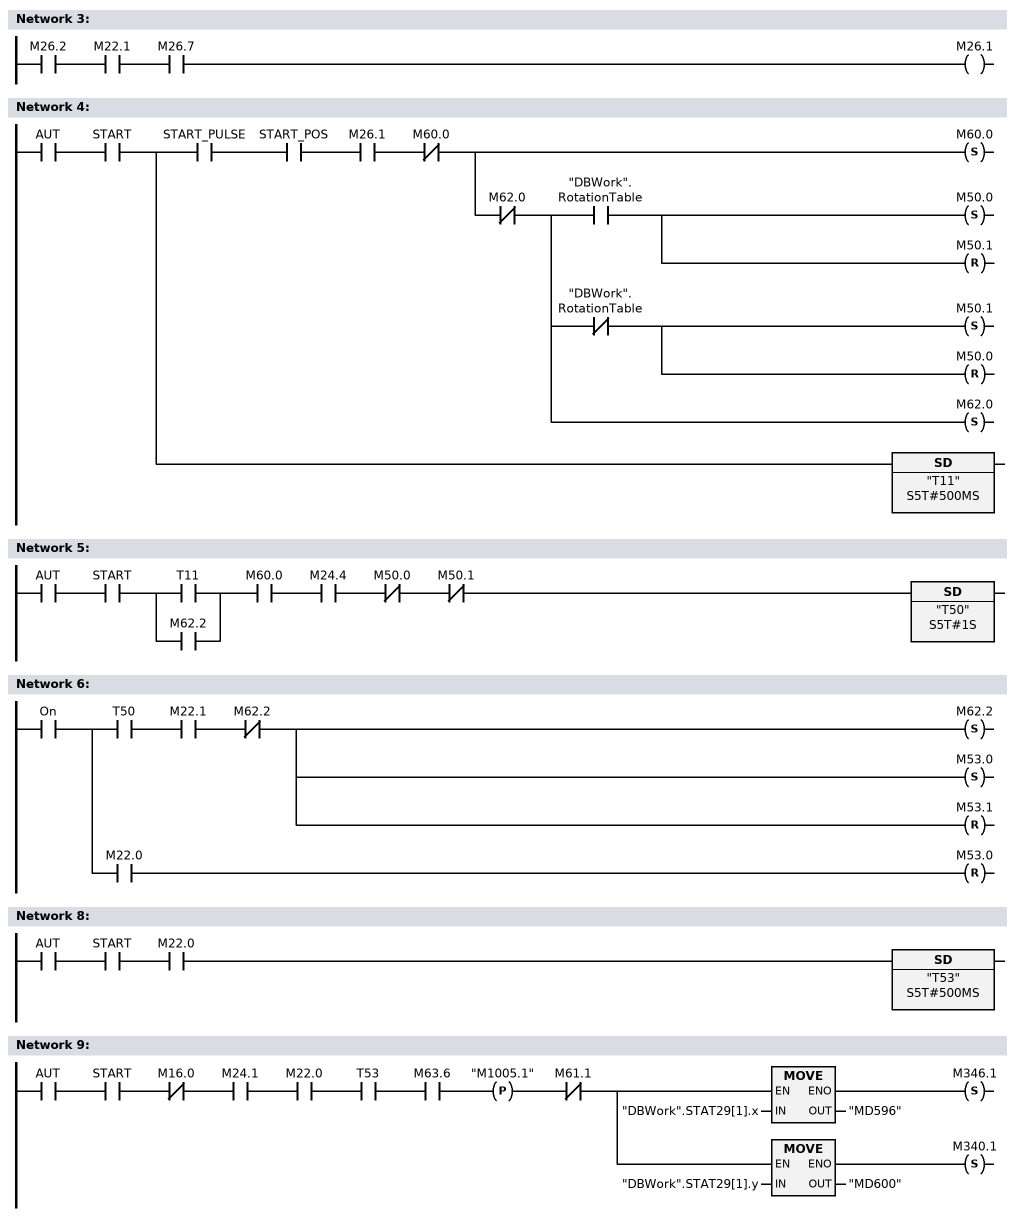
NETWORK
TITLE =
      A     "M26.2";
      A     "M22.1";
      A     "M26.7";
      =     "M26.1";
NETWORK
TITLE =
      A     "AUT";
      A     "START";
      =     L 24.0;
      A     L 24.0;
      A     "START_PULSE";
      A     "START_POS";
      A     "M26.1";
      AN    "M60.0";
      =     L 24.1;
      A     L 24.1;
      BLD   102;
      S     "M60.0";
      A     L 24.1;
      AN    "M62.0";
      =     L 24.2;
      A     L 24.2;
      A     "DBWork".RotationTable;
      S     "M50.0";
      R     "M50.1";
      A     L 24.2;
      AN    "DBWork".RotationTable;
      S     "M50.1";
      R     "M50.0";
      A     L 24.2;
      BLD   102;
      S     "M62.0";
      A     L 24.0;
      BLD   102;
      L     S5T#500MS;
      SD    "T11";
NETWORK
TITLE =
      A     "AUT";
      A     "START";
      A(;
      O     "T11";
      O     "M62.2";
      );
      A     "M60.0";
      A     "M24.4";
      AN    "M50.0";
      AN    "M50.1";
      L     S5T#1S;
      SD    "T50";
NETWORK
TITLE =
      A     "On";
      =     L 24.0;
      A     L 24.0;
      A     "T50";
      A     "M22.1";
      AN    "M62.2";
      S     "M62.2";
      S     "M53.0";
      R     "M53.1";
      A     L 24.0;
      A     "M22.0";
      R     "M53.0";
NETWORK
TITLE =
NETWORK
TITLE =
      A     "AUT";
      A     "START";
      A     "M22.0";
      L     S5T#500MS;
      SD    "T53";
NETWORK
TITLE =
      A     "AUT";
      A     "START";
      AN    "M16.0";
      A     "M24.1";
      A     "M22.0";
      A     "T53";
      A     "M63.6";
      FP    "M1005.1";
      AN    "M61.1";
      =     L 24.0;
      A     L 24.0;
      JNB   _004;
      L     "DBWork".STAT29[1].x;
      T     "MD596";
      SET;
      SAVE;
      CLR;
_004: A     BR;
      S     "M346.1";
      A     L 24.0;
      JNB   _005;
      L     "DBWork".STAT29[1].y;
      T     "MD600";
      SET;
      SAVE;
      CLR;
_005: A     BR;
      S     "M340.1";
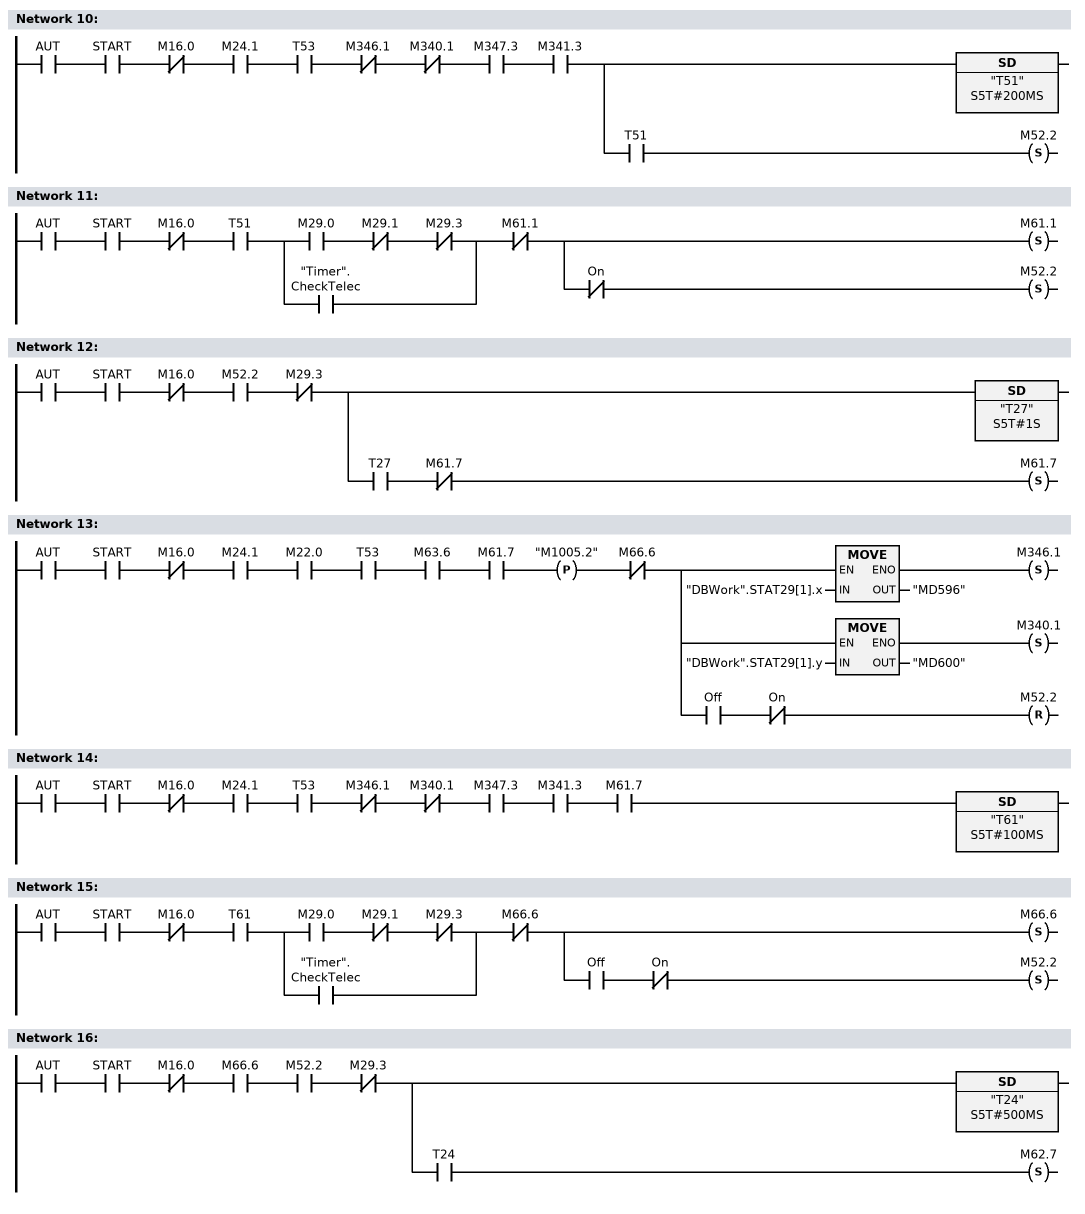
NETWORK
TITLE =
      A     "AUT";
      A     "START";
      AN    "M16.0";
      A     "M24.1";
      A     "T53";
      AN    "M346.1";
      AN    "M340.1";
      A     "M347.3";
      A     "M341.3";
      =     L 24.0;
      A     L 24.0;
      BLD   102;
      L     S5T#200MS;
      SD    "T51";
      A     L 24.0;
      A     "T51";
      S     "M52.2";
NETWORK
TITLE =
      A     "AUT";
      A     "START";
      AN    "M16.0";
      A     "T51";
      A(;
      A     "M29.0";
      AN    "M29.1";
      AN    "M29.3";
      O     "Timer".CheckTelec;
      );
      AN    "M61.1";
      =     L 24.0;
      A     L 24.0;
      BLD   102;
      S     "M61.1";
      A     L 24.0;
      AN    "On";
      S     "M52.2";
NETWORK
TITLE =
      A     "AUT";
      A     "START";
      AN    "M16.0";
      A     "M52.2";
      AN    "M29.3";
      =     L 24.0;
      A     L 24.0;
      BLD   102;
      L     S5T#1S;
      SD    "T27";
      A     L 24.0;
      A     "T27";
      AN    "M61.7";
      S     "M61.7";
NETWORK
TITLE =
      A     "AUT";
      A     "START";
      AN    "M16.0";
      A     "M24.1";
      A     "M22.0";
      A     "T53";
      A     "M63.6";
      A     "M61.7";
      FP    "M1005.2";
      AN    "M66.6";
      =     L 24.0;
      A     L 24.0;
      JNB   _006;
      L     "DBWork".STAT29[1].x;
      T     "MD596";
      SET;
      SAVE;
      CLR;
_006: A     BR;
      S     "M346.1";
      A     L 24.0;
      JNB   _007;
      L     "DBWork".STAT29[1].y;
      T     "MD600";
      SET;
      SAVE;
      CLR;
_007: A     BR;
      S     "M340.1";
      A     L 24.0;
      A     "Off";
      AN    "On";
      R     "M52.2";
NETWORK
TITLE =
      A     "AUT";
      A     "START";
      AN    "M16.0";
      A     "M24.1";
      A     "T53";
      AN    "M346.1";
      AN    "M340.1";
      A     "M347.3";
      A     "M341.3";
      A     "M61.7";
      L     S5T#100MS;
      SD    "T61";
NETWORK
TITLE =
      A     "AUT";
      A     "START";
      AN    "M16.0";
      A     "T61";
      A(;
      A     "M29.0";
      AN    "M29.1";
      AN    "M29.3";
      O     "Timer".CheckTelec;
      );
      AN    "M66.6";
      =     L 24.0;
      A     L 24.0;
      BLD   102;
      S     "M66.6";
      A     L 24.0;
      A     "Off";
      AN    "On";
      S     "M52.2";
NETWORK
TITLE =
      A     "AUT";
      A     "START";
      AN    "M16.0";
      A     "M66.6";
      A     "M52.2";
      AN    "M29.3";
      =     L 24.0;
      A     L 24.0;
      BLD   102;
      L     S5T#500MS;
      SD    "T24";
      A     L 24.0;
      A     "T24";
      S     "M62.7";
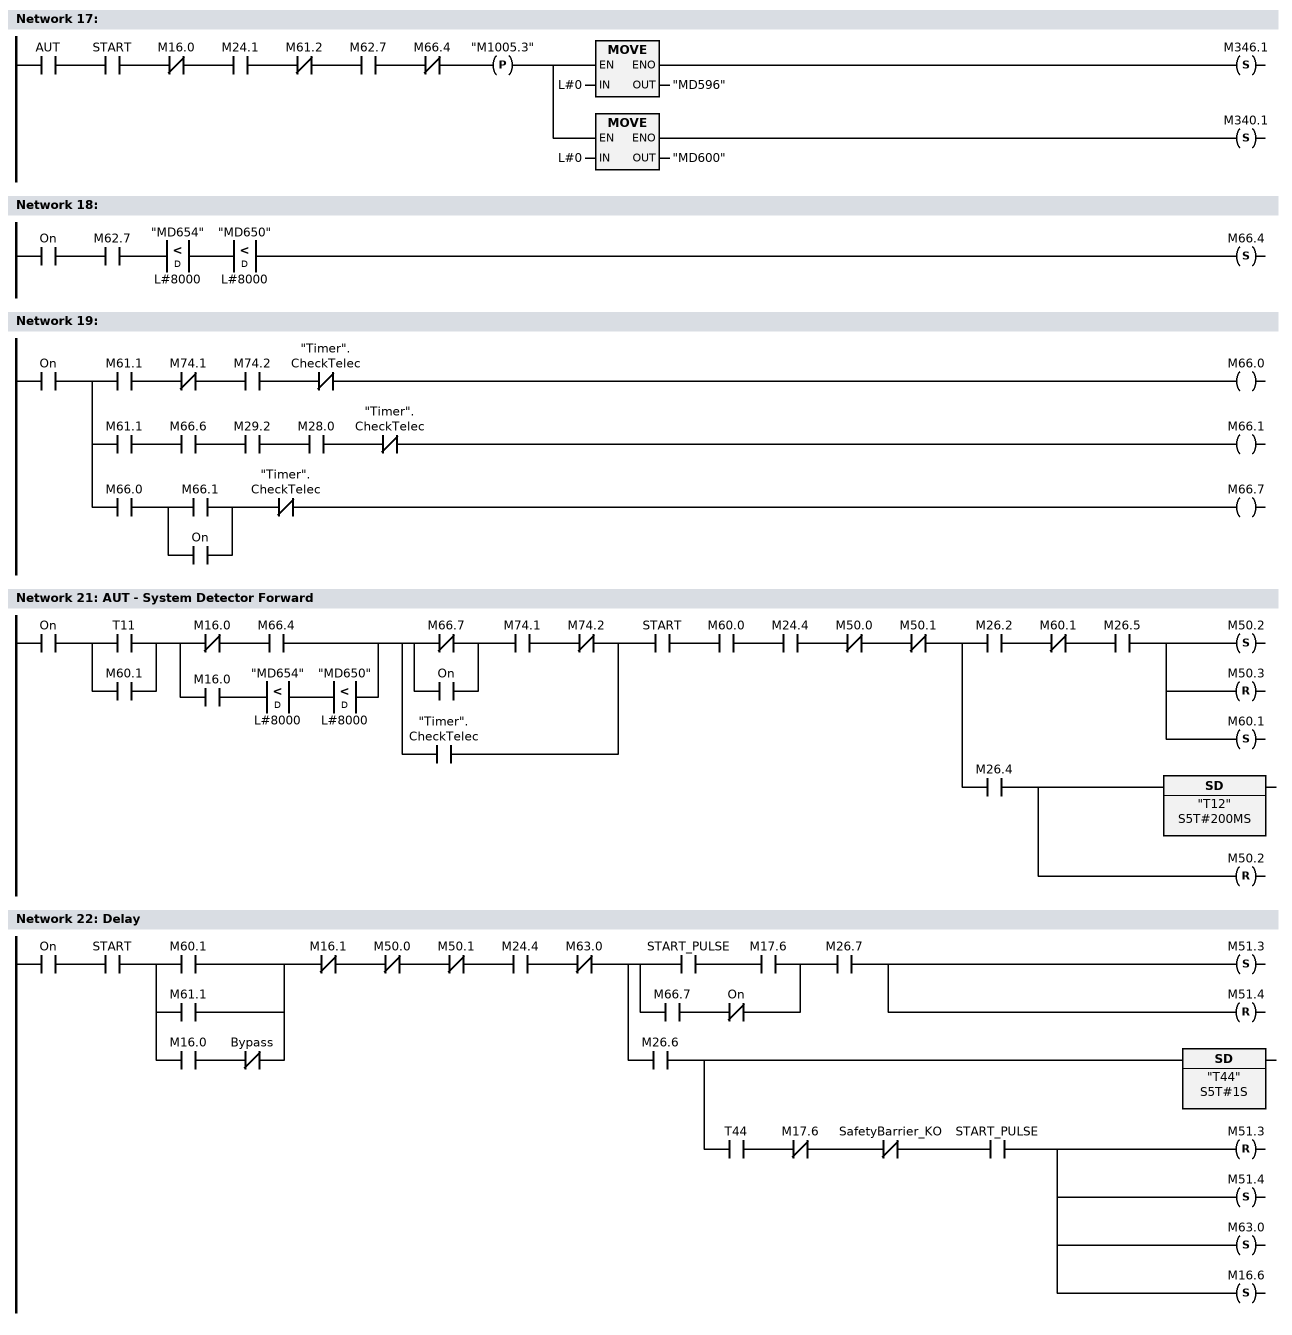
NETWORK
TITLE =
      A     "AUT";
      A     "START";
      AN    "M16.0";
      A     "M24.1";
      AN    "M61.2";
      A     "M62.7";
      AN    "M66.4";
      FP    "M1005.3";
      =     L 24.0;
      A     L 24.0;
      JNB   _008;
      L     L#0;
      T     "MD596";
      SET;
      SAVE;
      CLR;
_008: A     BR;
      S     "M346.1";
      A     L 24.0;
      JNB   _009;
      L     L#0;
      T     "MD600";
      SET;
      SAVE;
      CLR;
_009: A     BR;
      S     "M340.1";
NETWORK
TITLE =
      A     "On";
      A     "M62.7";
      A(;
      L     "MD654";
      L     L#8000;
      <D;
      );
      A(;
      L     "MD650";
      L     L#8000;
      <D;
      );
      S     "M66.4";
NETWORK
TITLE =
      A     "On";
      =     L 24.0;
      A     L 24.0;
      A     "M61.1";
      AN    "M74.1";
      A     "M74.2";
      AN    "Timer".CheckTelec;
      =     "M66.0";
      A     L 24.0;
      A     "M61.1";
      A     "M66.6";
      A     "M29.2";
      A     "M28.0";
      AN    "Timer".CheckTelec;
      =     "M66.1";
      A     L 24.0;
      A     "M66.0";
      A(;
      O     "M66.1";
      O     "On";
      );
      AN    "Timer".CheckTelec;
      =     "M66.7";
NETWORK
TITLE =
NETWORK
TITLE = AUT - System Detector Forward
      A     "On";
      A(;
      O     "T11";
      O     "M60.1";
      );
      A(;
      AN    "M16.0";
      A     "M66.4";
      O;
      A     "M16.0";
      A(;
      L     "MD654";
      L     L#8000;
      <D;
      );
      A(;
      L     "MD650";
      L     L#8000;
      <D;
      );
      );
      A(;
      A(;
      ON    "M66.7";
      O     "On";
      );
      A     "M74.1";
      AN    "M74.2";
      O     "Timer".CheckTelec;
      );
      A     "START";
      A     "M60.0";
      A     "M24.4";
      AN    "M50.0";
      AN    "M50.1";
      =     L 24.0;
      A     L 24.0;
      A     "M26.2";
      AN    "M60.1";
      A     "M26.5";
      S     "M50.2";
      R     "M50.3";
      S     "M60.1";
      A     L 24.0;
      A     "M26.4";
      L     S5T#200MS;
      SD    "T12";
      R     "M50.2";
NETWORK
TITLE = Delay
      A     "On";
      A     "START";
      A(;
      O     "M60.1";
      O     "M61.1";
      O;
      A     "M16.0";
      AN    "Bypass";
      );
      AN    "M16.1";
      AN    "M50.0";
      AN    "M50.1";
      A     "M24.4";
      AN    "M63.0";
      =     L 24.0;
      A     L 24.0;
      A(;
      A     "START_PULSE";
      A     "M17.6";
      O;
      A     "M66.7";
      AN    "On";
      );
      A     "M26.7";
      S     "M51.3";
      R     "M51.4";
      A     L 24.0;
      A     "M26.6";
      =     L 24.1;
      A     L 24.1;
      BLD   102;
      L     S5T#1S;
      SD    "T44";
      A     L 24.1;
      A     "T44";
      AN    "M17.6";
      AN    "SafetyBarrier_KO";
      A     "START_PULSE";
      R     "M51.3";
      S     "M51.4";
      S     "M63.0";
      S     "M16.6";
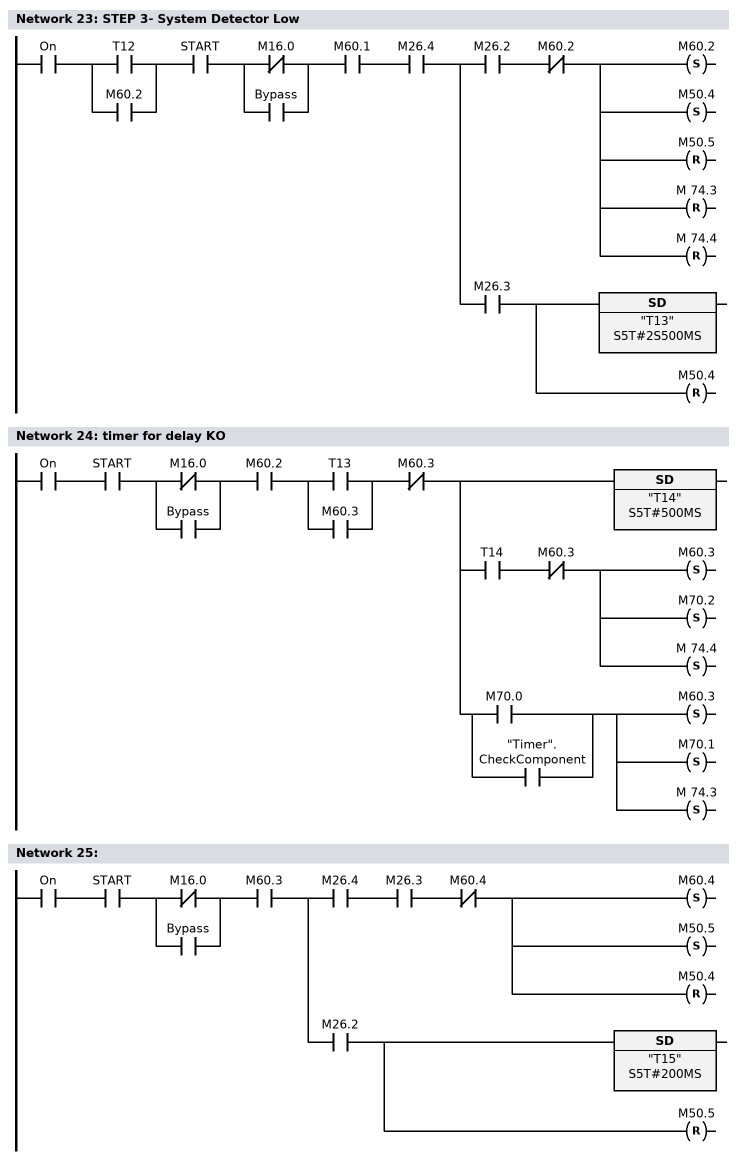
NETWORK
TITLE = STEP 3- System Detector Low
      A     "On";
      A(;
      O     "T12";
      O     "M60.2";
      );
      A     "START";
      A(;
      ON    "M16.0";
      O     "Bypass";
      );
      A     "M60.1";
      A     "M26.4";
      =     L 24.0;
      A     L 24.0;
      A     "M26.2";
      AN    "M60.2";
      S     "M60.2";
      S     "M50.4";
      R     "M50.5";
      R     M 74.3;
      R     M 74.4;
      A     L 24.0;
      A     "M26.3";
      L     S5T#2S500MS;
      SD    "T13";
      R     "M50.4";
NETWORK
TITLE = timer for delay KO
      A     "On";
      A     "START";
      A(;
      ON    "M16.0";
      O     "Bypass";
      );
      A     "M60.2";
      A(;
      O     "T13";
      O     "M60.3";
      );
      AN    "M60.3";
      =     L 24.0;
      A     L 24.0;
      BLD   102;
      L     S5T#500MS;
      SD    "T14";
      A     L 24.0;
      A     "T14";
      AN    "M60.3";
      S     "M60.3";
      S     "M70.2";
      S     M 74.4;
      A     L 24.0;
      A(;
      O     "M70.0";
      O     "Timer".CheckComponent;
      );
      S     "M60.3";
      S     "M70.1";
      S     M 74.3;
NETWORK
TITLE =
      A     "On";
      A     "START";
      A(;
      ON    "M16.0";
      O     "Bypass";
      );
      A     "M60.3";
      =     L 24.0;
      A     L 24.0;
      A     "M26.4";
      A     "M26.3";
      AN    "M60.4";
      S     "M60.4";
      S     "M50.5";
      R     "M50.4";
      A     L 24.0;
      A     "M26.2";
      L     S5T#200MS;
      SD    "T15";
      R     "M50.5";
